// TIA Portal V17 export
// export: Created 2025-03-05T07:59:04.4522338Z, ExportSetting WithDefaults, DisplayName Totally Integrated Automation Portal, DisplayVersion V17 Update 8, DisplayName TIA Portal Openness, DisplayVersion V17 Update 8, DisplayName TIA Portal Version Control Interface, DisplayVersion V17, DisplayName SINAMICS Startdrive Advanced, DisplayVersion V17 SP2, DisplayName SINAMICS Startdrive G110M, G120, G120C, G120D, G120P, G115D, DisplayVersion V17 SP2, DisplayName SINAMICS Startdrive G130, G150, S120, S150, SINAMICS MV, S210, DisplayVersion V17 SP2, DisplayName STEP 7 Professional, DisplayVersion V17 Update 8, DisplayName SINUMERIK ONE STEP 7 Toolbox, DisplayVersion V17 Update 12, DisplayName SINUMERIK 840D sl STEP 7 Toolbox, DisplayVersion V17 Update 12, DisplayName STEP 7 Safety, DisplayVersion V17 Update 6, DisplayName WinCC Advanced, DisplayVersion V17 Update 8
FUNCTION_BLOCK "FB2509_CYL_OPEN_CLOSE_FIX_CLADDING"   // FB2509, LAD
TITLE = CYLINDER CLOSE OPEN
{ S7_Optimized_Access := 'FALSE' }
AUTHOR : ETXETAR
VERSION : 1.0
// stored: AutoNumber false, IsIECCheckEnabled false, SetENOAutomatically false, UDAEnableTagReadback false
   VAR_INPUT
      OPTIONS_0 : Byte := 2#0000_0000;   // OPTIONS 0
      OPTIONS_1 : Byte := 2#0000_0000;   // OPTIONS 1
      OPTIONS_2 : Byte := 2#0000_0000;   // OPTIONS 2
      CLOSED_PART_A : Bool;   // CLOSED PART A INPUT
      CLOSED_PART_B : Bool;   // CLOSED PART B INPUT
      CLOSED_PART_C : Bool;   // CLOSED PART C INPUT
      CLOSED_PART_D : Bool;   // CLOSED PART D INPUT
      OPEN_PART_A : Bool;   // OPEN PART A INPUT
      OPEN_PART_B : Bool;   // OPEN PART B INPUT
      OPEN_PART_C : Bool;   // OPEN PART C INPUT
      OPEN_PART_D : Bool;   // OPEN PART D INPUT
      CLOSED_PRESSURE_SWITCH_1 : Bool;   // CLOSED PRESSURE SWITCH INPUT 1
      CLOSED_PRESSURE_SWITCH_2 : Bool;   // CLOSED PRESSURE SWITCH INPUT 2
      OPEN_PRESSURE_SWITCH_1 : Bool;   // OPEN PRESSURE SWITCH INPUT 1
      OPEN_PRESSURE_SWITCH_2 : Bool;   // OPEN PRESSURE SWITCH INPUT 2
      CLOSED_LOW_PRESSURE_SWITCH : Bool;   // CLOSED LOW PRESSURE SWITCH INPUT
      OPEN_LOW_PRESSURE_SWITCH : Bool;   // OPEN LOW PRESSURE SWITCH INPUT
      GENERAL_CONDITIONS : Bool;   // GENERAL CONDITIONS INPUT
      CLOSE_CONDITIONS : Bool;   // CLOSE CONDITIONS INPUT
      OPEN_CONDITIONS : Bool;   // OPEN CONDITIONS INPUT
      RELEASE_PRESSURE_CONDITIONS : Bool;   // RELEASE PRESSURE CONDITIONS INPUT
      LOW_PRESSURE_CONDITIONS : Bool;   // LOW PRESSURE CONDITIONS INPUT
      HYDRAULIC_OR_PNEUMATIC : Bool;   // HYDRAULIC OR PNEUMATIC IN SERVICE
      FIXTURE_PART_TYPE_SEL : Bool;   // FIXTURE PART TYPE SELECTED
      HMI_CMM_LINE_ACT_DEACT : Bool;   // HMI COMMAND LINE FOR CLOSE OPEN
      HMI_CMM_LINE_RELEASE_LOW : Bool;   // HMI COMMAND LINE FOR RELEASE LOW PRESSURE
      HMI_CLOSE_MAN_REQ : Bool;   // HMI CLOSE MANUAL REQUEST
      HMI_OPEN_MAN_REQ : Bool;   // HMI OPEN MANUAL REQUEST
      HMI_RELEASE_PRESSURE_MAN_REQ : Bool;   // HMI RELEASE PRESSURE MANUAL REQUEST
      HMI_LOW_PRESSURE_MAN_REQ : Bool;   // HMI LOW PRESSURE MANUAL REQUEST
      FLOWMETER_RESET : Bool;   // RESET FLOWMETER
      CLOSE_AUTO_REQ : Bool;   // CLOSE AUTOMATIC REQUEST
      OPEN_AUTO_REQ : Bool;   // OPEN AUTOMATIC REQUEST
      RELEASE_PRESSURE_AUTO_REQ : Bool;   // RELEASE PRESSURE AUTOMATIC REQUEST
      LOW_PRESSURE_AUTO_REQ : Bool;   // LOW PRESSURE AUTOMATIC REQUEST
      M_VERIFY_CLOSED : Bool;   // M CODE TO VERIFY CYLINDER CLOSED
      M_VERIFY_OPEN : Bool;   // M CODE TO VERIFY CYLINDER OPEN
      M_VERIFY_LOW_PRESSURE : Bool;   // M TO VERIFY LOW PRESSURED
      CHECK_CLOSED_CNC_PLC_SIGNAL : Bool;   // CHECK CLOSED CNC PLC SIGNAL
      CHECK_OPEN_CNC_PLC_SIGNAL : Bool;   // CHECK OPEN CNC PLC SIGNAL
      CHECK_CLOSED_LOW_PRESSURE_CNC_PLC_SIGNAL : Bool;   // CHECK CLOSED LOW PRESSURE CNC PLC SIGNAL
      CHECK_OPEN_LOW_PRESSURE_CNC_PLC_SIGNAL : Bool;   // CHECK OPEN LOW PRESSURE CNC PLC SIGNAL
      CLOSE_FLOW_ACTIVE : Bool;   // FLOWMETER CLOSE FLOW ACTIVE
      UNIT_ALARM : UInt;   // UNIT NUMBER MIN. NUMBER=1 MAX. NUMBER=3
      STATION_ALARM : UInt;   // UNIT NUMBER MIN. NUMBER=0 MAX. NUMBER=4
   END_VAR
   VAR_OUTPUT
      CLOSED : Bool;   // CLOSED
      OPEN_STATUS : Bool;   // OPEN
      PRESSURE_RELEASED : Bool;   // PRESSURE RELEASED
      LOW_PRESSURED : Bool;   // LOW PRESSURED
      HMI_MOTION_EXECUTABILITY_LEFT : Bool;   // HMI MOTION EXECUTABILITY LEFT
      HMI_MOTION_EXECUTABILITY_RIGHT : Bool;   // HMI MOTION EXECUTABILITY RIGHT
      HMI_MOTION_EXECUTABILITY_LEFT_2 : Bool;   // HMI MOTION EXECUTABILITY LEFT 2
      HMI_MOTION_EXECUTABILITY_RIGHT_2 : Bool;   // HMI MOTION EXECUTABILITY RIGHT 2
      HMI_MOTION_END_POS_LEFT : Bool;   // HMI MOTION END POSITION LEFT
      HMI_MOTION_END_POS_RIGHT : Bool;   // HMI MOTION END POSITION RIGHT
      HMI_MOTION_END_POS_LEFT_2 : Bool;   // HMI MOTION END POSITION LEFT 2
      HMI_MOTION_END_POS_RIGHT_2 : Bool;   // HMI MOTION END POSITION RIGHT 2
      HMI_MOTION_ACTIVE_LEFT : Bool;   // HMI MOTION ACTIVE LEFT
      HMI_MOTION_ACTIVE_RIGHT : Bool;   // HMI MOTION ACTIVE RIGHT
      HMI_MOTION_ACTIVE_LEFT_2 : Bool;   // HMI MOTION ACTIVE LEFT 2
      HMI_MOTION_ACTIVE_RIGHT_2 : Bool;   // HMI MOTION ACTIVE RIGHT 2
      ALARMS : "CYL_ALARMS_OPN_CLS";
      RESET_FLOWMETER : Bool;   // RESET FLOWMETER
      CLOSE : Bool;   // CLOSE
      OPEN_ACTION : Bool;   // OPEN
      LOW_PRESSURE : Bool;   // LOW PRESSURE
      SAFETY_UNBLOCK : Bool;   // SAFETY UNBLOCK
      PRESSURIZE_A : Bool;   // PRESSURIZE A
      PRESSURIZE_B : Bool;   // PRESSURIZE B
      PRESSURIZE_C : Bool;   // PRESSURIZE C
   END_VAR
   VAR_IN_OUT
      OPEN_FLOW_ACTIVE_FLOWMETER : Bool;   // FLOWMETER OPEN FLOW ACTIVE
   END_VAR
   VAR DB_SPECIFIC
      CYL { S7_SetPoint := 'True'} : "OPEN_CLOSE";
      TIMER_CLOSED { S7_SetPoint := 'True'} : TON_TIME;   // CLOSED TIMER
      TIMER_OPEN { S7_SetPoint := 'True'} : TON_TIME;   // OPEN TIMER
      TIMER_PRESSURE_RELEASED { S7_SetPoint := 'True'} : TON_TIME;   // PRESSURE RELEASED TIMER
      TIMER_LOW_PRESSURE { S7_SetPoint := 'True'} : TON_TIME;   // LOW PRESSURE TIMER
      TIMER_SIMULTANEITY { S7_SetPoint := 'True'} : TON_TIME;   // SIMULTANEITY TIMER
      TIMER_TIME_EXCEEDED { S7_SetPoint := 'True'} : TON_TIME;   // TIME EXCEEDED TIMER
      TIMER_ACTD_PRESSURE_TIME_EXCEEDED_1 { S7_SetPoint := 'True'} : TON_TIME;   // CLOSED PRESSURE TIME EXCEEDED TIMER 1
      TIMER_ACTD_PRESSURE_SWITCH_1 { S7_SetPoint := 'True'} : TON_TIME;   // CLOSED PRESSURE SWITCH TIMER 1
      "TIMER_ACTD PRESSURE_TIME_EXCEEDED_2" { S7_SetPoint := 'True'} : TON_TIME;   // CLOSED PRESSURE TIME EXCEEDED TIMER 2
      "TIMER_ACTD PRESSURE_SWITCH_2" { S7_SetPoint := 'True'} : TON_TIME;   // CLOSED PRESSURE SWITCH TIMER 2
      TIMER_DEACTD_PRESSURE_TIME_EXCEEDED_1 { S7_SetPoint := 'True'} : TON_TIME;   // OPEN PRESSURE TIME EXCEEDED TIMER 1
      TIMER_DEACTD_PRESSURE_SWITCH_1 { S7_SetPoint := 'True'} : TON_TIME;   // OPEN PRESSURE SWITCH TIMER 1
      TIMER_DEACTD_PRESSURE_TIME_EXCEEDED_2 { S7_SetPoint := 'True'} : TON_TIME;   // OPEN PRESSURE TIME EXCEEDED TIMER 2
      TIMER_DEACTD_PRESSURE_SWITCH_2 { S7_SetPoint := 'True'} : TON_TIME;   // OPEN PRESSURE SWITCH TIMER 2
      TIMER_ACTD_LOW_PRESSURE_TIME_EXCEEDED { S7_SetPoint := 'True'} : TON_TIME;   // CLOSED LOW PRESSURE TIME EXCEEDED TIMER
      TIMER_ACTD_LOW_PRESSURE_SWITCH { S7_SetPoint := 'True'} : TON_TIME;   // CLOSED LOW PRESSURE SWITCH TIMER
      TIMER_DEACTD_LOW_PRESSURE_TIME_EXCEEDED { S7_SetPoint := 'True'} : TON_TIME;   // OPEN LOW PRESSURE TIME EXCEEDED TIMER
      TIMER_DEACTD_LOW_PRESSURE_SWITCH { S7_SetPoint := 'True'} : TON_TIME;   // OPEN LOW PRESSURE SWITCH TIMER
      TIMER_SAFETY_UNBLOCK { S7_SetPoint := 'True'} : TOF_TIME;   // SAFETY UNBLOCK TIMER
      TIMER_CLMP_RCVRY_CLAMPED { S7_SetPoint := 'True'} : TON_TIME;   // CLAMP RECOVERY CLAMPED TIMER
      TIMER_CLMP_RCVRY_UNCLAMPED { S7_SetPoint := 'True'} : TON_TIME;   // CLAMP RECOVERY UNCLAMPED TIMER
   END_VAR
   VAR_TEMP
      INPUTS_MASK : Byte;   // INPUTS MASK
      O_BYTE_0 : Struct   // OPTIONS BYTE 0
         CLOSED_PART_A : Bool;   // CLOSED PART A OPTION
         CLOSED_PART_B : Bool;   // CLOSED PART B OPTION
         CLOSED_PART_C : Bool;   // CLOSED PART C OPTION
         CLOSED_PART_D : Bool;   // CLOSED PART D OPTION
         CLOSED_PRESSURE_INPUT_1 : Bool;   // CLOSED PRESSURE INPUT 1 OPTION
         CLOSED_PRESSURE_INPUT_2 : Bool;   // CLOSED PRESSURE INPUT 2 OPTION
         CLOSED_LOW_PRESSURE_INPUT : Bool;   // CLOSED LOW PRESSURE INPUT OPTION
         SPARE_7 : Bool;   // SPARE OPTION
      END_STRUCT;
      O_BYTE_1 : Struct   // OPTIONS BYTE 1
         OPEN_PART_A : Bool;   // OPEN PART A OPTION
         OPEN_PART_B : Bool;   // OPEN PART B OPTION
         OPEN_PART_C : Bool;   // OPEN PART C OPTION
         OPEN_PART_D : Bool;   // OPEN PART D OPTION
         OPEN_PRESSURE_INPUT_1 : Bool;   // OPEN PRESSURE INPUT 1 OPTION
         OPEN_PRESSURE_INPUT_2 : Bool;   // OPEN PRESSURE INPUT 2 OPTION
         OPEN_LOW_PRESSURE_INPUT : Bool;   // OPEN LOW PRESSURE INPUT OPTION
         SPARE_7 : Bool;   // SPARE OPTION
      END_STRUCT;
      O_BYTE_2 : Struct   // OPTIONS BYTE 2
         TWO_STATES_VALVE : Bool;   // TWO STATES VALVE OPTION
         HIGH_LOW_PRESSURE_VALVE : Bool;   // HIGH OR LOW PRESSURE VALVE OPTION
         OPEN_LOW : Bool;   // OPEN LOW OPTION
         SPARE_3 : Bool;   // SPARE OPTION
         SPARE_4 : Bool;   // SPARE OPTION
         SPARE_5 : Bool;   // SPARE OPTION
         SPARE_6 : Bool;   // SPARE OPTION
         CLAMP_RECOVERY : Bool;   // CLAMP RECOVERY OPTION
      END_STRUCT;
      DB_NUMBER : DInt;   // DB NUMBER FOR ALARM AND HELP DECODING
      CLAMP_RECOVERY_AUX : Bool;   // CLAMP RECOVERY AUXILIARY
   END_VAR
   // TIMER_CLOSED.PT := T#100MS;
   // TIMER_OPEN.PT := T#100MS;
   // TIMER_PRESSURE_RELEASED.PT := T#100MS;
   // TIMER_LOW_PRESSURE.PT := T#100MS;
   // TIMER_SIMULTANEITY.PT := T#100MS;
   // TIMER_TIME_EXCEEDED.PT := T#3S;
   // TIMER_ACTD_PRESSURE_TIME_EXCEEDED_1.PT := T#3S;
   // TIMER_ACTD_PRESSURE_SWITCH_1.PT := T#3S;
   // "TIMER_ACTD PRESSURE_TIME_EXCEEDED_2".PT := T#3S;
   // "TIMER_ACTD PRESSURE_SWITCH_2".PT := T#3S;
   // TIMER_DEACTD_PRESSURE_TIME_EXCEEDED_1.PT := T#3S;
   // TIMER_DEACTD_PRESSURE_SWITCH_1.PT := T#3S;
   // TIMER_DEACTD_PRESSURE_TIME_EXCEEDED_2.PT := T#3S;
   // TIMER_DEACTD_PRESSURE_SWITCH_2.PT := T#3S;
   // TIMER_ACTD_LOW_PRESSURE_TIME_EXCEEDED.PT := T#3S;
   // TIMER_ACTD_LOW_PRESSURE_SWITCH.PT := T#3S;
   // TIMER_DEACTD_LOW_PRESSURE_TIME_EXCEEDED.PT := T#3S;
   // TIMER_DEACTD_LOW_PRESSURE_SWITCH.PT := T#3S;
   // TIMER_SAFETY_UNBLOCK.PT := T#5s;
   // TIMER_CLMP_RCVRY_CLAMPED.PT := T#5s;
   // TIMER_CLMP_RCVRY_UNCLAMPED.PT := T#5s;
   VAR_TEMP   // added for the SCL form of the ladder/FBD networks
      _w1 : Bool;
      _w2 : Bool;
      _w3 : Bool;
      _w4 : Bool;
      _w5 : Bool;
      _w6 : Bool;
      _w7 : Bool;
      _w8 : Bool;
      _w9 : Bool;
      _w10 : Bool;
      _w11 : Bool;
      _w12 : Bool;
      _w13 : Bool;
   END_VAR
BEGIN

NETWORK
TITLE = READ INSTANCE DB
      L     DINO;
      +     10#800000;
      T     #DB_NUMBER;


REGION Network 2: OPTIONS
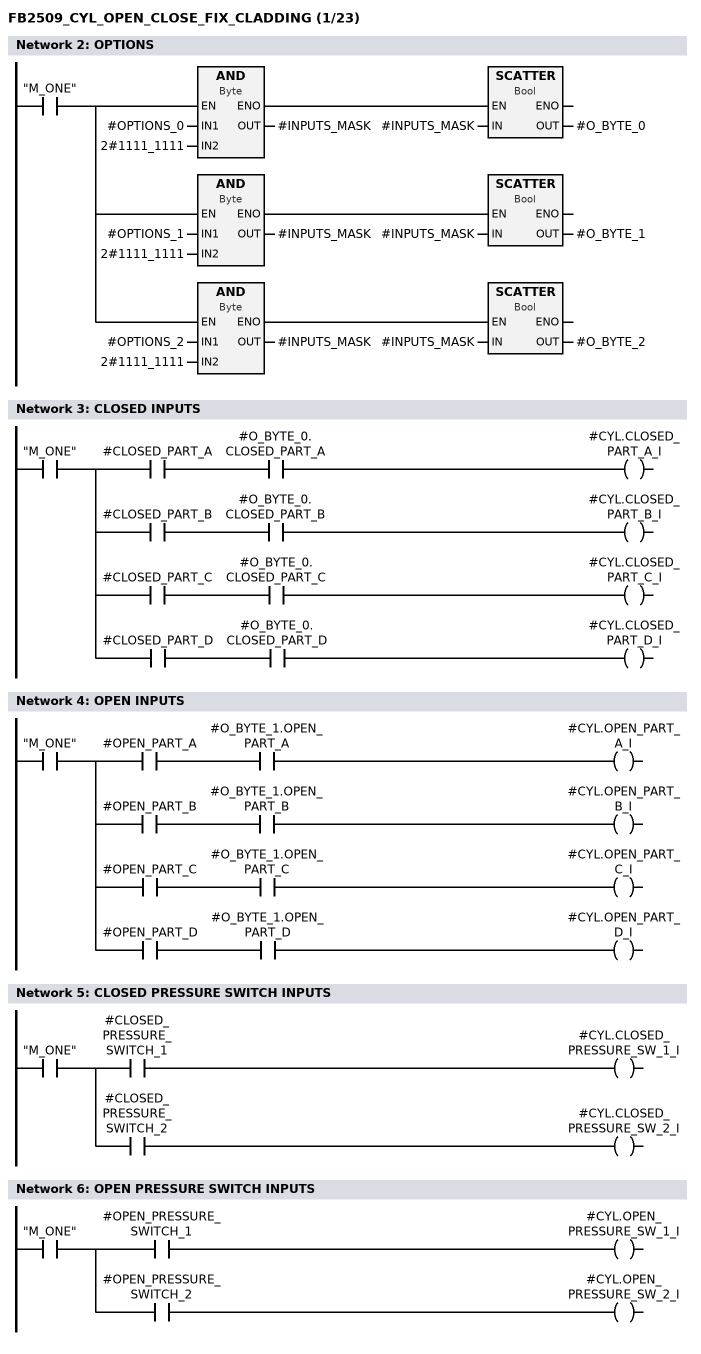
   RUNG wire#powerrail
      Contact( "M_ONE" )
      wire#w1
      { S7_Templates := "SrcType := Byte"; S7_GenerateENO := "TRUE" } And(in1 := #OPTIONS_0, in2 := 2#1111_1111, out => #INPUTS_MASK)
      { S7_Templates := "[dest_type := Bool, src_type := Byte]" } SCATTER(IN := #INPUTS_MASK, OUT => #O_BYTE_0)
   END_RUNG
   RUNG wire#w1
      { S7_Templates := "SrcType := Byte"; S7_GenerateENO := "TRUE" } And(in1 := #OPTIONS_1, in2 := 2#1111_1111, out => #INPUTS_MASK)
      { S7_Templates := "[dest_type := Bool, src_type := Byte]" } SCATTER(IN := #INPUTS_MASK, OUT => #O_BYTE_1)
   END_RUNG
   RUNG wire#w1
      { S7_Templates := "SrcType := Byte"; S7_GenerateENO := "TRUE" } And(in1 := #OPTIONS_2, in2 := 2#1111_1111, out => #INPUTS_MASK)
      { S7_Templates := "[dest_type := Bool, src_type := Byte]" } SCATTER(IN := #INPUTS_MASK, OUT => #O_BYTE_2)
   END_RUNG
   // the same network as SCL:
   IF "M_ONE" THEN #INPUTS_MASK := #OPTIONS_0 AND 2#1111_1111; END_IF;
   #_w1 := "M_ONE";
   IF #_w1 THEN
       SCATTER(IN := #INPUTS_MASK, OUT => #O_BYTE_0);
       #INPUTS_MASK := #OPTIONS_1 AND 2#1111_1111;
       SCATTER(IN := #INPUTS_MASK, OUT => #O_BYTE_1);
       #INPUTS_MASK := #OPTIONS_2 AND 2#1111_1111;
       SCATTER(IN := #INPUTS_MASK, OUT => #O_BYTE_2);
   END_IF;
END_REGION

REGION Network 3: CLOSED INPUTS
   RUNG wire#powerrail
      Contact( "M_ONE" )
      wire#w1
      Contact( #CLOSED_PART_A )
      Contact( #O_BYTE_0.CLOSED_PART_A )
      Coil( #CYL.CLOSED_PART_A_I )
   END_RUNG
   RUNG wire#w1
      Contact( #CLOSED_PART_B )
      Contact( #O_BYTE_0.CLOSED_PART_B )
      Coil( #CYL.CLOSED_PART_B_I )
   END_RUNG
   RUNG wire#w1
      Contact( #CLOSED_PART_C )
      Contact( #O_BYTE_0.CLOSED_PART_C )
      Coil( #CYL.CLOSED_PART_C_I )
   END_RUNG
   RUNG wire#w1
      Contact( #CLOSED_PART_D )
      Contact( #O_BYTE_0.CLOSED_PART_D )
      Coil( #CYL.CLOSED_PART_D_I )
   END_RUNG
   // the same network as SCL:
   #CYL.CLOSED_PART_A_I := "M_ONE" AND #CLOSED_PART_A AND #O_BYTE_0.CLOSED_PART_A;
   #CYL.CLOSED_PART_B_I := "M_ONE" AND #CLOSED_PART_B AND #O_BYTE_0.CLOSED_PART_B;
   #CYL.CLOSED_PART_C_I := "M_ONE" AND #CLOSED_PART_C AND #O_BYTE_0.CLOSED_PART_C;
   #CYL.CLOSED_PART_D_I := "M_ONE" AND #CLOSED_PART_D AND #O_BYTE_0.CLOSED_PART_D;
END_REGION

REGION Network 4: OPEN INPUTS
   RUNG wire#powerrail
      Contact( "M_ONE" )
      wire#w1
      Contact( #OPEN_PART_A )
      Contact( #O_BYTE_1.OPEN_PART_A )
      Coil( #CYL.OPEN_PART_A_I )
   END_RUNG
   RUNG wire#w1
      Contact( #OPEN_PART_B )
      Contact( #O_BYTE_1.OPEN_PART_B )
      Coil( #CYL.OPEN_PART_B_I )
   END_RUNG
   RUNG wire#w1
      Contact( #OPEN_PART_C )
      Contact( #O_BYTE_1.OPEN_PART_C )
      Coil( #CYL.OPEN_PART_C_I )
   END_RUNG
   RUNG wire#w1
      Contact( #OPEN_PART_D )
      Contact( #O_BYTE_1.OPEN_PART_D )
      Coil( #CYL.OPEN_PART_D_I )
   END_RUNG
   // the same network as SCL:
   #CYL.OPEN_PART_A_I := "M_ONE" AND #OPEN_PART_A AND #O_BYTE_1.OPEN_PART_A;
   #CYL.OPEN_PART_B_I := "M_ONE" AND #OPEN_PART_B AND #O_BYTE_1.OPEN_PART_B;
   #CYL.OPEN_PART_C_I := "M_ONE" AND #OPEN_PART_C AND #O_BYTE_1.OPEN_PART_C;
   #CYL.OPEN_PART_D_I := "M_ONE" AND #OPEN_PART_D AND #O_BYTE_1.OPEN_PART_D;
END_REGION

REGION Network 5: CLOSED PRESSURE SWITCH INPUTS
   RUNG wire#powerrail
      Contact( "M_ONE" )
      wire#w1
      Contact( #CLOSED_PRESSURE_SWITCH_1 )
      Coil( #CYL.CLOSED_PRESSURE_SW_1_I )
   END_RUNG
   RUNG wire#w1
      Contact( #CLOSED_PRESSURE_SWITCH_2 )
      Coil( #CYL.CLOSED_PRESSURE_SW_2_I )
   END_RUNG
   // the same network as SCL:
   #CYL.CLOSED_PRESSURE_SW_1_I := "M_ONE" AND #CLOSED_PRESSURE_SWITCH_1;
   #CYL.CLOSED_PRESSURE_SW_2_I := "M_ONE" AND #CLOSED_PRESSURE_SWITCH_2;
END_REGION

REGION Network 6: OPEN PRESSURE SWITCH INPUTS
   RUNG wire#powerrail
      Contact( "M_ONE" )
      wire#w1
      Contact( #OPEN_PRESSURE_SWITCH_1 )
      Coil( #CYL.OPEN_PRESSURE_SW_1_I )
   END_RUNG
   RUNG wire#w1
      Contact( #OPEN_PRESSURE_SWITCH_2 )
      Coil( #CYL.OPEN_PRESSURE_SW_2_I )
   END_RUNG
   // the same network as SCL:
   #CYL.OPEN_PRESSURE_SW_1_I := "M_ONE" AND #OPEN_PRESSURE_SWITCH_1;
   #CYL.OPEN_PRESSURE_SW_2_I := "M_ONE" AND #OPEN_PRESSURE_SWITCH_2;
END_REGION

REGION Network 7: LOW PRESSURE SWITCH INPUT
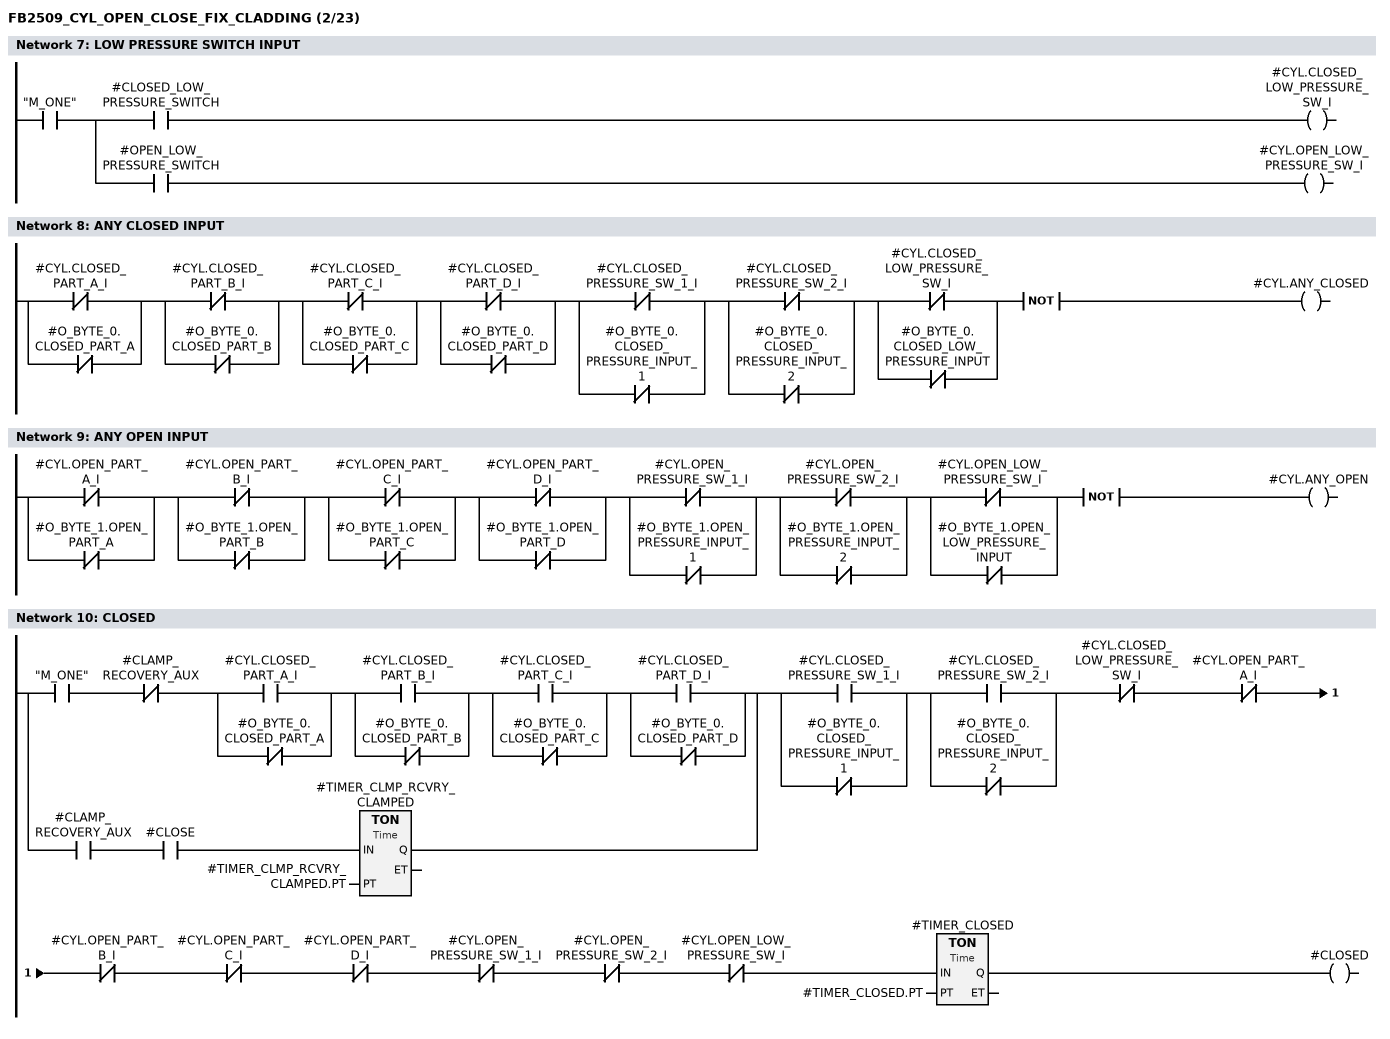
   RUNG wire#powerrail
      Contact( "M_ONE" )
      wire#w1
      Contact( #CLOSED_LOW_PRESSURE_SWITCH )
      Coil( #CYL.CLOSED_LOW_PRESSURE_SW_I )
   END_RUNG
   RUNG wire#w1
      Contact( #OPEN_LOW_PRESSURE_SWITCH )
      Coil( #CYL.OPEN_LOW_PRESSURE_SW_I )
   END_RUNG
   // the same network as SCL:
   #CYL.CLOSED_LOW_PRESSURE_SW_I := "M_ONE" AND #CLOSED_LOW_PRESSURE_SWITCH;
   #CYL.OPEN_LOW_PRESSURE_SW_I := "M_ONE" AND #OPEN_LOW_PRESSURE_SWITCH;
END_REGION

REGION Network 8: ANY CLOSED INPUT
   RUNG wire#powerrail
      I_Contact( #CYL.CLOSED_PART_A_I )
      wire#w1
      I_Contact( #CYL.CLOSED_PART_B_I )
      wire#w2
      I_Contact( #CYL.CLOSED_PART_C_I )
      wire#w3
      I_Contact( #CYL.CLOSED_PART_D_I )
      wire#w4
      I_Contact( #CYL.CLOSED_PRESSURE_SW_1_I )
      wire#w5
      I_Contact( #CYL.CLOSED_PRESSURE_SW_2_I )
      wire#w6
      I_Contact( #CYL.CLOSED_LOW_PRESSURE_SW_I )
      wire#w7
      Not()
      Coil( #CYL.ANY_CLOSED )
   END_RUNG
   RUNG wire#powerrail
      I_Contact( #O_BYTE_0.CLOSED_PART_A )
   END_RUNG wire#w1
   RUNG wire#w1
      I_Contact( #O_BYTE_0.CLOSED_PART_B )
   END_RUNG wire#w2
   RUNG wire#w2
      I_Contact( #O_BYTE_0.CLOSED_PART_C )
   END_RUNG wire#w3
   RUNG wire#w3
      I_Contact( #O_BYTE_0.CLOSED_PART_D )
   END_RUNG wire#w4
   RUNG wire#w4
      I_Contact( #O_BYTE_0.CLOSED_PRESSURE_INPUT_1 )
   END_RUNG wire#w5
   RUNG wire#w5
      I_Contact( #O_BYTE_0.CLOSED_PRESSURE_INPUT_2 )
   END_RUNG wire#w6
   RUNG wire#w6
      I_Contact( #O_BYTE_0.CLOSED_LOW_PRESSURE_INPUT )
   END_RUNG wire#w7
   // the same network as SCL:
   #CYL.ANY_CLOSED := NOT ((NOT #CYL.CLOSED_PART_A_I OR NOT #O_BYTE_0.CLOSED_PART_A) AND (NOT #CYL.CLOSED_PART_B_I OR NOT #O_BYTE_0.CLOSED_PART_B) AND (NOT #CYL.CLOSED_PART_C_I OR NOT #O_BYTE_0.CLOSED_PART_C) AND (NOT #CYL.CLOSED_PART_D_I OR NOT #O_BYTE_0.CLOSED_PART_D) AND (NOT #CYL.CLOSED_PRESSURE_SW_1_I OR NOT #O_BYTE_0.CLOSED_PRESSURE_INPUT_1) AND (NOT #CYL.CLOSED_PRESSURE_SW_2_I OR NOT #O_BYTE_0.CLOSED_PRESSURE_INPUT_2) AND (NOT #CYL.CLOSED_LOW_PRESSURE_SW_I OR NOT #O_BYTE_0.CLOSED_LOW_PRESSURE_INPUT));
END_REGION

REGION Network 9: ANY OPEN INPUT
   RUNG wire#powerrail
      I_Contact( #CYL.OPEN_PART_A_I )
      wire#w1
      I_Contact( #CYL.OPEN_PART_B_I )
      wire#w2
      I_Contact( #CYL.OPEN_PART_C_I )
      wire#w3
      I_Contact( #CYL.OPEN_PART_D_I )
      wire#w4
      I_Contact( #CYL.OPEN_PRESSURE_SW_1_I )
      wire#w5
      I_Contact( #CYL.OPEN_PRESSURE_SW_2_I )
      wire#w6
      I_Contact( #CYL.OPEN_LOW_PRESSURE_SW_I )
      wire#w7
      Not()
      Coil( #CYL.ANY_OPEN )
   END_RUNG
   RUNG wire#powerrail
      I_Contact( #O_BYTE_1.OPEN_PART_A )
   END_RUNG wire#w1
   RUNG wire#w1
      I_Contact( #O_BYTE_1.OPEN_PART_B )
   END_RUNG wire#w2
   RUNG wire#w2
      I_Contact( #O_BYTE_1.OPEN_PART_C )
   END_RUNG wire#w3
   RUNG wire#w3
      I_Contact( #O_BYTE_1.OPEN_PART_D )
   END_RUNG wire#w4
   RUNG wire#w4
      I_Contact( #O_BYTE_1.OPEN_PRESSURE_INPUT_1 )
   END_RUNG wire#w5
   RUNG wire#w5
      I_Contact( #O_BYTE_1.OPEN_PRESSURE_INPUT_2 )
   END_RUNG wire#w6
   RUNG wire#w6
      I_Contact( #O_BYTE_1.OPEN_LOW_PRESSURE_INPUT )
   END_RUNG wire#w7
   // the same network as SCL:
   #CYL.ANY_OPEN := NOT ((NOT #CYL.OPEN_PART_A_I OR NOT #O_BYTE_1.OPEN_PART_A) AND (NOT #CYL.OPEN_PART_B_I OR NOT #O_BYTE_1.OPEN_PART_B) AND (NOT #CYL.OPEN_PART_C_I OR NOT #O_BYTE_1.OPEN_PART_C) AND (NOT #CYL.OPEN_PART_D_I OR NOT #O_BYTE_1.OPEN_PART_D) AND (NOT #CYL.OPEN_PRESSURE_SW_1_I OR NOT #O_BYTE_1.OPEN_PRESSURE_INPUT_1) AND (NOT #CYL.OPEN_PRESSURE_SW_2_I OR NOT #O_BYTE_1.OPEN_PRESSURE_INPUT_2) AND (NOT #CYL.OPEN_LOW_PRESSURE_SW_I OR NOT #O_BYTE_1.OPEN_LOW_PRESSURE_INPUT));
END_REGION

REGION Network 10: CLOSED
   RUNG wire#powerrail
      Contact( "M_ONE" )
      I_Contact( #CLAMP_RECOVERY_AUX )
      wire#w1
      Contact( #CYL.CLOSED_PART_A_I )
      wire#w2
      Contact( #CYL.CLOSED_PART_B_I )
      wire#w3
      Contact( #CYL.CLOSED_PART_C_I )
      wire#w4
      Contact( #CYL.CLOSED_PART_D_I )
      wire#w5
      Contact( #CYL.CLOSED_PRESSURE_SW_1_I )
      wire#w6
      Contact( #CYL.CLOSED_PRESSURE_SW_2_I )
      wire#w7
      I_Contact( #CYL.CLOSED_LOW_PRESSURE_SW_I )
      I_Contact( #CYL.OPEN_PART_A_I )
      I_Contact( #CYL.OPEN_PART_B_I )
      I_Contact( #CYL.OPEN_PART_C_I )
      I_Contact( #CYL.OPEN_PART_D_I )
      I_Contact( #CYL.OPEN_PRESSURE_SW_1_I )
      I_Contact( #CYL.OPEN_PRESSURE_SW_2_I )
      I_Contact( #CYL.OPEN_LOW_PRESSURE_SW_I )
      { S7_Templates := "time_type := Time" } #TIMER_CLOSED.TON(pt := #TIMER_CLOSED.PT, et =>)
      Coil( #CLOSED )
   END_RUNG
   RUNG wire#w1
      I_Contact( #O_BYTE_0.CLOSED_PART_A )
   END_RUNG wire#w2
   RUNG wire#w2
      I_Contact( #O_BYTE_0.CLOSED_PART_B )
   END_RUNG wire#w3
   RUNG wire#w3
      I_Contact( #O_BYTE_0.CLOSED_PART_C )
   END_RUNG wire#w4
   RUNG wire#w4
      I_Contact( #O_BYTE_0.CLOSED_PART_D )
   END_RUNG wire#w5
   RUNG wire#powerrail
      Contact( #CLAMP_RECOVERY_AUX )
      Contact( #CLOSE )
      { S7_Templates := "time_type := Time" } #TIMER_CLMP_RCVRY_CLAMPED.TON(pt := #TIMER_CLMP_RCVRY_CLAMPED.PT, et =>)
   END_RUNG wire#w5
   RUNG wire#w5
      I_Contact( #O_BYTE_0.CLOSED_PRESSURE_INPUT_1 )
   END_RUNG wire#w6
   RUNG wire#w6
      I_Contact( #O_BYTE_0.CLOSED_PRESSURE_INPUT_2 )
   END_RUNG wire#w7
   // the same network as SCL:
   #TIMER_CLMP_RCVRY_CLAMPED(IN := #CLAMP_RECOVERY_AUX AND #CLOSE, PT := #TIMER_CLMP_RCVRY_CLAMPED.PT);   // TON
   #TIMER_CLOSED(IN := (("M_ONE" AND NOT #CLAMP_RECOVERY_AUX AND (#CYL.CLOSED_PART_A_I OR NOT #O_BYTE_0.CLOSED_PART_A) AND (#CYL.CLOSED_PART_B_I OR NOT #O_BYTE_0.CLOSED_PART_B) AND (#CYL.CLOSED_PART_C_I OR NOT #O_BYTE_0.CLOSED_PART_C) AND (#CYL.CLOSED_PART_D_I OR NOT #O_BYTE_0.CLOSED_PART_D)) OR #TIMER_CLMP_RCVRY_CLAMPED.Q) AND (#CYL.CLOSED_PRESSURE_SW_1_I OR NOT #O_BYTE_0.CLOSED_PRESSURE_INPUT_1) AND (#CYL.CLOSED_PRESSURE_SW_2_I OR NOT #O_BYTE_0.CLOSED_PRESSURE_INPUT_2) AND NOT #CYL.CLOSED_LOW_PRESSURE_SW_I AND NOT #CYL.OPEN_PART_A_I AND NOT #CYL.OPEN_PART_B_I AND NOT #CYL.OPEN_PART_C_I AND NOT #CYL.OPEN_PART_D_I AND NOT #CYL.OPEN_PRESSURE_SW_1_I AND NOT #CYL.OPEN_PRESSURE_SW_2_I AND NOT #CYL.OPEN_LOW_PRESSURE_SW_I,   // TON
                 PT := #TIMER_CLOSED.PT);
   #CLOSED := #TIMER_CLOSED.Q;
END_REGION

REGION Network 11: OPEN
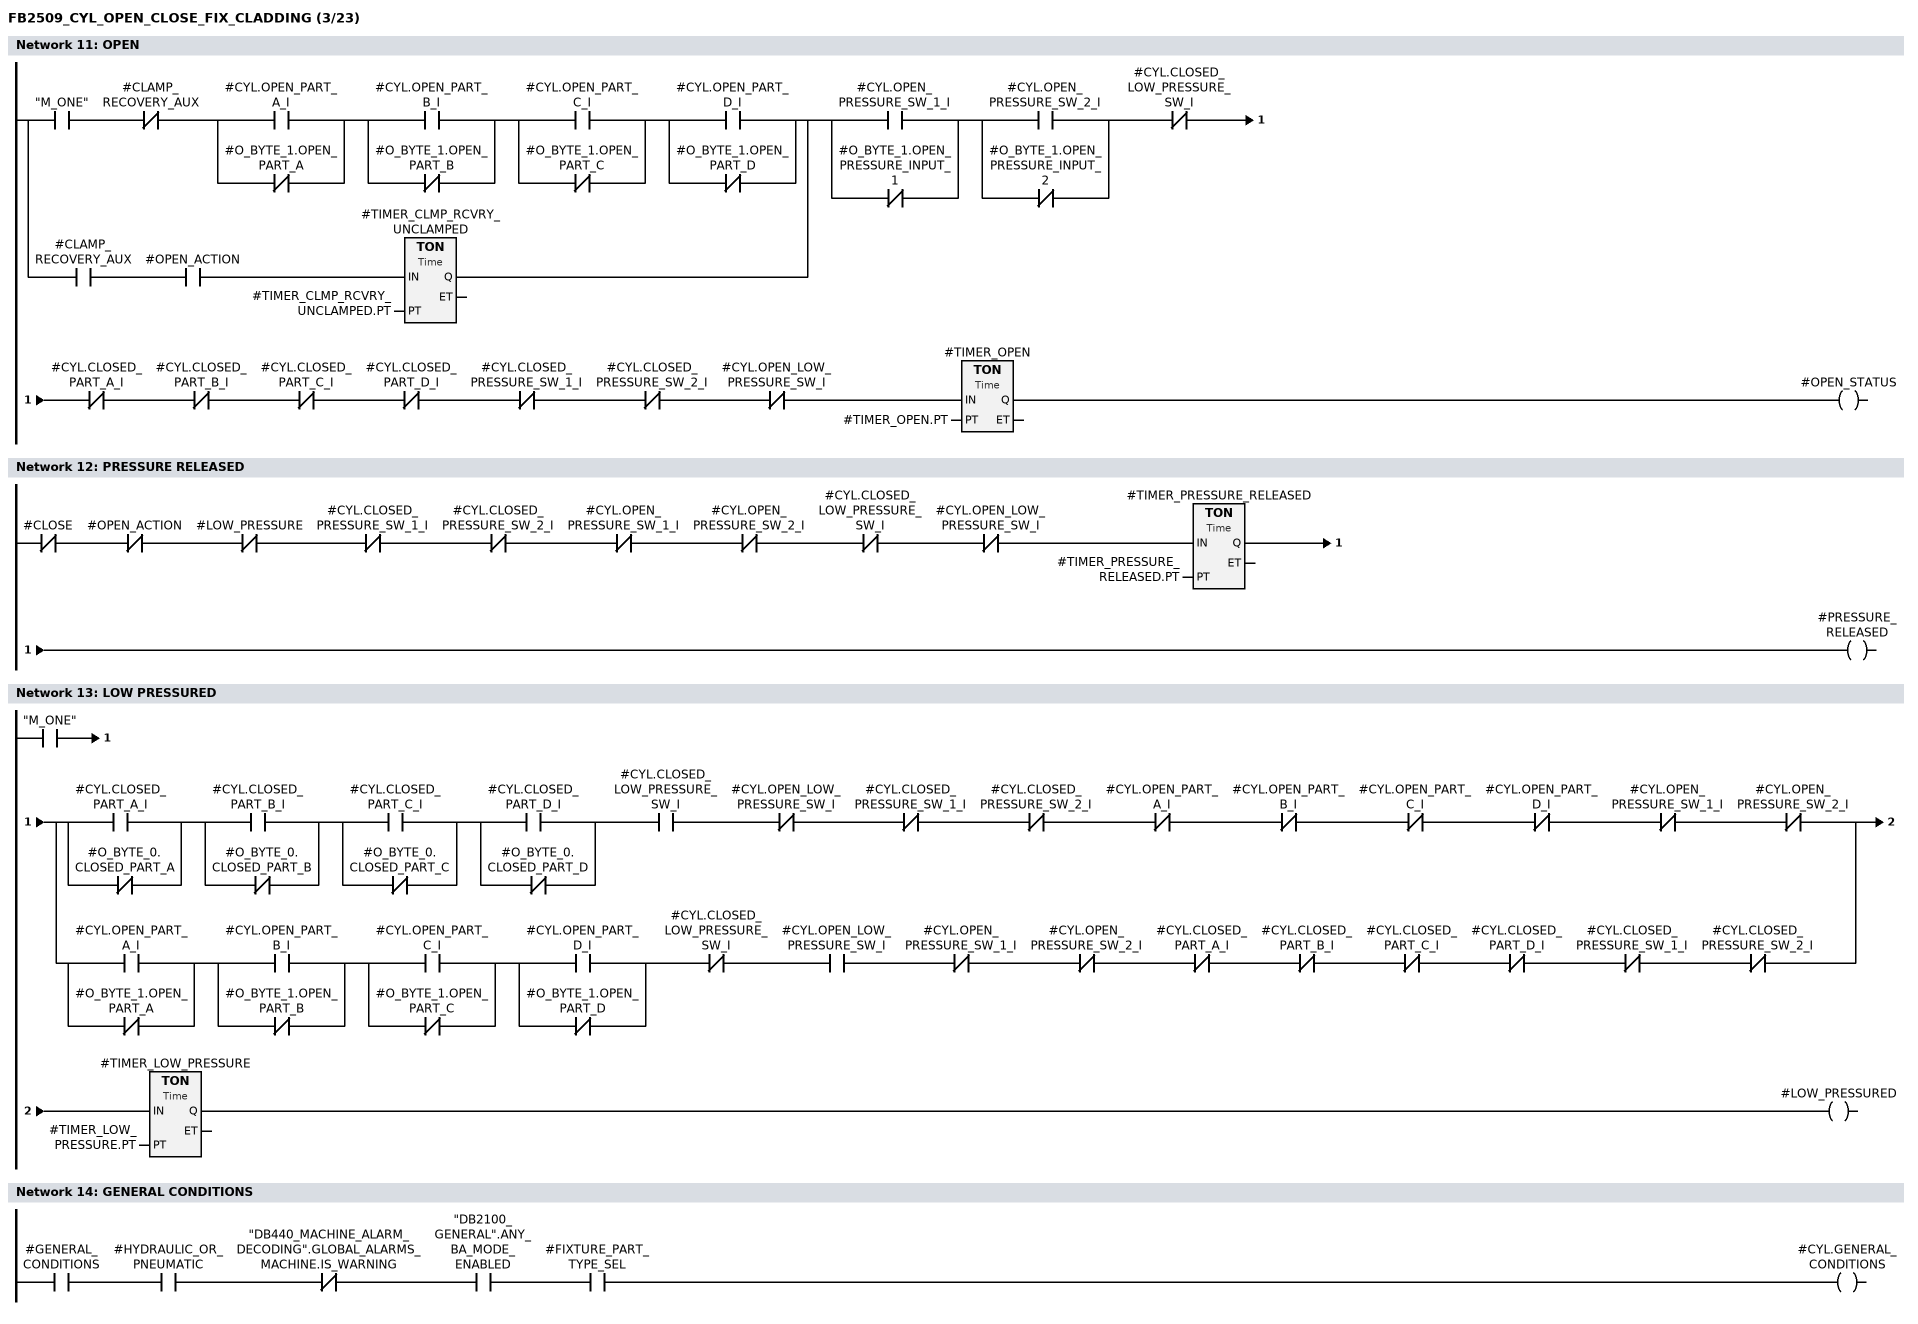
   RUNG wire#powerrail
      Contact( "M_ONE" )
      I_Contact( #CLAMP_RECOVERY_AUX )
      wire#w1
      Contact( #CYL.OPEN_PART_A_I )
      wire#w2
      Contact( #CYL.OPEN_PART_B_I )
      wire#w3
      Contact( #CYL.OPEN_PART_C_I )
      wire#w4
      Contact( #CYL.OPEN_PART_D_I )
      wire#w5
      Contact( #CYL.OPEN_PRESSURE_SW_1_I )
      wire#w6
      Contact( #CYL.OPEN_PRESSURE_SW_2_I )
      wire#w7
      I_Contact( #CYL.CLOSED_LOW_PRESSURE_SW_I )
      I_Contact( #CYL.CLOSED_PART_A_I )
      I_Contact( #CYL.CLOSED_PART_B_I )
      I_Contact( #CYL.CLOSED_PART_C_I )
      I_Contact( #CYL.CLOSED_PART_D_I )
      I_Contact( #CYL.CLOSED_PRESSURE_SW_1_I )
      I_Contact( #CYL.CLOSED_PRESSURE_SW_2_I )
      I_Contact( #CYL.OPEN_LOW_PRESSURE_SW_I )
      { S7_Templates := "time_type := Time" } #TIMER_OPEN.TON(pt := #TIMER_OPEN.PT, et =>)
      Coil( #OPEN_STATUS )
   END_RUNG
   RUNG wire#w1
      I_Contact( #O_BYTE_1.OPEN_PART_A )
   END_RUNG wire#w2
   RUNG wire#w2
      I_Contact( #O_BYTE_1.OPEN_PART_B )
   END_RUNG wire#w3
   RUNG wire#w3
      I_Contact( #O_BYTE_1.OPEN_PART_C )
   END_RUNG wire#w4
   RUNG wire#w4
      I_Contact( #O_BYTE_1.OPEN_PART_D )
   END_RUNG wire#w5
   RUNG wire#powerrail
      Contact( #CLAMP_RECOVERY_AUX )
      Contact( #OPEN_ACTION )
      { S7_Templates := "time_type := Time" } #TIMER_CLMP_RCVRY_UNCLAMPED.TON(pt := #TIMER_CLMP_RCVRY_UNCLAMPED.PT, et =>)
   END_RUNG wire#w5
   RUNG wire#w5
      I_Contact( #O_BYTE_1.OPEN_PRESSURE_INPUT_1 )
   END_RUNG wire#w6
   RUNG wire#w6
      I_Contact( #O_BYTE_1.OPEN_PRESSURE_INPUT_2 )
   END_RUNG wire#w7
   // the same network as SCL:
   #TIMER_CLMP_RCVRY_UNCLAMPED(IN := #CLAMP_RECOVERY_AUX AND #OPEN_ACTION, PT := #TIMER_CLMP_RCVRY_UNCLAMPED.PT);   // TON
   #TIMER_OPEN(IN := (("M_ONE" AND NOT #CLAMP_RECOVERY_AUX AND (#CYL.OPEN_PART_A_I OR NOT #O_BYTE_1.OPEN_PART_A) AND (#CYL.OPEN_PART_B_I OR NOT #O_BYTE_1.OPEN_PART_B) AND (#CYL.OPEN_PART_C_I OR NOT #O_BYTE_1.OPEN_PART_C) AND (#CYL.OPEN_PART_D_I OR NOT #O_BYTE_1.OPEN_PART_D)) OR #TIMER_CLMP_RCVRY_UNCLAMPED.Q) AND (#CYL.OPEN_PRESSURE_SW_1_I OR NOT #O_BYTE_1.OPEN_PRESSURE_INPUT_1) AND (#CYL.OPEN_PRESSURE_SW_2_I OR NOT #O_BYTE_1.OPEN_PRESSURE_INPUT_2) AND NOT #CYL.CLOSED_LOW_PRESSURE_SW_I AND NOT #CYL.CLOSED_PART_A_I AND NOT #CYL.CLOSED_PART_B_I AND NOT #CYL.CLOSED_PART_C_I AND NOT #CYL.CLOSED_PART_D_I AND NOT #CYL.CLOSED_PRESSURE_SW_1_I AND NOT #CYL.CLOSED_PRESSURE_SW_2_I AND NOT #CYL.OPEN_LOW_PRESSURE_SW_I,   // TON
               PT := #TIMER_OPEN.PT);
   #OPEN_STATUS := #TIMER_OPEN.Q;
END_REGION

REGION Network 12: PRESSURE RELEASED
   RUNG wire#powerrail
      I_Contact( #CLOSE )
      I_Contact( #OPEN_ACTION )
      I_Contact( #LOW_PRESSURE )
      I_Contact( #CYL.CLOSED_PRESSURE_SW_1_I )
      I_Contact( #CYL.CLOSED_PRESSURE_SW_2_I )
      I_Contact( #CYL.OPEN_PRESSURE_SW_1_I )
      I_Contact( #CYL.OPEN_PRESSURE_SW_2_I )
      I_Contact( #CYL.CLOSED_LOW_PRESSURE_SW_I )
      I_Contact( #CYL.OPEN_LOW_PRESSURE_SW_I )
      { S7_Templates := "time_type := Time" } #TIMER_PRESSURE_RELEASED.TON(pt := #TIMER_PRESSURE_RELEASED.PT, et =>)
      Coil( #PRESSURE_RELEASED )
   END_RUNG
   // the same network as SCL:
   #TIMER_PRESSURE_RELEASED(IN := NOT #CLOSE AND NOT #OPEN_ACTION AND NOT #LOW_PRESSURE AND NOT #CYL.CLOSED_PRESSURE_SW_1_I AND NOT #CYL.CLOSED_PRESSURE_SW_2_I AND NOT #CYL.OPEN_PRESSURE_SW_1_I AND NOT #CYL.OPEN_PRESSURE_SW_2_I AND NOT #CYL.CLOSED_LOW_PRESSURE_SW_I AND NOT #CYL.OPEN_LOW_PRESSURE_SW_I,   // TON
                           PT := #TIMER_PRESSURE_RELEASED.PT);
   #PRESSURE_RELEASED := #TIMER_PRESSURE_RELEASED.Q;
END_REGION

REGION Network 13: LOW PRESSURED
   RUNG wire#powerrail
      Contact( "M_ONE" )
      wire#w1
      Contact( #CYL.CLOSED_PART_A_I )
      wire#w2
      Contact( #CYL.CLOSED_PART_B_I )
      wire#w3
      Contact( #CYL.CLOSED_PART_C_I )
      wire#w4
      Contact( #CYL.CLOSED_PART_D_I )
      wire#w5
      Contact( #CYL.CLOSED_LOW_PRESSURE_SW_I )
      I_Contact( #CYL.OPEN_LOW_PRESSURE_SW_I )
      I_Contact( #CYL.CLOSED_PRESSURE_SW_1_I )
      I_Contact( #CYL.CLOSED_PRESSURE_SW_2_I )
      I_Contact( #CYL.OPEN_PART_A_I )
      I_Contact( #CYL.OPEN_PART_B_I )
      I_Contact( #CYL.OPEN_PART_C_I )
      I_Contact( #CYL.OPEN_PART_D_I )
      I_Contact( #CYL.OPEN_PRESSURE_SW_1_I )
      I_Contact( #CYL.OPEN_PRESSURE_SW_2_I )
      wire#w6
      { S7_Templates := "time_type := Time" } #TIMER_LOW_PRESSURE.TON(pt := #TIMER_LOW_PRESSURE.PT, et =>)
      Coil( #LOW_PRESSURED )
   END_RUNG
   RUNG wire#w1
      I_Contact( #O_BYTE_0.CLOSED_PART_A )
   END_RUNG wire#w2
   RUNG wire#w2
      I_Contact( #O_BYTE_0.CLOSED_PART_B )
   END_RUNG wire#w3
   RUNG wire#w3
      I_Contact( #O_BYTE_0.CLOSED_PART_C )
   END_RUNG wire#w4
   RUNG wire#w4
      I_Contact( #O_BYTE_0.CLOSED_PART_D )
   END_RUNG wire#w5
   RUNG wire#w1
      Contact( #CYL.OPEN_PART_A_I )
      wire#w7
      Contact( #CYL.OPEN_PART_B_I )
      wire#w8
      Contact( #CYL.OPEN_PART_C_I )
      wire#w9
      Contact( #CYL.OPEN_PART_D_I )
      wire#w10
      I_Contact( #CYL.CLOSED_LOW_PRESSURE_SW_I )
      Contact( #CYL.OPEN_LOW_PRESSURE_SW_I )
      I_Contact( #CYL.OPEN_PRESSURE_SW_1_I )
      I_Contact( #CYL.OPEN_PRESSURE_SW_2_I )
      I_Contact( #CYL.CLOSED_PART_A_I )
      I_Contact( #CYL.CLOSED_PART_B_I )
      I_Contact( #CYL.CLOSED_PART_C_I )
      I_Contact( #CYL.CLOSED_PART_D_I )
      I_Contact( #CYL.CLOSED_PRESSURE_SW_1_I )
      I_Contact( #CYL.CLOSED_PRESSURE_SW_2_I )
   END_RUNG wire#w6
   RUNG wire#w1
      I_Contact( #O_BYTE_1.OPEN_PART_A )
   END_RUNG wire#w7
   RUNG wire#w7
      I_Contact( #O_BYTE_1.OPEN_PART_B )
   END_RUNG wire#w8
   RUNG wire#w8
      I_Contact( #O_BYTE_1.OPEN_PART_C )
   END_RUNG wire#w9
   RUNG wire#w9
      I_Contact( #O_BYTE_1.OPEN_PART_D )
   END_RUNG wire#w10
   // the same network as SCL:
   #TIMER_LOW_PRESSURE(IN := "M_ONE" AND (((#CYL.CLOSED_PART_A_I OR NOT #O_BYTE_0.CLOSED_PART_A) AND (#CYL.CLOSED_PART_B_I OR NOT #O_BYTE_0.CLOSED_PART_B) AND (#CYL.CLOSED_PART_C_I OR NOT #O_BYTE_0.CLOSED_PART_C) AND (#CYL.CLOSED_PART_D_I OR NOT #O_BYTE_0.CLOSED_PART_D) AND #CYL.CLOSED_LOW_PRESSURE_SW_I AND NOT #CYL.OPEN_LOW_PRESSURE_SW_I AND NOT #CYL.CLOSED_PRESSURE_SW_1_I AND NOT #CYL.CLOSED_PRESSURE_SW_2_I AND NOT #CYL.OPEN_PART_A_I AND NOT #CYL.OPEN_PART_B_I AND NOT #CYL.OPEN_PART_C_I AND NOT #CYL.OPEN_PART_D_I AND NOT #CYL.OPEN_PRESSURE_SW_1_I AND NOT #CYL.OPEN_PRESSURE_SW_2_I) OR ((#CYL.OPEN_PART_A_I OR NOT #O_BYTE_1.OPEN_PART_A) AND (#CYL.OPEN_PART_B_I OR NOT #O_BYTE_1.OPEN_PART_B) AND (#CYL.OPEN_PART_C_I OR NOT #O_BYTE_1.OPEN_PART_C) AND (#CYL.OPEN_PART_D_I OR NOT #O_BYTE_1.OPEN_PART_D) AND NOT #CYL.CLOSED_LOW_PRESSURE_SW_I AND #CYL.OPEN_LOW_PRESSURE_SW_I AND NOT #CYL.OPEN_PRESSURE_SW_1_I AND NOT #CYL.OPEN_PRESSURE_SW_2_I AND NOT #CYL.CLOSED_PART_A_I AND NOT #CYL.CLOSED_PART_B_I AND NOT #CYL.CLOSED_PART_C_I AND NOT #CYL.CLOSED_PART_D_I AND NOT #CYL.CLOSED_PRESSURE_SW_1_I AND NOT #CYL.CLOSED_PRESSURE_SW_2_I)),   // TON
                       PT := #TIMER_LOW_PRESSURE.PT);
   #LOW_PRESSURED := #TIMER_LOW_PRESSURE.Q;
END_REGION

REGION Network 14: GENERAL CONDITIONS
   RUNG wire#powerrail
      Contact( #GENERAL_CONDITIONS )
      Contact( #HYDRAULIC_OR_PNEUMATIC )
      I_Contact( "DB440_MACHINE_ALARM_DECODING".GLOBAL_ALARMS_MACHINE.IS_WARNING )
      Contact( "DB2100_GENERAL".ANY_BA_MODE_ENABLED )
      Contact( #FIXTURE_PART_TYPE_SEL )
      Coil( #CYL.GENERAL_CONDITIONS )
   END_RUNG
   // the same network as SCL:
   #CYL.GENERAL_CONDITIONS := #GENERAL_CONDITIONS AND #HYDRAULIC_OR_PNEUMATIC AND NOT "DB440_MACHINE_ALARM_DECODING".GLOBAL_ALARMS_MACHINE.IS_WARNING AND "DB2100_GENERAL".ANY_BA_MODE_ENABLED AND #FIXTURE_PART_TYPE_SEL;
END_REGION

REGION Network 15: OPERATOR HELP
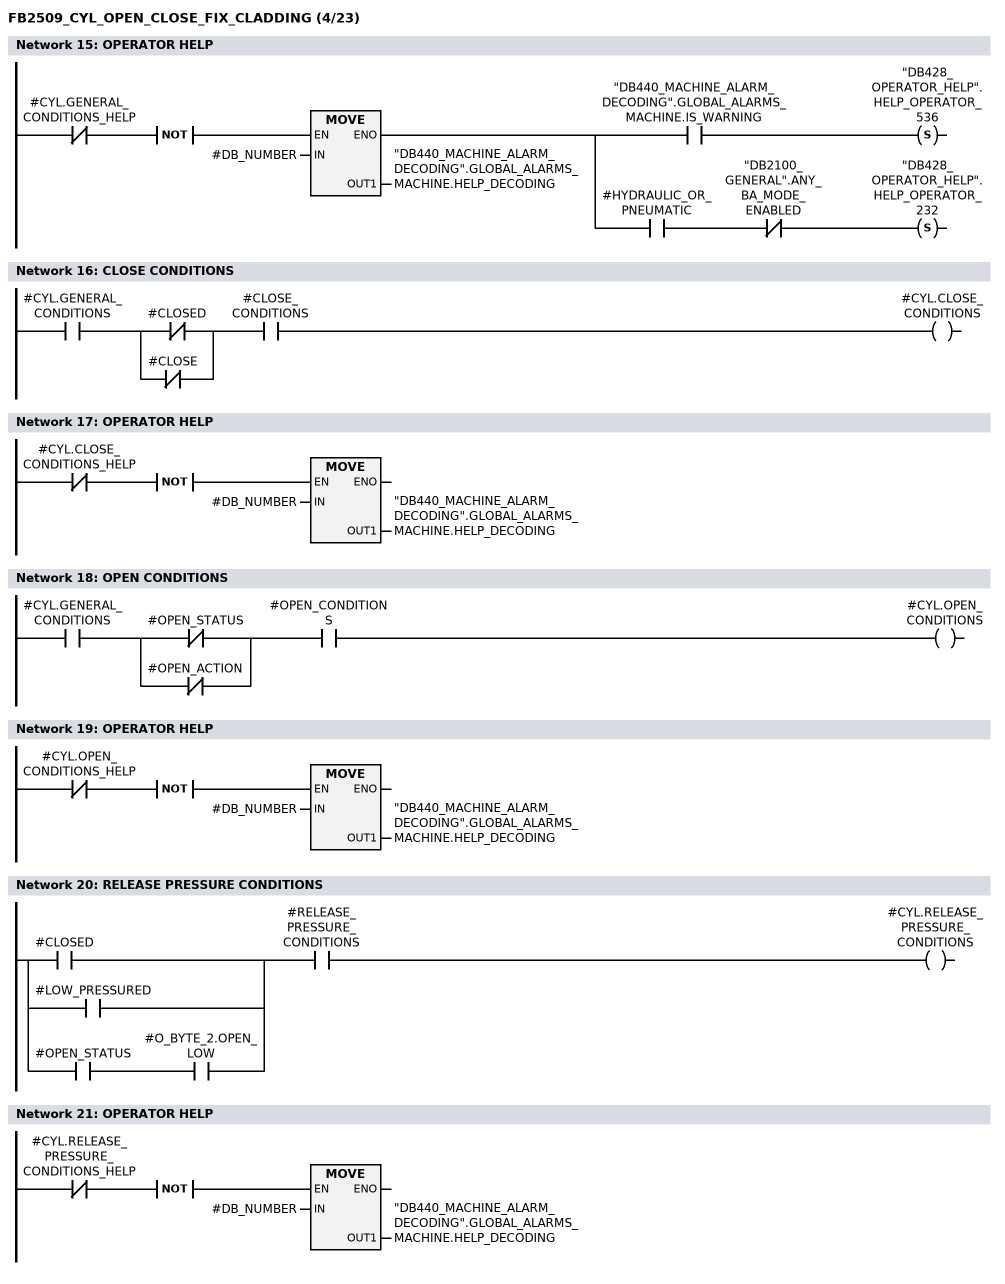
   RUNG wire#powerrail
      I_Contact( #CYL.GENERAL_CONDITIONS_HELP )
      Not()
      { S7_GenerateENO := "TRUE" } Move(in := #DB_NUMBER, out1 => "DB440_MACHINE_ALARM_DECODING".GLOBAL_ALARMS_MACHINE.HELP_DECODING)
      wire#w1
      Contact( "DB440_MACHINE_ALARM_DECODING".GLOBAL_ALARMS_MACHINE.IS_WARNING )
      S_Coil( "DB428_OPERATOR_HELP".HELP_OPERATOR_536 )
   END_RUNG
   RUNG wire#w1
      Contact( #HYDRAULIC_OR_PNEUMATIC )
      I_Contact( "DB2100_GENERAL".ANY_BA_MODE_ENABLED )
      S_Coil( "DB428_OPERATOR_HELP".HELP_OPERATOR_232 )
   END_RUNG
   // the same network as SCL:
   // ENO of a box is taken as its EN; it also drops when the box reports an error
   #_w1 := NOT (NOT #CYL.GENERAL_CONDITIONS_HELP);
   IF #_w1 THEN "DB440_MACHINE_ALARM_DECODING".GLOBAL_ALARMS_MACHINE.HELP_DECODING := #DB_NUMBER; END_IF;
   IF #_w1 AND "DB440_MACHINE_ALARM_DECODING".GLOBAL_ALARMS_MACHINE.IS_WARNING THEN
       "DB428_OPERATOR_HELP".HELP_OPERATOR_536 := TRUE;
   END_IF;
   IF #_w1 AND #HYDRAULIC_OR_PNEUMATIC AND NOT "DB2100_GENERAL".ANY_BA_MODE_ENABLED THEN
       "DB428_OPERATOR_HELP".HELP_OPERATOR_232 := TRUE;
   END_IF;
END_REGION

REGION Network 16: CLOSE CONDITIONS
   RUNG wire#powerrail
      Contact( #CYL.GENERAL_CONDITIONS )
      wire#w1
      I_Contact( #CLOSED )
      wire#w2
      Contact( #CLOSE_CONDITIONS )
      Coil( #CYL.CLOSE_CONDITIONS )
   END_RUNG
   RUNG wire#w1
      I_Contact( #CLOSE )
   END_RUNG wire#w2
   // the same network as SCL:
   #CYL.CLOSE_CONDITIONS := #CYL.GENERAL_CONDITIONS AND (NOT #CLOSED OR NOT #CLOSE) AND #CLOSE_CONDITIONS;
END_REGION

REGION Network 17: OPERATOR HELP
   RUNG wire#powerrail
      I_Contact( #CYL.CLOSE_CONDITIONS_HELP )
      Not()
      { S7_GenerateENO := "TRUE" } Move(in := #DB_NUMBER, out1 => "DB440_MACHINE_ALARM_DECODING".GLOBAL_ALARMS_MACHINE.HELP_DECODING)
   END_RUNG
   // the same network as SCL:
   IF NOT (NOT #CYL.CLOSE_CONDITIONS_HELP) THEN
       "DB440_MACHINE_ALARM_DECODING".GLOBAL_ALARMS_MACHINE.HELP_DECODING := #DB_NUMBER;
   END_IF;
END_REGION

REGION Network 18: OPEN CONDITIONS
   RUNG wire#powerrail
      Contact( #CYL.GENERAL_CONDITIONS )
      wire#w1
      I_Contact( #OPEN_STATUS )
      wire#w2
      Contact( #OPEN_CONDITIONS )
      Coil( #CYL.OPEN_CONDITIONS )
   END_RUNG
   RUNG wire#w1
      I_Contact( #OPEN_ACTION )
   END_RUNG wire#w2
   // the same network as SCL:
   #CYL.OPEN_CONDITIONS := #CYL.GENERAL_CONDITIONS AND (NOT #OPEN_STATUS OR NOT #OPEN_ACTION) AND #OPEN_CONDITIONS;
END_REGION

REGION Network 19: OPERATOR HELP
   RUNG wire#powerrail
      I_Contact( #CYL.OPEN_CONDITIONS_HELP )
      Not()
      { S7_GenerateENO := "TRUE" } Move(in := #DB_NUMBER, out1 => "DB440_MACHINE_ALARM_DECODING".GLOBAL_ALARMS_MACHINE.HELP_DECODING)
   END_RUNG
   // the same network as SCL:
   IF NOT (NOT #CYL.OPEN_CONDITIONS_HELP) THEN
       "DB440_MACHINE_ALARM_DECODING".GLOBAL_ALARMS_MACHINE.HELP_DECODING := #DB_NUMBER;
   END_IF;
END_REGION

REGION Network 20: RELEASE PRESSURE CONDITIONS
   RUNG wire#powerrail
      Contact( #CLOSED )
      wire#w1
      Contact( #RELEASE_PRESSURE_CONDITIONS )
      Coil( #CYL.RELEASE_PRESSURE_CONDITIONS )
   END_RUNG
   RUNG wire#powerrail
      Contact( #LOW_PRESSURED )
   END_RUNG wire#w1
   RUNG wire#powerrail
      Contact( #OPEN_STATUS )
      Contact( #O_BYTE_2.OPEN_LOW )
   END_RUNG wire#w1
   // the same network as SCL:
   #CYL.RELEASE_PRESSURE_CONDITIONS := (#CLOSED OR #LOW_PRESSURED OR (#OPEN_STATUS AND #O_BYTE_2.OPEN_LOW)) AND #RELEASE_PRESSURE_CONDITIONS;
END_REGION

REGION Network 21: OPERATOR HELP
   RUNG wire#powerrail
      I_Contact( #CYL.RELEASE_PRESSURE_CONDITIONS_HELP )
      Not()
      { S7_GenerateENO := "TRUE" } Move(in := #DB_NUMBER, out1 => "DB440_MACHINE_ALARM_DECODING".GLOBAL_ALARMS_MACHINE.HELP_DECODING)
   END_RUNG
   // the same network as SCL:
   IF NOT (NOT #CYL.RELEASE_PRESSURE_CONDITIONS_HELP) THEN
       "DB440_MACHINE_ALARM_DECODING".GLOBAL_ALARMS_MACHINE.HELP_DECODING := #DB_NUMBER;
   END_IF;
END_REGION

REGION Network 22: LOW PRESSURE CONDITIONS
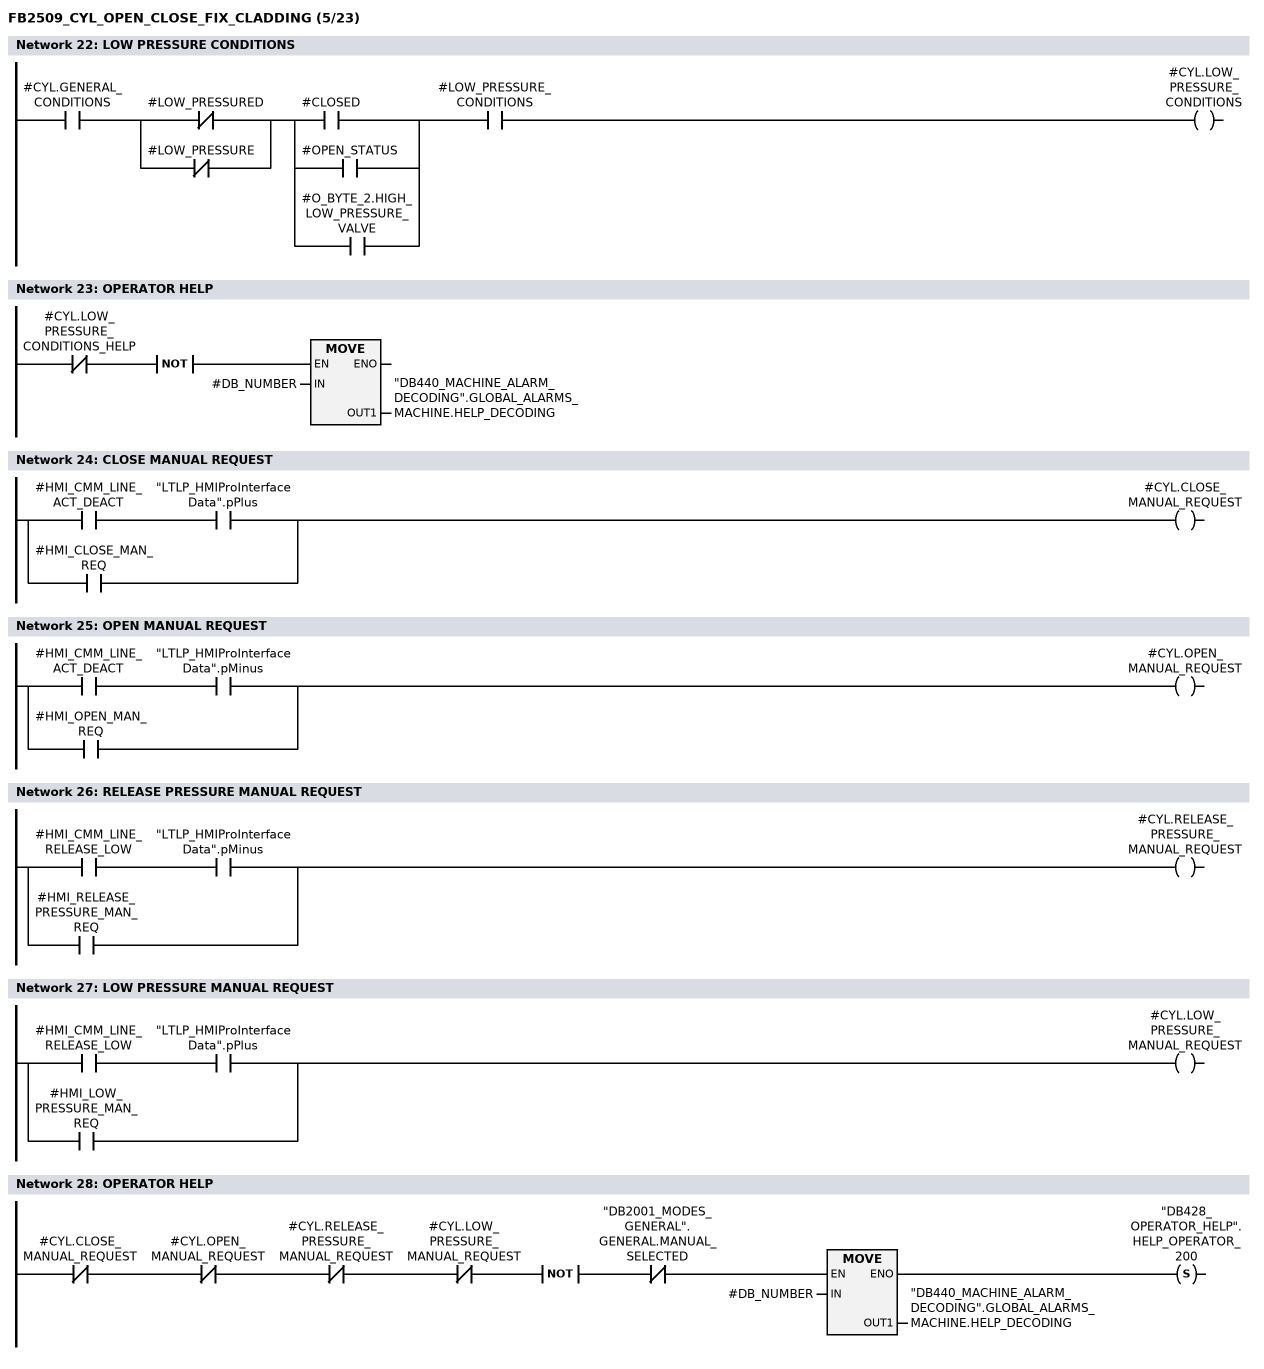
   RUNG wire#powerrail
      Contact( #CYL.GENERAL_CONDITIONS )
      wire#w1
      I_Contact( #LOW_PRESSURED )
      wire#w2
      Contact( #CLOSED )
      wire#w3
      Contact( #LOW_PRESSURE_CONDITIONS )
      Coil( #CYL.LOW_PRESSURE_CONDITIONS )
   END_RUNG
   RUNG wire#w1
      I_Contact( #LOW_PRESSURE )
   END_RUNG wire#w2
   RUNG wire#w2
      Contact( #OPEN_STATUS )
   END_RUNG wire#w3
   RUNG wire#w2
      Contact( #O_BYTE_2.HIGH_LOW_PRESSURE_VALVE )
   END_RUNG wire#w3
   // the same network as SCL:
   #CYL.LOW_PRESSURE_CONDITIONS := #CYL.GENERAL_CONDITIONS AND (NOT #LOW_PRESSURED OR NOT #LOW_PRESSURE) AND (#CLOSED OR #OPEN_STATUS OR #O_BYTE_2.HIGH_LOW_PRESSURE_VALVE) AND #LOW_PRESSURE_CONDITIONS;
END_REGION

REGION Network 23: OPERATOR HELP
   RUNG wire#powerrail
      I_Contact( #CYL.LOW_PRESSURE_CONDITIONS_HELP )
      Not()
      { S7_GenerateENO := "TRUE" } Move(in := #DB_NUMBER, out1 => "DB440_MACHINE_ALARM_DECODING".GLOBAL_ALARMS_MACHINE.HELP_DECODING)
   END_RUNG
   // the same network as SCL:
   IF NOT (NOT #CYL.LOW_PRESSURE_CONDITIONS_HELP) THEN
       "DB440_MACHINE_ALARM_DECODING".GLOBAL_ALARMS_MACHINE.HELP_DECODING := #DB_NUMBER;
   END_IF;
END_REGION

REGION Network 24: CLOSE MANUAL REQUEST
   RUNG wire#powerrail
      Contact( #HMI_CMM_LINE_ACT_DEACT )
      Contact( "LTLP_HMIProInterfaceData".pPlus )
      wire#w1
      Coil( #CYL.CLOSE_MANUAL_REQUEST )
   END_RUNG
   RUNG wire#powerrail
      Contact( #HMI_CLOSE_MAN_REQ )
   END_RUNG wire#w1
   // the same network as SCL:
   #CYL.CLOSE_MANUAL_REQUEST := (#HMI_CMM_LINE_ACT_DEACT AND "LTLP_HMIProInterfaceData".pPlus) OR #HMI_CLOSE_MAN_REQ;
END_REGION

REGION Network 25: OPEN MANUAL REQUEST
   RUNG wire#powerrail
      Contact( #HMI_CMM_LINE_ACT_DEACT )
      Contact( "LTLP_HMIProInterfaceData".pMinus )
      wire#w1
      Coil( #CYL.OPEN_MANUAL_REQUEST )
   END_RUNG
   RUNG wire#powerrail
      Contact( #HMI_OPEN_MAN_REQ )
   END_RUNG wire#w1
   // the same network as SCL:
   #CYL.OPEN_MANUAL_REQUEST := (#HMI_CMM_LINE_ACT_DEACT AND "LTLP_HMIProInterfaceData".pMinus) OR #HMI_OPEN_MAN_REQ;
END_REGION

REGION Network 26: RELEASE PRESSURE MANUAL REQUEST
   RUNG wire#powerrail
      Contact( #HMI_CMM_LINE_RELEASE_LOW )
      Contact( "LTLP_HMIProInterfaceData".pMinus )
      wire#w1
      Coil( #CYL.RELEASE_PRESSURE_MANUAL_REQUEST )
   END_RUNG
   RUNG wire#powerrail
      Contact( #HMI_RELEASE_PRESSURE_MAN_REQ )
   END_RUNG wire#w1
   // the same network as SCL:
   #CYL.RELEASE_PRESSURE_MANUAL_REQUEST := (#HMI_CMM_LINE_RELEASE_LOW AND "LTLP_HMIProInterfaceData".pMinus) OR #HMI_RELEASE_PRESSURE_MAN_REQ;
END_REGION

REGION Network 27: LOW PRESSURE MANUAL REQUEST
   RUNG wire#powerrail
      Contact( #HMI_CMM_LINE_RELEASE_LOW )
      Contact( "LTLP_HMIProInterfaceData".pPlus )
      wire#w1
      Coil( #CYL.LOW_PRESSURE_MANUAL_REQUEST )
   END_RUNG
   RUNG wire#powerrail
      Contact( #HMI_LOW_PRESSURE_MAN_REQ )
   END_RUNG wire#w1
   // the same network as SCL:
   #CYL.LOW_PRESSURE_MANUAL_REQUEST := (#HMI_CMM_LINE_RELEASE_LOW AND "LTLP_HMIProInterfaceData".pPlus) OR #HMI_LOW_PRESSURE_MAN_REQ;
END_REGION

REGION Network 28: OPERATOR HELP
   RUNG wire#powerrail
      I_Contact( #CYL.CLOSE_MANUAL_REQUEST )
      I_Contact( #CYL.OPEN_MANUAL_REQUEST )
      I_Contact( #CYL.RELEASE_PRESSURE_MANUAL_REQUEST )
      I_Contact( #CYL.LOW_PRESSURE_MANUAL_REQUEST )
      Not()
      I_Contact( "DB2001_MODES_GENERAL".GENERAL.MANUAL_SELECTED )
      { S7_GenerateENO := "TRUE" } Move(in := #DB_NUMBER, out1 => "DB440_MACHINE_ALARM_DECODING".GLOBAL_ALARMS_MACHINE.HELP_DECODING)
      S_Coil( "DB428_OPERATOR_HELP".HELP_OPERATOR_200 )
   END_RUNG
   // the same network as SCL:
   // ENO of a box is taken as its EN; it also drops when the box reports an error
   IF NOT (NOT #CYL.CLOSE_MANUAL_REQUEST AND NOT #CYL.OPEN_MANUAL_REQUEST AND NOT #CYL.RELEASE_PRESSURE_MANUAL_REQUEST AND NOT #CYL.LOW_PRESSURE_MANUAL_REQUEST) AND NOT "DB2001_MODES_GENERAL".GENERAL.MANUAL_SELECTED THEN
       "DB440_MACHINE_ALARM_DECODING".GLOBAL_ALARMS_MACHINE.HELP_DECODING := #DB_NUMBER;
       "DB428_OPERATOR_HELP".HELP_OPERATOR_200 := TRUE;
   END_IF;
END_REGION

REGION Network 29: CLOSE AUTO REQUEST
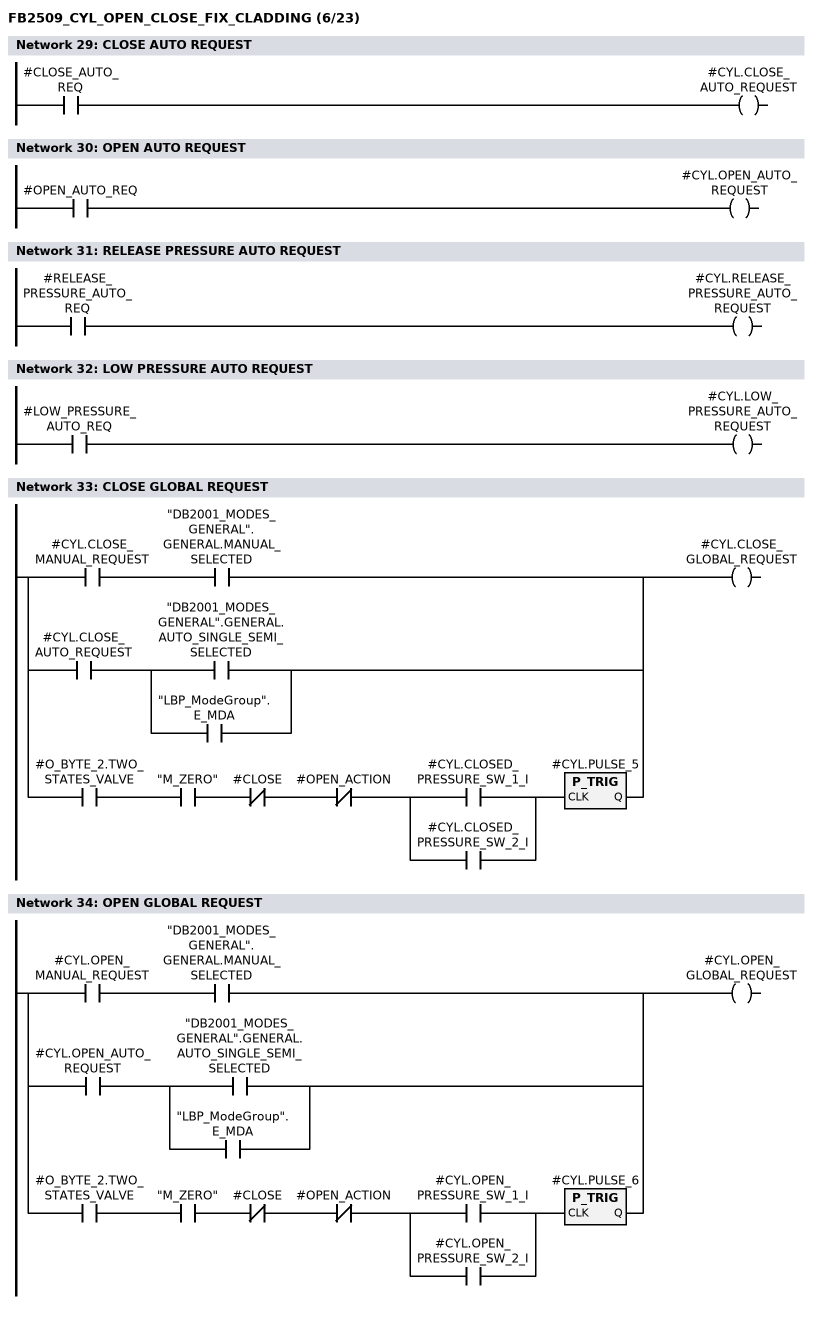
   RUNG wire#powerrail
      Contact( #CLOSE_AUTO_REQ )
      Coil( #CYL.CLOSE_AUTO_REQUEST )
   END_RUNG
   // the same network as SCL:
   #CYL.CLOSE_AUTO_REQUEST := #CLOSE_AUTO_REQ;
END_REGION

REGION Network 30: OPEN AUTO REQUEST
   RUNG wire#powerrail
      Contact( #OPEN_AUTO_REQ )
      Coil( #CYL.OPEN_AUTO_REQUEST )
   END_RUNG
   // the same network as SCL:
   #CYL.OPEN_AUTO_REQUEST := #OPEN_AUTO_REQ;
END_REGION

REGION Network 31: RELEASE PRESSURE AUTO REQUEST
   RUNG wire#powerrail
      Contact( #RELEASE_PRESSURE_AUTO_REQ )
      Coil( #CYL.RELEASE_PRESSURE_AUTO_REQUEST )
   END_RUNG
   // the same network as SCL:
   #CYL.RELEASE_PRESSURE_AUTO_REQUEST := #RELEASE_PRESSURE_AUTO_REQ;
END_REGION

REGION Network 32: LOW PRESSURE AUTO REQUEST
   RUNG wire#powerrail
      Contact( #LOW_PRESSURE_AUTO_REQ )
      Coil( #CYL.LOW_PRESSURE_AUTO_REQUEST )
   END_RUNG
   // the same network as SCL:
   #CYL.LOW_PRESSURE_AUTO_REQUEST := #LOW_PRESSURE_AUTO_REQ;
END_REGION

REGION Network 33: CLOSE GLOBAL REQUEST
   RUNG wire#powerrail
      Contact( #CYL.CLOSE_MANUAL_REQUEST )
      Contact( "DB2001_MODES_GENERAL".GENERAL.MANUAL_SELECTED )
      wire#w1
      Coil( #CYL.CLOSE_GLOBAL_REQUEST )
   END_RUNG
   RUNG wire#powerrail
      Contact( #CYL.CLOSE_AUTO_REQUEST )
      wire#w2
      Contact( "DB2001_MODES_GENERAL".GENERAL.AUTO_SINGLE_SEMI_SELECTED )
   END_RUNG wire#w1
   RUNG wire#w2
      Contact( "LBP_ModeGroup".E_MDA )
   END_RUNG wire#w1
   RUNG wire#powerrail
      Contact( #O_BYTE_2.TWO_STATES_VALVE )
      Contact( "M_ZERO" )
      I_Contact( #CLOSE )
      I_Contact( #OPEN_ACTION )
      wire#w3
      Contact( #CYL.CLOSED_PRESSURE_SW_1_I )
      wire#w4
      P_Trig( #CYL.PULSE_5 )
   END_RUNG wire#w1
   RUNG wire#w3
      Contact( #CYL.CLOSED_PRESSURE_SW_2_I )
   END_RUNG wire#w4
   // the same network as SCL:
   #_w1 := #O_BYTE_2.TWO_STATES_VALVE AND "M_ZERO" AND NOT #CLOSE AND NOT #OPEN_ACTION AND (#CYL.CLOSED_PRESSURE_SW_1_I OR #CYL.CLOSED_PRESSURE_SW_2_I);
   #_w2 := #_w1 AND NOT #CYL.PULSE_5;   // rising edge
   #CYL.PULSE_5 := #_w1;
   #CYL.CLOSE_GLOBAL_REQUEST := (#CYL.CLOSE_MANUAL_REQUEST AND "DB2001_MODES_GENERAL".GENERAL.MANUAL_SELECTED) OR (#CYL.CLOSE_AUTO_REQUEST AND ("DB2001_MODES_GENERAL".GENERAL.AUTO_SINGLE_SEMI_SELECTED OR "LBP_ModeGroup".E_MDA)) OR #_w2;
END_REGION

REGION Network 34: OPEN GLOBAL REQUEST
   RUNG wire#powerrail
      Contact( #CYL.OPEN_MANUAL_REQUEST )
      Contact( "DB2001_MODES_GENERAL".GENERAL.MANUAL_SELECTED )
      wire#w1
      Coil( #CYL.OPEN_GLOBAL_REQUEST )
   END_RUNG
   RUNG wire#powerrail
      Contact( #CYL.OPEN_AUTO_REQUEST )
      wire#w2
      Contact( "DB2001_MODES_GENERAL".GENERAL.AUTO_SINGLE_SEMI_SELECTED )
   END_RUNG wire#w1
   RUNG wire#w2
      Contact( "LBP_ModeGroup".E_MDA )
   END_RUNG wire#w1
   RUNG wire#powerrail
      Contact( #O_BYTE_2.TWO_STATES_VALVE )
      Contact( "M_ZERO" )
      I_Contact( #CLOSE )
      I_Contact( #OPEN_ACTION )
      wire#w3
      Contact( #CYL.OPEN_PRESSURE_SW_1_I )
      wire#w4
      P_Trig( #CYL.PULSE_6 )
   END_RUNG wire#w1
   RUNG wire#w3
      Contact( #CYL.OPEN_PRESSURE_SW_2_I )
   END_RUNG wire#w4
   // the same network as SCL:
   #_w1 := #O_BYTE_2.TWO_STATES_VALVE AND "M_ZERO" AND NOT #CLOSE AND NOT #OPEN_ACTION AND (#CYL.OPEN_PRESSURE_SW_1_I OR #CYL.OPEN_PRESSURE_SW_2_I);
   #_w2 := #_w1 AND NOT #CYL.PULSE_6;   // rising edge
   #CYL.PULSE_6 := #_w1;
   #CYL.OPEN_GLOBAL_REQUEST := (#CYL.OPEN_MANUAL_REQUEST AND "DB2001_MODES_GENERAL".GENERAL.MANUAL_SELECTED) OR (#CYL.OPEN_AUTO_REQUEST AND ("DB2001_MODES_GENERAL".GENERAL.AUTO_SINGLE_SEMI_SELECTED OR "LBP_ModeGroup".E_MDA)) OR #_w2;
END_REGION

REGION Network 35: RELEASE PRESSURE GLOBAL REQUEST
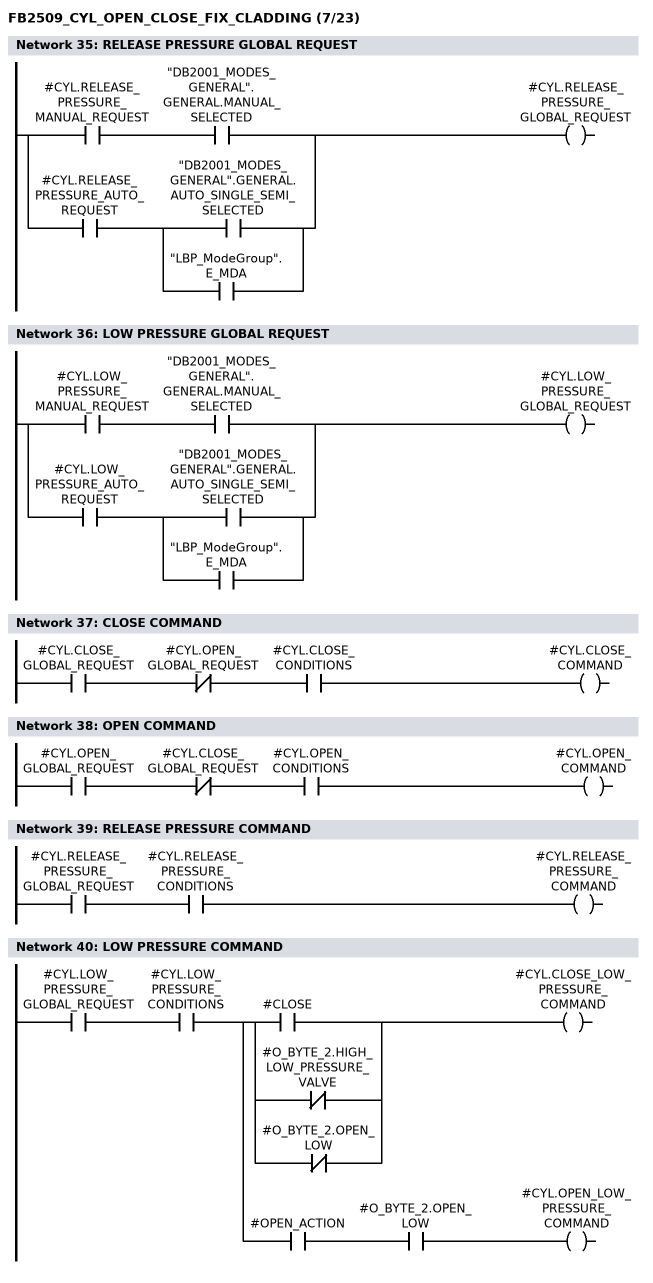
   RUNG wire#powerrail
      Contact( #CYL.RELEASE_PRESSURE_MANUAL_REQUEST )
      Contact( "DB2001_MODES_GENERAL".GENERAL.MANUAL_SELECTED )
      wire#w1
      Coil( #CYL.RELEASE_PRESSURE_GLOBAL_REQUEST )
   END_RUNG
   RUNG wire#powerrail
      Contact( #CYL.RELEASE_PRESSURE_AUTO_REQUEST )
      wire#w2
      Contact( "DB2001_MODES_GENERAL".GENERAL.AUTO_SINGLE_SEMI_SELECTED )
   END_RUNG wire#w1
   RUNG wire#w2
      Contact( "LBP_ModeGroup".E_MDA )
   END_RUNG wire#w1
   // the same network as SCL:
   #CYL.RELEASE_PRESSURE_GLOBAL_REQUEST := (#CYL.RELEASE_PRESSURE_MANUAL_REQUEST AND "DB2001_MODES_GENERAL".GENERAL.MANUAL_SELECTED) OR (#CYL.RELEASE_PRESSURE_AUTO_REQUEST AND ("DB2001_MODES_GENERAL".GENERAL.AUTO_SINGLE_SEMI_SELECTED OR "LBP_ModeGroup".E_MDA));
END_REGION

REGION Network 36: LOW PRESSURE GLOBAL REQUEST
   RUNG wire#powerrail
      Contact( #CYL.LOW_PRESSURE_MANUAL_REQUEST )
      Contact( "DB2001_MODES_GENERAL".GENERAL.MANUAL_SELECTED )
      wire#w1
      Coil( #CYL.LOW_PRESSURE_GLOBAL_REQUEST )
   END_RUNG
   RUNG wire#powerrail
      Contact( #CYL.LOW_PRESSURE_AUTO_REQUEST )
      wire#w2
      Contact( "DB2001_MODES_GENERAL".GENERAL.AUTO_SINGLE_SEMI_SELECTED )
   END_RUNG wire#w1
   RUNG wire#w2
      Contact( "LBP_ModeGroup".E_MDA )
   END_RUNG wire#w1
   // the same network as SCL:
   #CYL.LOW_PRESSURE_GLOBAL_REQUEST := (#CYL.LOW_PRESSURE_MANUAL_REQUEST AND "DB2001_MODES_GENERAL".GENERAL.MANUAL_SELECTED) OR (#CYL.LOW_PRESSURE_AUTO_REQUEST AND ("DB2001_MODES_GENERAL".GENERAL.AUTO_SINGLE_SEMI_SELECTED OR "LBP_ModeGroup".E_MDA));
END_REGION

REGION Network 37: CLOSE COMMAND
   RUNG wire#powerrail
      Contact( #CYL.CLOSE_GLOBAL_REQUEST )
      I_Contact( #CYL.OPEN_GLOBAL_REQUEST )
      Contact( #CYL.CLOSE_CONDITIONS )
      Coil( #CYL.CLOSE_COMMAND )
   END_RUNG
   // the same network as SCL:
   #CYL.CLOSE_COMMAND := #CYL.CLOSE_GLOBAL_REQUEST AND NOT #CYL.OPEN_GLOBAL_REQUEST AND #CYL.CLOSE_CONDITIONS;
END_REGION

REGION Network 38: OPEN COMMAND
   RUNG wire#powerrail
      Contact( #CYL.OPEN_GLOBAL_REQUEST )
      I_Contact( #CYL.CLOSE_GLOBAL_REQUEST )
      Contact( #CYL.OPEN_CONDITIONS )
      Coil( #CYL.OPEN_COMMAND )
   END_RUNG
   // the same network as SCL:
   #CYL.OPEN_COMMAND := #CYL.OPEN_GLOBAL_REQUEST AND NOT #CYL.CLOSE_GLOBAL_REQUEST AND #CYL.OPEN_CONDITIONS;
END_REGION

REGION Network 39: RELEASE PRESSURE COMMAND
   RUNG wire#powerrail
      Contact( #CYL.RELEASE_PRESSURE_GLOBAL_REQUEST )
      Contact( #CYL.RELEASE_PRESSURE_CONDITIONS )
      Coil( #CYL.RELEASE_PRESSURE_COMMAND )
   END_RUNG
   // the same network as SCL:
   #CYL.RELEASE_PRESSURE_COMMAND := #CYL.RELEASE_PRESSURE_GLOBAL_REQUEST AND #CYL.RELEASE_PRESSURE_CONDITIONS;
END_REGION

REGION Network 40: LOW PRESSURE COMMAND
   RUNG wire#powerrail
      Contact( #CYL.LOW_PRESSURE_GLOBAL_REQUEST )
      Contact( #CYL.LOW_PRESSURE_CONDITIONS )
      wire#w1
      Contact( #CLOSE )
      wire#w2
      Coil( #CYL.CLOSE_LOW_PRESSURE_COMMAND )
   END_RUNG
   RUNG wire#w1
      I_Contact( #O_BYTE_2.HIGH_LOW_PRESSURE_VALVE )
   END_RUNG wire#w2
   RUNG wire#w1
      I_Contact( #O_BYTE_2.OPEN_LOW )
   END_RUNG wire#w2
   RUNG wire#w1
      Contact( #OPEN_ACTION )
      Contact( #O_BYTE_2.OPEN_LOW )
      Coil( #CYL.OPEN_LOW_PRESSURE_COMMAND )
   END_RUNG
   // the same network as SCL:
   #_w1 := #CYL.LOW_PRESSURE_GLOBAL_REQUEST AND #CYL.LOW_PRESSURE_CONDITIONS;
   #CYL.CLOSE_LOW_PRESSURE_COMMAND := #_w1 AND (#CLOSE OR NOT #O_BYTE_2.HIGH_LOW_PRESSURE_VALVE OR NOT #O_BYTE_2.OPEN_LOW);
   #CYL.OPEN_LOW_PRESSURE_COMMAND := #_w1 AND #OPEN_ACTION AND #O_BYTE_2.OPEN_LOW;
END_REGION

REGION Network 41: CLOSE LOW PRESSURE
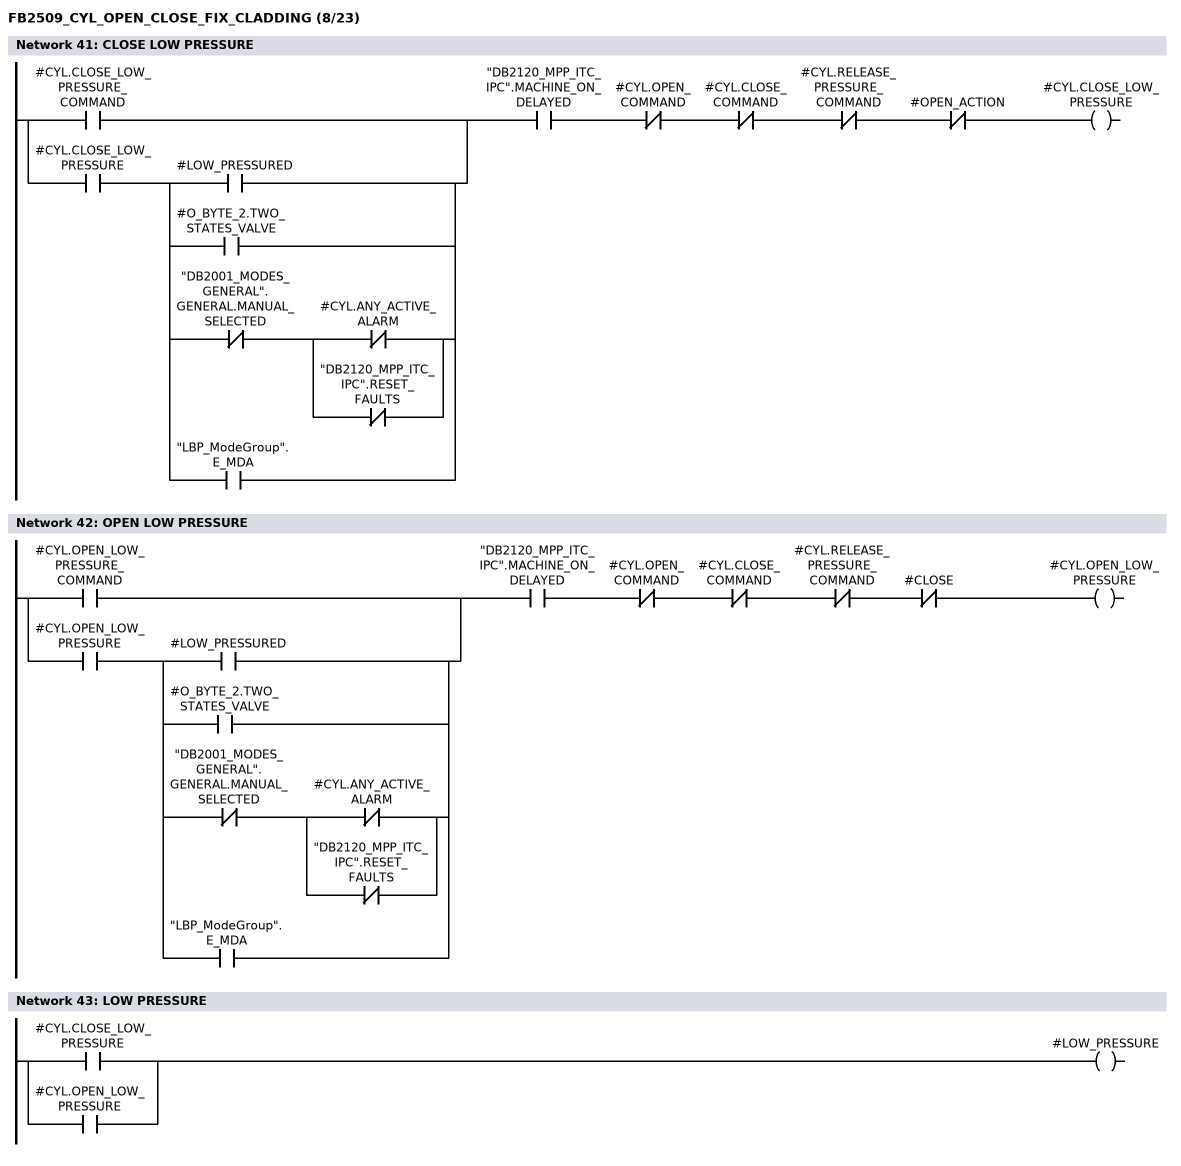
   RUNG wire#powerrail
      Contact( #CYL.CLOSE_LOW_PRESSURE_COMMAND )
      wire#w1
      Contact( "DB2120_MPP_ITC_IPC".MACHINE_ON_DELAYED )
      I_Contact( #CYL.OPEN_COMMAND )
      I_Contact( #CYL.CLOSE_COMMAND )
      I_Contact( #CYL.RELEASE_PRESSURE_COMMAND )
      I_Contact( #OPEN_ACTION )
      Coil( #CYL.CLOSE_LOW_PRESSURE )
   END_RUNG
   RUNG wire#powerrail
      Contact( #CYL.CLOSE_LOW_PRESSURE )
      wire#w2
      Contact( #LOW_PRESSURED )
   END_RUNG wire#w1
   RUNG wire#w2
      Contact( #O_BYTE_2.TWO_STATES_VALVE )
   END_RUNG wire#w1
   RUNG wire#w2
      I_Contact( "DB2001_MODES_GENERAL".GENERAL.MANUAL_SELECTED )
      wire#w3
      I_Contact( #CYL.ANY_ACTIVE_ALARM )
   END_RUNG wire#w1
   RUNG wire#w3
      I_Contact( "DB2120_MPP_ITC_IPC".RESET_FAULTS )
   END_RUNG wire#w1
   RUNG wire#w2
      Contact( "LBP_ModeGroup".E_MDA )
   END_RUNG wire#w1
   // the same network as SCL:
   #CYL.CLOSE_LOW_PRESSURE := (#CYL.CLOSE_LOW_PRESSURE_COMMAND OR (#CYL.CLOSE_LOW_PRESSURE AND (#LOW_PRESSURED OR #O_BYTE_2.TWO_STATES_VALVE OR (NOT "DB2001_MODES_GENERAL".GENERAL.MANUAL_SELECTED AND (NOT #CYL.ANY_ACTIVE_ALARM OR NOT "DB2120_MPP_ITC_IPC".RESET_FAULTS)) OR "LBP_ModeGroup".E_MDA))) AND "DB2120_MPP_ITC_IPC".MACHINE_ON_DELAYED AND NOT #CYL.OPEN_COMMAND AND NOT #CYL.CLOSE_COMMAND AND NOT #CYL.RELEASE_PRESSURE_COMMAND AND NOT #OPEN_ACTION;
END_REGION

REGION Network 42: OPEN LOW PRESSURE
   RUNG wire#powerrail
      Contact( #CYL.OPEN_LOW_PRESSURE_COMMAND )
      wire#w1
      Contact( "DB2120_MPP_ITC_IPC".MACHINE_ON_DELAYED )
      I_Contact( #CYL.OPEN_COMMAND )
      I_Contact( #CYL.CLOSE_COMMAND )
      I_Contact( #CYL.RELEASE_PRESSURE_COMMAND )
      I_Contact( #CLOSE )
      Coil( #CYL.OPEN_LOW_PRESSURE )
   END_RUNG
   RUNG wire#powerrail
      Contact( #CYL.OPEN_LOW_PRESSURE )
      wire#w2
      Contact( #LOW_PRESSURED )
   END_RUNG wire#w1
   RUNG wire#w2
      Contact( #O_BYTE_2.TWO_STATES_VALVE )
   END_RUNG wire#w1
   RUNG wire#w2
      I_Contact( "DB2001_MODES_GENERAL".GENERAL.MANUAL_SELECTED )
      wire#w3
      I_Contact( #CYL.ANY_ACTIVE_ALARM )
   END_RUNG wire#w1
   RUNG wire#w3
      I_Contact( "DB2120_MPP_ITC_IPC".RESET_FAULTS )
   END_RUNG wire#w1
   RUNG wire#w2
      Contact( "LBP_ModeGroup".E_MDA )
   END_RUNG wire#w1
   // the same network as SCL:
   #CYL.OPEN_LOW_PRESSURE := (#CYL.OPEN_LOW_PRESSURE_COMMAND OR (#CYL.OPEN_LOW_PRESSURE AND (#LOW_PRESSURED OR #O_BYTE_2.TWO_STATES_VALVE OR (NOT "DB2001_MODES_GENERAL".GENERAL.MANUAL_SELECTED AND (NOT #CYL.ANY_ACTIVE_ALARM OR NOT "DB2120_MPP_ITC_IPC".RESET_FAULTS)) OR "LBP_ModeGroup".E_MDA))) AND "DB2120_MPP_ITC_IPC".MACHINE_ON_DELAYED AND NOT #CYL.OPEN_COMMAND AND NOT #CYL.CLOSE_COMMAND AND NOT #CYL.RELEASE_PRESSURE_COMMAND AND NOT #CLOSE;
END_REGION

REGION Network 43: LOW PRESSURE
   RUNG wire#powerrail
      Contact( #CYL.CLOSE_LOW_PRESSURE )
      wire#w1
      Coil( #LOW_PRESSURE )
   END_RUNG
   RUNG wire#powerrail
      Contact( #CYL.OPEN_LOW_PRESSURE )
   END_RUNG wire#w1
   // the same network as SCL:
   #LOW_PRESSURE := #CYL.CLOSE_LOW_PRESSURE OR #CYL.OPEN_LOW_PRESSURE;
END_REGION

REGION Network 44: CLOSE
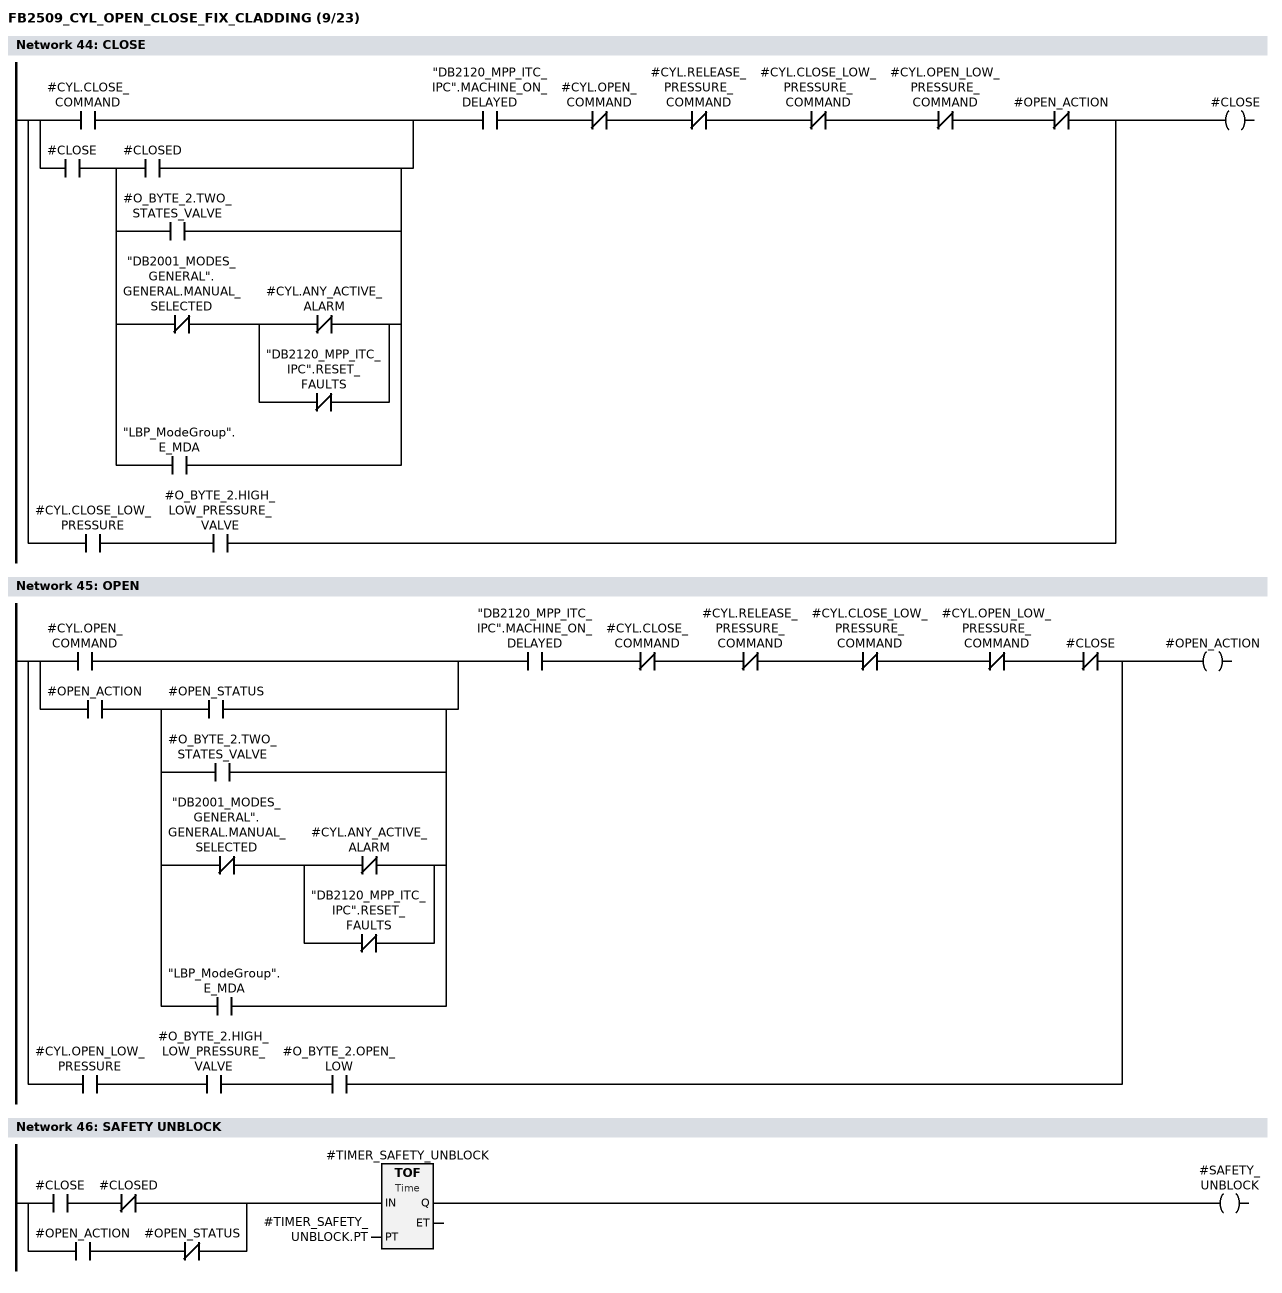
   RUNG wire#powerrail
      Contact( #CYL.CLOSE_COMMAND )
      wire#w1
      Contact( "DB2120_MPP_ITC_IPC".MACHINE_ON_DELAYED )
      I_Contact( #CYL.OPEN_COMMAND )
      I_Contact( #CYL.RELEASE_PRESSURE_COMMAND )
      I_Contact( #CYL.CLOSE_LOW_PRESSURE_COMMAND )
      I_Contact( #CYL.OPEN_LOW_PRESSURE_COMMAND )
      I_Contact( #OPEN_ACTION )
      wire#w4
      Coil( #CLOSE )
   END_RUNG
   RUNG wire#powerrail
      Contact( #CLOSE )
      wire#w2
      Contact( #CLOSED )
   END_RUNG wire#w1
   RUNG wire#w2
      Contact( #O_BYTE_2.TWO_STATES_VALVE )
   END_RUNG wire#w1
   RUNG wire#w2
      I_Contact( "DB2001_MODES_GENERAL".GENERAL.MANUAL_SELECTED )
      wire#w3
      I_Contact( #CYL.ANY_ACTIVE_ALARM )
   END_RUNG wire#w1
   RUNG wire#w3
      I_Contact( "DB2120_MPP_ITC_IPC".RESET_FAULTS )
   END_RUNG wire#w1
   RUNG wire#w2
      Contact( "LBP_ModeGroup".E_MDA )
   END_RUNG wire#w1
   RUNG wire#powerrail
      Contact( #CYL.CLOSE_LOW_PRESSURE )
      Contact( #O_BYTE_2.HIGH_LOW_PRESSURE_VALVE )
   END_RUNG wire#w4
   // the same network as SCL:
   #CLOSE := ((#CYL.CLOSE_COMMAND OR (#CLOSE AND (#CLOSED OR #O_BYTE_2.TWO_STATES_VALVE OR (NOT "DB2001_MODES_GENERAL".GENERAL.MANUAL_SELECTED AND (NOT #CYL.ANY_ACTIVE_ALARM OR NOT "DB2120_MPP_ITC_IPC".RESET_FAULTS)) OR "LBP_ModeGroup".E_MDA))) AND "DB2120_MPP_ITC_IPC".MACHINE_ON_DELAYED AND NOT #CYL.OPEN_COMMAND AND NOT #CYL.RELEASE_PRESSURE_COMMAND AND NOT #CYL.CLOSE_LOW_PRESSURE_COMMAND AND NOT #CYL.OPEN_LOW_PRESSURE_COMMAND AND NOT #OPEN_ACTION) OR (#CYL.CLOSE_LOW_PRESSURE AND #O_BYTE_2.HIGH_LOW_PRESSURE_VALVE);
END_REGION

REGION Network 45: OPEN
   RUNG wire#powerrail
      Contact( #CYL.OPEN_COMMAND )
      wire#w1
      Contact( "DB2120_MPP_ITC_IPC".MACHINE_ON_DELAYED )
      I_Contact( #CYL.CLOSE_COMMAND )
      I_Contact( #CYL.RELEASE_PRESSURE_COMMAND )
      I_Contact( #CYL.CLOSE_LOW_PRESSURE_COMMAND )
      I_Contact( #CYL.OPEN_LOW_PRESSURE_COMMAND )
      I_Contact( #CLOSE )
      wire#w4
      Coil( #OPEN_ACTION )
   END_RUNG
   RUNG wire#powerrail
      Contact( #OPEN_ACTION )
      wire#w2
      Contact( #OPEN_STATUS )
   END_RUNG wire#w1
   RUNG wire#w2
      Contact( #O_BYTE_2.TWO_STATES_VALVE )
   END_RUNG wire#w1
   RUNG wire#w2
      I_Contact( "DB2001_MODES_GENERAL".GENERAL.MANUAL_SELECTED )
      wire#w3
      I_Contact( #CYL.ANY_ACTIVE_ALARM )
   END_RUNG wire#w1
   RUNG wire#w3
      I_Contact( "DB2120_MPP_ITC_IPC".RESET_FAULTS )
   END_RUNG wire#w1
   RUNG wire#w2
      Contact( "LBP_ModeGroup".E_MDA )
   END_RUNG wire#w1
   RUNG wire#powerrail
      Contact( #CYL.OPEN_LOW_PRESSURE )
      Contact( #O_BYTE_2.HIGH_LOW_PRESSURE_VALVE )
      Contact( #O_BYTE_2.OPEN_LOW )
   END_RUNG wire#w4
   // the same network as SCL:
   #OPEN_ACTION := ((#CYL.OPEN_COMMAND OR (#OPEN_ACTION AND (#OPEN_STATUS OR #O_BYTE_2.TWO_STATES_VALVE OR (NOT "DB2001_MODES_GENERAL".GENERAL.MANUAL_SELECTED AND (NOT #CYL.ANY_ACTIVE_ALARM OR NOT "DB2120_MPP_ITC_IPC".RESET_FAULTS)) OR "LBP_ModeGroup".E_MDA))) AND "DB2120_MPP_ITC_IPC".MACHINE_ON_DELAYED AND NOT #CYL.CLOSE_COMMAND AND NOT #CYL.RELEASE_PRESSURE_COMMAND AND NOT #CYL.CLOSE_LOW_PRESSURE_COMMAND AND NOT #CYL.OPEN_LOW_PRESSURE_COMMAND AND NOT #CLOSE) OR (#CYL.OPEN_LOW_PRESSURE AND #O_BYTE_2.HIGH_LOW_PRESSURE_VALVE AND #O_BYTE_2.OPEN_LOW);
END_REGION

REGION Network 46: SAFETY UNBLOCK
   RUNG wire#powerrail
      Contact( #CLOSE )
      I_Contact( #CLOSED )
      wire#w1
      { S7_Templates := "time_type := Time" } #TIMER_SAFETY_UNBLOCK.TOF(pt := #TIMER_SAFETY_UNBLOCK.PT, et =>)
      Coil( #SAFETY_UNBLOCK )
   END_RUNG
   RUNG wire#powerrail
      Contact( #OPEN_ACTION )
      I_Contact( #OPEN_STATUS )
   END_RUNG wire#w1
   // the same network as SCL:
   #TIMER_SAFETY_UNBLOCK(IN := (#CLOSE AND NOT #CLOSED) OR (#OPEN_ACTION AND NOT #OPEN_STATUS),   // TOF
                         PT := #TIMER_SAFETY_UNBLOCK.PT);
   #SAFETY_UNBLOCK := #TIMER_SAFETY_UNBLOCK.Q;
END_REGION

REGION Network 47: PRESSURIZE
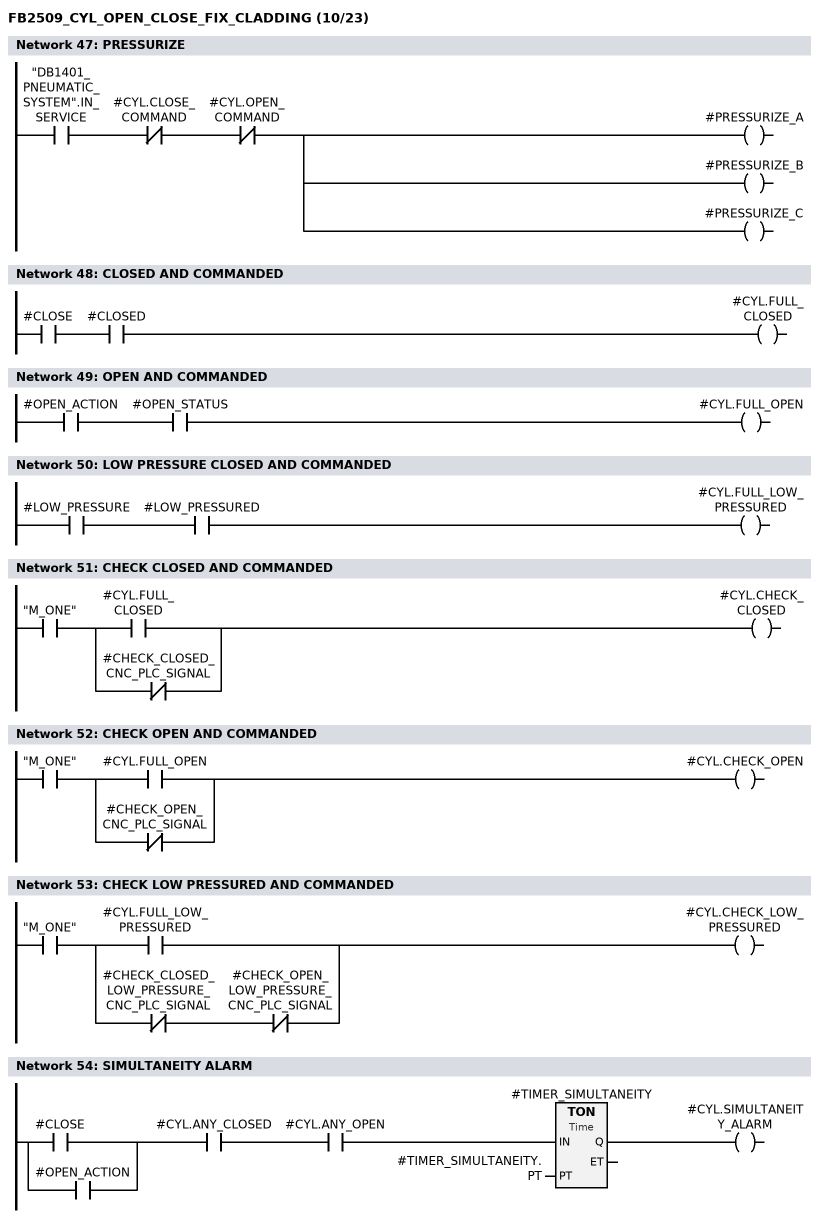
   RUNG wire#powerrail
      Contact( "DB1401_PNEUMATIC_SYSTEM".IN_SERVICE )
      I_Contact( #CYL.CLOSE_COMMAND )
      I_Contact( #CYL.OPEN_COMMAND )
      wire#w1
      Coil( #PRESSURIZE_A )
   END_RUNG
   RUNG wire#w1
      Coil( #PRESSURIZE_B )
   END_RUNG
   RUNG wire#w1
      Coil( #PRESSURIZE_C )
   END_RUNG
   // the same network as SCL:
   #PRESSURIZE_A := "DB1401_PNEUMATIC_SYSTEM".IN_SERVICE AND NOT #CYL.CLOSE_COMMAND AND NOT #CYL.OPEN_COMMAND;
   #PRESSURIZE_B := #PRESSURIZE_A;
   #PRESSURIZE_C := #PRESSURIZE_A;
END_REGION

REGION Network 48: CLOSED AND COMMANDED
   RUNG wire#powerrail
      Contact( #CLOSE )
      Contact( #CLOSED )
      Coil( #CYL.FULL_CLOSED )
   END_RUNG
   // the same network as SCL:
   #CYL.FULL_CLOSED := #CLOSE AND #CLOSED;
END_REGION

REGION Network 49: OPEN AND COMMANDED
   RUNG wire#powerrail
      Contact( #OPEN_ACTION )
      Contact( #OPEN_STATUS )
      Coil( #CYL.FULL_OPEN )
   END_RUNG
   // the same network as SCL:
   #CYL.FULL_OPEN := #OPEN_ACTION AND #OPEN_STATUS;
END_REGION

REGION Network 50: LOW PRESSURE CLOSED AND COMMANDED
   RUNG wire#powerrail
      Contact( #LOW_PRESSURE )
      Contact( #LOW_PRESSURED )
      Coil( #CYL.FULL_LOW_PRESSURED )
   END_RUNG
   // the same network as SCL:
   #CYL.FULL_LOW_PRESSURED := #LOW_PRESSURE AND #LOW_PRESSURED;
END_REGION

REGION Network 51: CHECK CLOSED AND COMMANDED
   RUNG wire#powerrail
      Contact( "M_ONE" )
      wire#w1
      Contact( #CYL.FULL_CLOSED )
      wire#w2
      Coil( #CYL.CHECK_CLOSED )
   END_RUNG
   RUNG wire#w1
      I_Contact( #CHECK_CLOSED_CNC_PLC_SIGNAL )
   END_RUNG wire#w2
   // the same network as SCL:
   #CYL.CHECK_CLOSED := "M_ONE" AND (#CYL.FULL_CLOSED OR NOT #CHECK_CLOSED_CNC_PLC_SIGNAL);
END_REGION

REGION Network 52: CHECK OPEN AND COMMANDED
   RUNG wire#powerrail
      Contact( "M_ONE" )
      wire#w1
      Contact( #CYL.FULL_OPEN )
      wire#w2
      Coil( #CYL.CHECK_OPEN )
   END_RUNG
   RUNG wire#w1
      I_Contact( #CHECK_OPEN_CNC_PLC_SIGNAL )
   END_RUNG wire#w2
   // the same network as SCL:
   #CYL.CHECK_OPEN := "M_ONE" AND (#CYL.FULL_OPEN OR NOT #CHECK_OPEN_CNC_PLC_SIGNAL);
END_REGION

REGION Network 53: CHECK LOW PRESSURED AND COMMANDED
   RUNG wire#powerrail
      Contact( "M_ONE" )
      wire#w1
      Contact( #CYL.FULL_LOW_PRESSURED )
      wire#w2
      Coil( #CYL.CHECK_LOW_PRESSURED )
   END_RUNG
   RUNG wire#w1
      I_Contact( #CHECK_CLOSED_LOW_PRESSURE_CNC_PLC_SIGNAL )
      I_Contact( #CHECK_OPEN_LOW_PRESSURE_CNC_PLC_SIGNAL )
   END_RUNG wire#w2
   // the same network as SCL:
   #CYL.CHECK_LOW_PRESSURED := "M_ONE" AND (#CYL.FULL_LOW_PRESSURED OR (NOT #CHECK_CLOSED_LOW_PRESSURE_CNC_PLC_SIGNAL AND NOT #CHECK_OPEN_LOW_PRESSURE_CNC_PLC_SIGNAL));
END_REGION

REGION Network 54: SIMULTANEITY ALARM
   RUNG wire#powerrail
      Contact( #CLOSE )
      wire#w1
      Contact( #CYL.ANY_CLOSED )
      Contact( #CYL.ANY_OPEN )
      { S7_Templates := "time_type := Time" } #TIMER_SIMULTANEITY.TON(pt := #TIMER_SIMULTANEITY.PT, et =>)
      Coil( #CYL.SIMULTANEITY_ALARM )
   END_RUNG
   RUNG wire#powerrail
      Contact( #OPEN_ACTION )
   END_RUNG wire#w1
   // the same network as SCL:
   #TIMER_SIMULTANEITY(IN := (#CLOSE OR #OPEN_ACTION) AND #CYL.ANY_CLOSED AND #CYL.ANY_OPEN,   // TON
                       PT := #TIMER_SIMULTANEITY.PT);
   #CYL.SIMULTANEITY_ALARM := #TIMER_SIMULTANEITY.Q;
END_REGION

REGION Network 55: TIME EXCEEDED ALARM
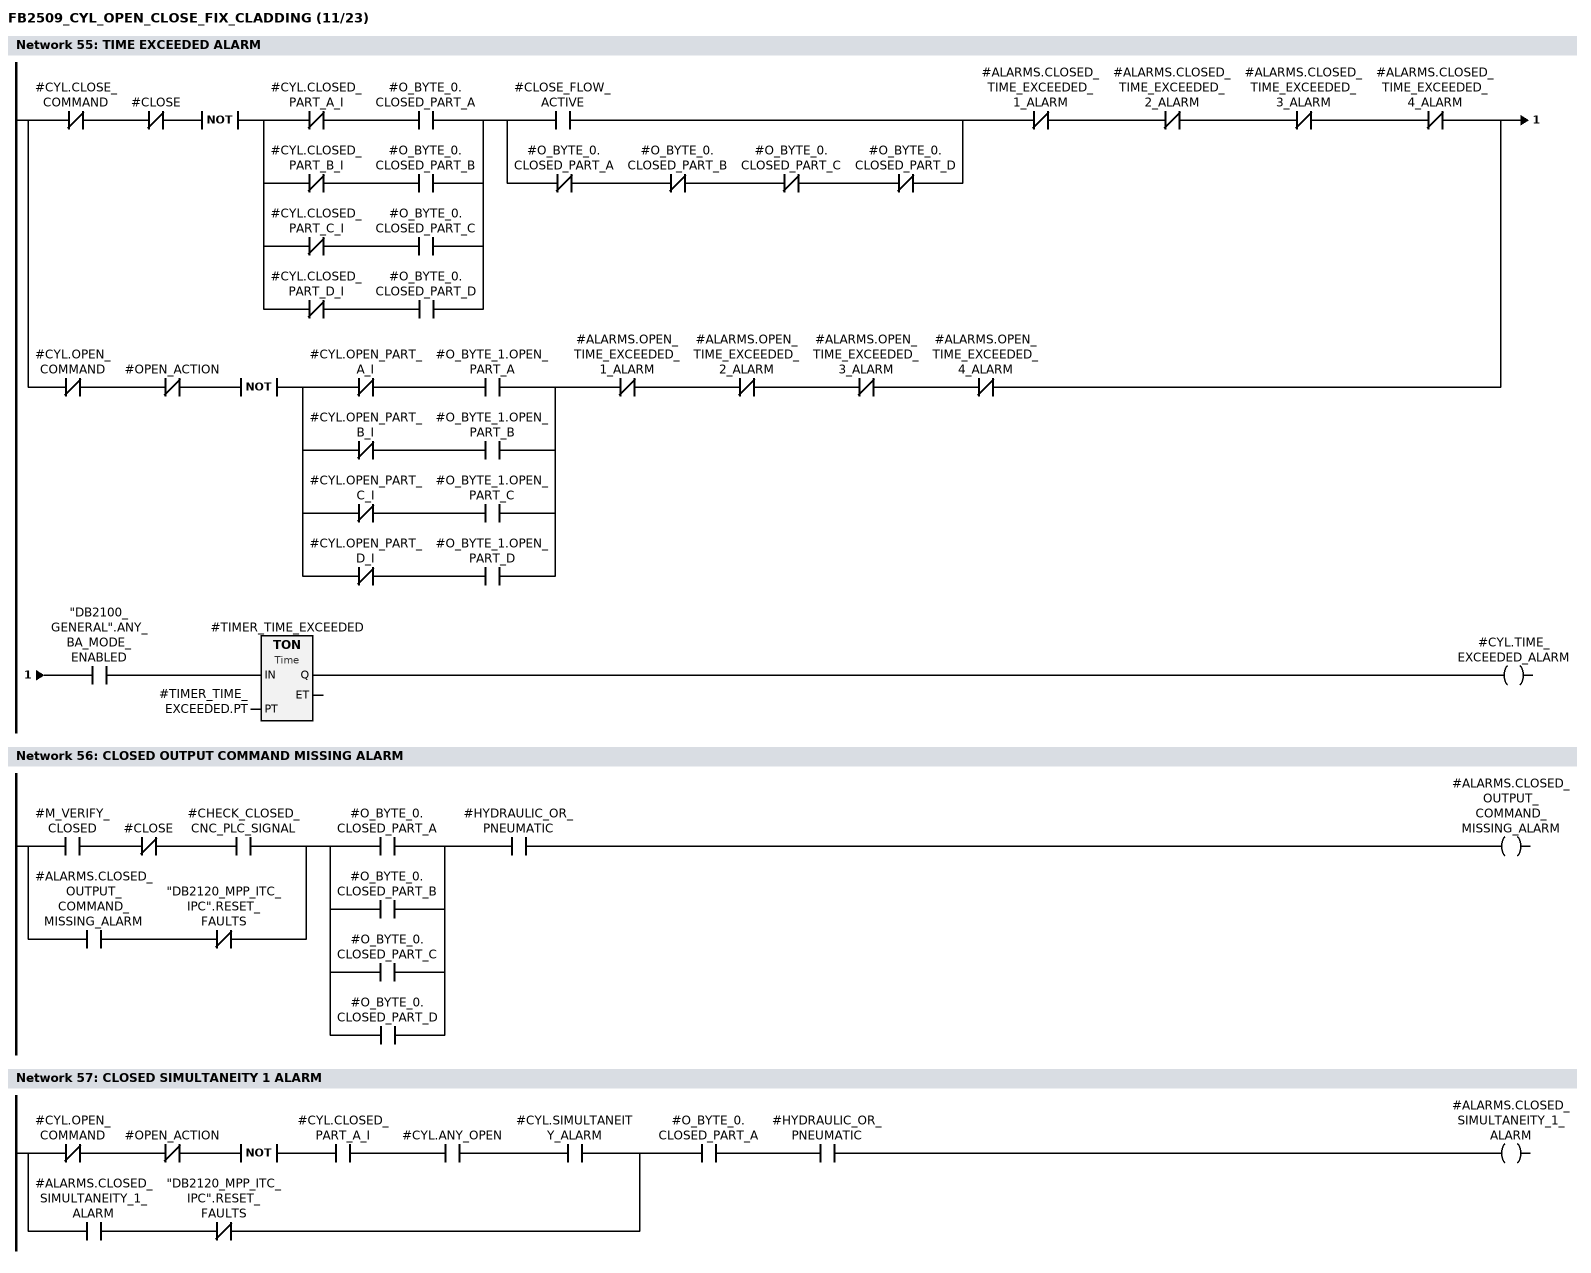
   RUNG wire#powerrail
      I_Contact( #CYL.CLOSE_COMMAND )
      I_Contact( #CLOSE )
      Not()
      wire#w1
      I_Contact( #CYL.CLOSED_PART_A_I )
      Contact( #O_BYTE_0.CLOSED_PART_A )
      wire#w2
      Contact( #CLOSE_FLOW_ACTIVE )
      wire#w3
      I_Contact( #ALARMS.CLOSED_TIME_EXCEEDED_1_ALARM )
      I_Contact( #ALARMS.CLOSED_TIME_EXCEEDED_2_ALARM )
      I_Contact( #ALARMS.CLOSED_TIME_EXCEEDED_3_ALARM )
      I_Contact( #ALARMS.CLOSED_TIME_EXCEEDED_4_ALARM )
      wire#w4
      Contact( "DB2100_GENERAL".ANY_BA_MODE_ENABLED )
      { S7_Templates := "time_type := Time" } #TIMER_TIME_EXCEEDED.TON(pt := #TIMER_TIME_EXCEEDED.PT, et =>)
      Coil( #CYL.TIME_EXCEEDED_ALARM )
   END_RUNG
   RUNG wire#w1
      I_Contact( #CYL.CLOSED_PART_B_I )
      Contact( #O_BYTE_0.CLOSED_PART_B )
   END_RUNG wire#w2
   RUNG wire#w1
      I_Contact( #CYL.CLOSED_PART_C_I )
      Contact( #O_BYTE_0.CLOSED_PART_C )
   END_RUNG wire#w2
   RUNG wire#w1
      I_Contact( #CYL.CLOSED_PART_D_I )
      Contact( #O_BYTE_0.CLOSED_PART_D )
   END_RUNG wire#w2
   RUNG wire#w2
      I_Contact( #O_BYTE_0.CLOSED_PART_A )
      I_Contact( #O_BYTE_0.CLOSED_PART_B )
      I_Contact( #O_BYTE_0.CLOSED_PART_C )
      I_Contact( #O_BYTE_0.CLOSED_PART_D )
   END_RUNG wire#w3
   RUNG wire#powerrail
      I_Contact( #CYL.OPEN_COMMAND )
      I_Contact( #OPEN_ACTION )
      Not()
      wire#w5
      I_Contact( #CYL.OPEN_PART_A_I )
      Contact( #O_BYTE_1.OPEN_PART_A )
      wire#w6
      I_Contact( #ALARMS.OPEN_TIME_EXCEEDED_1_ALARM )
      I_Contact( #ALARMS.OPEN_TIME_EXCEEDED_2_ALARM )
      I_Contact( #ALARMS.OPEN_TIME_EXCEEDED_3_ALARM )
      I_Contact( #ALARMS.OPEN_TIME_EXCEEDED_4_ALARM )
   END_RUNG wire#w4
   RUNG wire#w5
      I_Contact( #CYL.OPEN_PART_B_I )
      Contact( #O_BYTE_1.OPEN_PART_B )
   END_RUNG wire#w6
   RUNG wire#w5
      I_Contact( #CYL.OPEN_PART_C_I )
      Contact( #O_BYTE_1.OPEN_PART_C )
   END_RUNG wire#w6
   RUNG wire#w5
      I_Contact( #CYL.OPEN_PART_D_I )
      Contact( #O_BYTE_1.OPEN_PART_D )
   END_RUNG wire#w6
   // the same network as SCL:
   #TIMER_TIME_EXCEEDED(IN := ((NOT (NOT #CYL.CLOSE_COMMAND AND NOT #CLOSE) AND ((NOT #CYL.CLOSED_PART_A_I AND #O_BYTE_0.CLOSED_PART_A) OR (NOT #CYL.CLOSED_PART_B_I AND #O_BYTE_0.CLOSED_PART_B) OR (NOT #CYL.CLOSED_PART_C_I AND #O_BYTE_0.CLOSED_PART_C) OR (NOT #CYL.CLOSED_PART_D_I AND #O_BYTE_0.CLOSED_PART_D)) AND (#CLOSE_FLOW_ACTIVE OR (NOT #O_BYTE_0.CLOSED_PART_A AND NOT #O_BYTE_0.CLOSED_PART_B AND NOT #O_BYTE_0.CLOSED_PART_C AND NOT #O_BYTE_0.CLOSED_PART_D)) AND NOT #ALARMS.CLOSED_TIME_EXCEEDED_1_ALARM AND NOT #ALARMS.CLOSED_TIME_EXCEEDED_2_ALARM AND NOT #ALARMS.CLOSED_TIME_EXCEEDED_3_ALARM AND NOT #ALARMS.CLOSED_TIME_EXCEEDED_4_ALARM) OR (NOT (NOT #CYL.OPEN_COMMAND AND NOT #OPEN_ACTION) AND ((NOT #CYL.OPEN_PART_A_I AND #O_BYTE_1.OPEN_PART_A) OR (NOT #CYL.OPEN_PART_B_I AND #O_BYTE_1.OPEN_PART_B) OR (NOT #CYL.OPEN_PART_C_I AND #O_BYTE_1.OPEN_PART_C) OR (NOT #CYL.OPEN_PART_D_I AND #O_BYTE_1.OPEN_PART_D)) AND NOT #ALARMS.OPEN_TIME_EXCEEDED_1_ALARM AND NOT #ALARMS.OPEN_TIME_EXCEEDED_2_ALARM AND NOT #ALARMS.OPEN_TIME_EXCEEDED_3_ALARM AND NOT #ALARMS.OPEN_TIME_EXCEEDED_4_ALARM)) AND "DB2100_GENERAL".ANY_BA_MODE_ENABLED,   // TON
                        PT := #TIMER_TIME_EXCEEDED.PT);
   #CYL.TIME_EXCEEDED_ALARM := #TIMER_TIME_EXCEEDED.Q;
END_REGION

REGION Network 56: CLOSED OUTPUT COMMAND MISSING ALARM
   RUNG wire#powerrail
      Contact( #M_VERIFY_CLOSED )
      I_Contact( #CLOSE )
      Contact( #CHECK_CLOSED_CNC_PLC_SIGNAL )
      wire#w1
      Contact( #O_BYTE_0.CLOSED_PART_A )
      wire#w2
      Contact( #HYDRAULIC_OR_PNEUMATIC )
      Coil( #ALARMS.CLOSED_OUTPUT_COMMAND_MISSING_ALARM )
   END_RUNG
   RUNG wire#powerrail
      Contact( #ALARMS.CLOSED_OUTPUT_COMMAND_MISSING_ALARM )
      I_Contact( "DB2120_MPP_ITC_IPC".RESET_FAULTS )
   END_RUNG wire#w1
   RUNG wire#w1
      Contact( #O_BYTE_0.CLOSED_PART_B )
   END_RUNG wire#w2
   RUNG wire#w1
      Contact( #O_BYTE_0.CLOSED_PART_C )
   END_RUNG wire#w2
   RUNG wire#w1
      Contact( #O_BYTE_0.CLOSED_PART_D )
   END_RUNG wire#w2
   // the same network as SCL:
   #ALARMS.CLOSED_OUTPUT_COMMAND_MISSING_ALARM := ((#M_VERIFY_CLOSED AND NOT #CLOSE AND #CHECK_CLOSED_CNC_PLC_SIGNAL) OR (#ALARMS.CLOSED_OUTPUT_COMMAND_MISSING_ALARM AND NOT "DB2120_MPP_ITC_IPC".RESET_FAULTS)) AND (#O_BYTE_0.CLOSED_PART_A OR #O_BYTE_0.CLOSED_PART_B OR #O_BYTE_0.CLOSED_PART_C OR #O_BYTE_0.CLOSED_PART_D) AND #HYDRAULIC_OR_PNEUMATIC;
END_REGION

REGION Network 57: CLOSED SIMULTANEITY 1 ALARM
   RUNG wire#powerrail
      I_Contact( #CYL.OPEN_COMMAND )
      I_Contact( #OPEN_ACTION )
      Not()
      Contact( #CYL.CLOSED_PART_A_I )
      Contact( #CYL.ANY_OPEN )
      Contact( #CYL.SIMULTANEITY_ALARM )
      wire#w1
      Contact( #O_BYTE_0.CLOSED_PART_A )
      Contact( #HYDRAULIC_OR_PNEUMATIC )
      Coil( #ALARMS.CLOSED_SIMULTANEITY_1_ALARM )
   END_RUNG
   RUNG wire#powerrail
      Contact( #ALARMS.CLOSED_SIMULTANEITY_1_ALARM )
      I_Contact( "DB2120_MPP_ITC_IPC".RESET_FAULTS )
   END_RUNG wire#w1
   // the same network as SCL:
   #ALARMS.CLOSED_SIMULTANEITY_1_ALARM := ((NOT (NOT #CYL.OPEN_COMMAND AND NOT #OPEN_ACTION) AND #CYL.CLOSED_PART_A_I AND #CYL.ANY_OPEN AND #CYL.SIMULTANEITY_ALARM) OR (#ALARMS.CLOSED_SIMULTANEITY_1_ALARM AND NOT "DB2120_MPP_ITC_IPC".RESET_FAULTS)) AND #O_BYTE_0.CLOSED_PART_A AND #HYDRAULIC_OR_PNEUMATIC;
END_REGION

REGION Network 58: CLOSED TIME EXCEEDED 1 ALARM
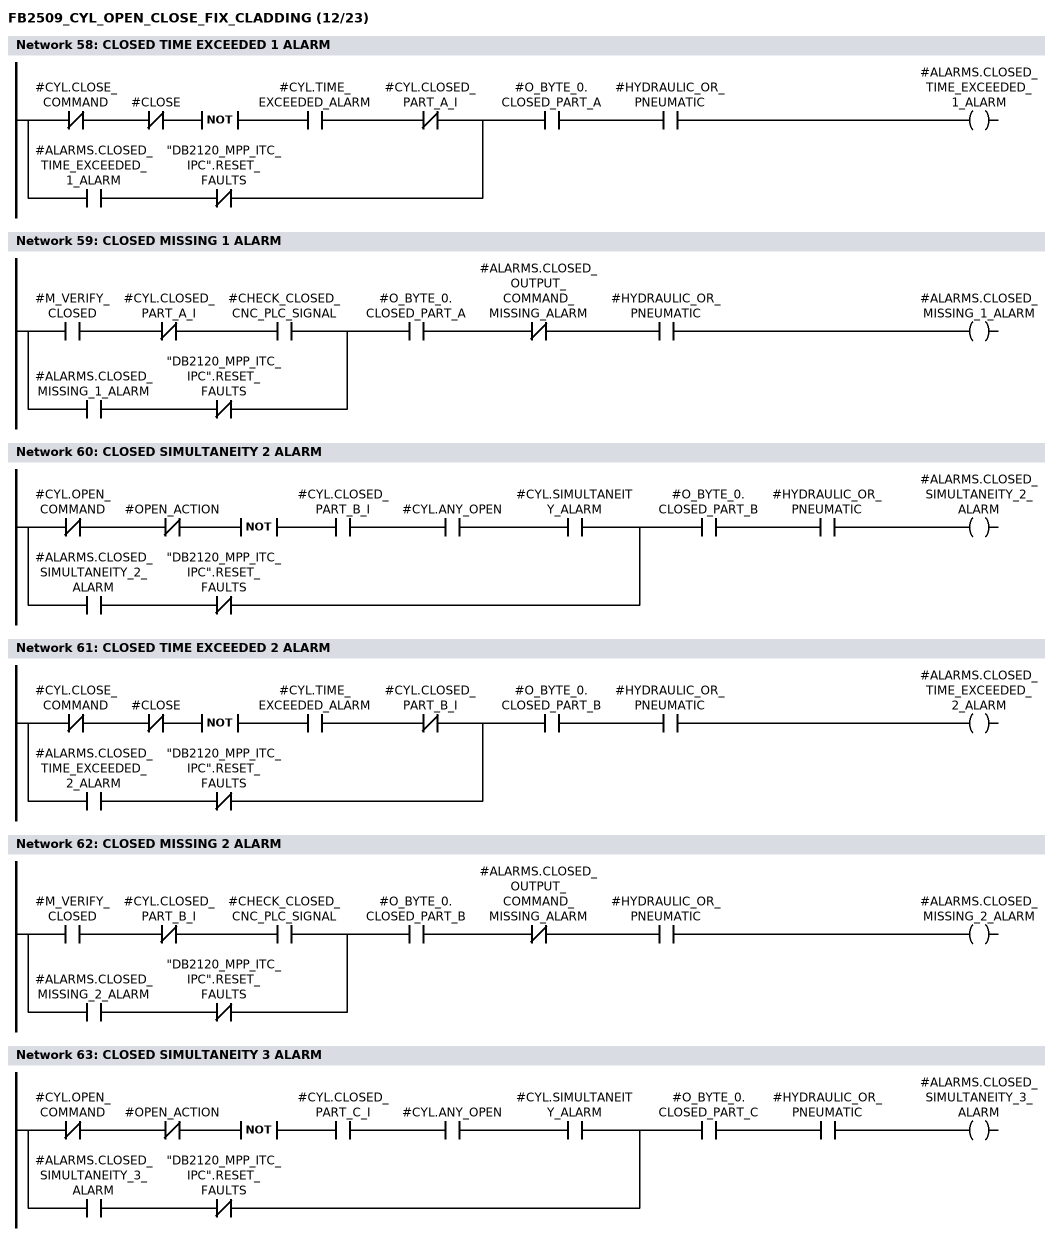
   RUNG wire#powerrail
      I_Contact( #CYL.CLOSE_COMMAND )
      I_Contact( #CLOSE )
      Not()
      Contact( #CYL.TIME_EXCEEDED_ALARM )
      I_Contact( #CYL.CLOSED_PART_A_I )
      wire#w1
      Contact( #O_BYTE_0.CLOSED_PART_A )
      Contact( #HYDRAULIC_OR_PNEUMATIC )
      Coil( #ALARMS.CLOSED_TIME_EXCEEDED_1_ALARM )
   END_RUNG
   RUNG wire#powerrail
      Contact( #ALARMS.CLOSED_TIME_EXCEEDED_1_ALARM )
      I_Contact( "DB2120_MPP_ITC_IPC".RESET_FAULTS )
   END_RUNG wire#w1
   // the same network as SCL:
   #ALARMS.CLOSED_TIME_EXCEEDED_1_ALARM := ((NOT (NOT #CYL.CLOSE_COMMAND AND NOT #CLOSE) AND #CYL.TIME_EXCEEDED_ALARM AND NOT #CYL.CLOSED_PART_A_I) OR (#ALARMS.CLOSED_TIME_EXCEEDED_1_ALARM AND NOT "DB2120_MPP_ITC_IPC".RESET_FAULTS)) AND #O_BYTE_0.CLOSED_PART_A AND #HYDRAULIC_OR_PNEUMATIC;
END_REGION

REGION Network 59: CLOSED MISSING 1 ALARM
   RUNG wire#powerrail
      Contact( #M_VERIFY_CLOSED )
      I_Contact( #CYL.CLOSED_PART_A_I )
      Contact( #CHECK_CLOSED_CNC_PLC_SIGNAL )
      wire#w1
      Contact( #O_BYTE_0.CLOSED_PART_A )
      I_Contact( #ALARMS.CLOSED_OUTPUT_COMMAND_MISSING_ALARM )
      Contact( #HYDRAULIC_OR_PNEUMATIC )
      Coil( #ALARMS.CLOSED_MISSING_1_ALARM )
   END_RUNG
   RUNG wire#powerrail
      Contact( #ALARMS.CLOSED_MISSING_1_ALARM )
      I_Contact( "DB2120_MPP_ITC_IPC".RESET_FAULTS )
   END_RUNG wire#w1
   // the same network as SCL:
   #ALARMS.CLOSED_MISSING_1_ALARM := ((#M_VERIFY_CLOSED AND NOT #CYL.CLOSED_PART_A_I AND #CHECK_CLOSED_CNC_PLC_SIGNAL) OR (#ALARMS.CLOSED_MISSING_1_ALARM AND NOT "DB2120_MPP_ITC_IPC".RESET_FAULTS)) AND #O_BYTE_0.CLOSED_PART_A AND NOT #ALARMS.CLOSED_OUTPUT_COMMAND_MISSING_ALARM AND #HYDRAULIC_OR_PNEUMATIC;
END_REGION

REGION Network 60: CLOSED SIMULTANEITY 2 ALARM
   RUNG wire#powerrail
      I_Contact( #CYL.OPEN_COMMAND )
      I_Contact( #OPEN_ACTION )
      Not()
      Contact( #CYL.CLOSED_PART_B_I )
      Contact( #CYL.ANY_OPEN )
      Contact( #CYL.SIMULTANEITY_ALARM )
      wire#w1
      Contact( #O_BYTE_0.CLOSED_PART_B )
      Contact( #HYDRAULIC_OR_PNEUMATIC )
      Coil( #ALARMS.CLOSED_SIMULTANEITY_2_ALARM )
   END_RUNG
   RUNG wire#powerrail
      Contact( #ALARMS.CLOSED_SIMULTANEITY_2_ALARM )
      I_Contact( "DB2120_MPP_ITC_IPC".RESET_FAULTS )
   END_RUNG wire#w1
   // the same network as SCL:
   #ALARMS.CLOSED_SIMULTANEITY_2_ALARM := ((NOT (NOT #CYL.OPEN_COMMAND AND NOT #OPEN_ACTION) AND #CYL.CLOSED_PART_B_I AND #CYL.ANY_OPEN AND #CYL.SIMULTANEITY_ALARM) OR (#ALARMS.CLOSED_SIMULTANEITY_2_ALARM AND NOT "DB2120_MPP_ITC_IPC".RESET_FAULTS)) AND #O_BYTE_0.CLOSED_PART_B AND #HYDRAULIC_OR_PNEUMATIC;
END_REGION

REGION Network 61: CLOSED TIME EXCEEDED 2 ALARM
   RUNG wire#powerrail
      I_Contact( #CYL.CLOSE_COMMAND )
      I_Contact( #CLOSE )
      Not()
      Contact( #CYL.TIME_EXCEEDED_ALARM )
      I_Contact( #CYL.CLOSED_PART_B_I )
      wire#w1
      Contact( #O_BYTE_0.CLOSED_PART_B )
      Contact( #HYDRAULIC_OR_PNEUMATIC )
      Coil( #ALARMS.CLOSED_TIME_EXCEEDED_2_ALARM )
   END_RUNG
   RUNG wire#powerrail
      Contact( #ALARMS.CLOSED_TIME_EXCEEDED_2_ALARM )
      I_Contact( "DB2120_MPP_ITC_IPC".RESET_FAULTS )
   END_RUNG wire#w1
   // the same network as SCL:
   #ALARMS.CLOSED_TIME_EXCEEDED_2_ALARM := ((NOT (NOT #CYL.CLOSE_COMMAND AND NOT #CLOSE) AND #CYL.TIME_EXCEEDED_ALARM AND NOT #CYL.CLOSED_PART_B_I) OR (#ALARMS.CLOSED_TIME_EXCEEDED_2_ALARM AND NOT "DB2120_MPP_ITC_IPC".RESET_FAULTS)) AND #O_BYTE_0.CLOSED_PART_B AND #HYDRAULIC_OR_PNEUMATIC;
END_REGION

REGION Network 62: CLOSED MISSING 2 ALARM
   RUNG wire#powerrail
      Contact( #M_VERIFY_CLOSED )
      I_Contact( #CYL.CLOSED_PART_B_I )
      Contact( #CHECK_CLOSED_CNC_PLC_SIGNAL )
      wire#w1
      Contact( #O_BYTE_0.CLOSED_PART_B )
      I_Contact( #ALARMS.CLOSED_OUTPUT_COMMAND_MISSING_ALARM )
      Contact( #HYDRAULIC_OR_PNEUMATIC )
      Coil( #ALARMS.CLOSED_MISSING_2_ALARM )
   END_RUNG
   RUNG wire#powerrail
      Contact( #ALARMS.CLOSED_MISSING_2_ALARM )
      I_Contact( "DB2120_MPP_ITC_IPC".RESET_FAULTS )
   END_RUNG wire#w1
   // the same network as SCL:
   #ALARMS.CLOSED_MISSING_2_ALARM := ((#M_VERIFY_CLOSED AND NOT #CYL.CLOSED_PART_B_I AND #CHECK_CLOSED_CNC_PLC_SIGNAL) OR (#ALARMS.CLOSED_MISSING_2_ALARM AND NOT "DB2120_MPP_ITC_IPC".RESET_FAULTS)) AND #O_BYTE_0.CLOSED_PART_B AND NOT #ALARMS.CLOSED_OUTPUT_COMMAND_MISSING_ALARM AND #HYDRAULIC_OR_PNEUMATIC;
END_REGION

REGION Network 63: CLOSED SIMULTANEITY 3 ALARM
   RUNG wire#powerrail
      I_Contact( #CYL.OPEN_COMMAND )
      I_Contact( #OPEN_ACTION )
      Not()
      Contact( #CYL.CLOSED_PART_C_I )
      Contact( #CYL.ANY_OPEN )
      Contact( #CYL.SIMULTANEITY_ALARM )
      wire#w1
      Contact( #O_BYTE_0.CLOSED_PART_C )
      Contact( #HYDRAULIC_OR_PNEUMATIC )
      Coil( #ALARMS.CLOSED_SIMULTANEITY_3_ALARM )
   END_RUNG
   RUNG wire#powerrail
      Contact( #ALARMS.CLOSED_SIMULTANEITY_3_ALARM )
      I_Contact( "DB2120_MPP_ITC_IPC".RESET_FAULTS )
   END_RUNG wire#w1
   // the same network as SCL:
   #ALARMS.CLOSED_SIMULTANEITY_3_ALARM := ((NOT (NOT #CYL.OPEN_COMMAND AND NOT #OPEN_ACTION) AND #CYL.CLOSED_PART_C_I AND #CYL.ANY_OPEN AND #CYL.SIMULTANEITY_ALARM) OR (#ALARMS.CLOSED_SIMULTANEITY_3_ALARM AND NOT "DB2120_MPP_ITC_IPC".RESET_FAULTS)) AND #O_BYTE_0.CLOSED_PART_C AND #HYDRAULIC_OR_PNEUMATIC;
END_REGION

REGION Network 64: CLOSED TIME EXCEEDED 3 ALARM
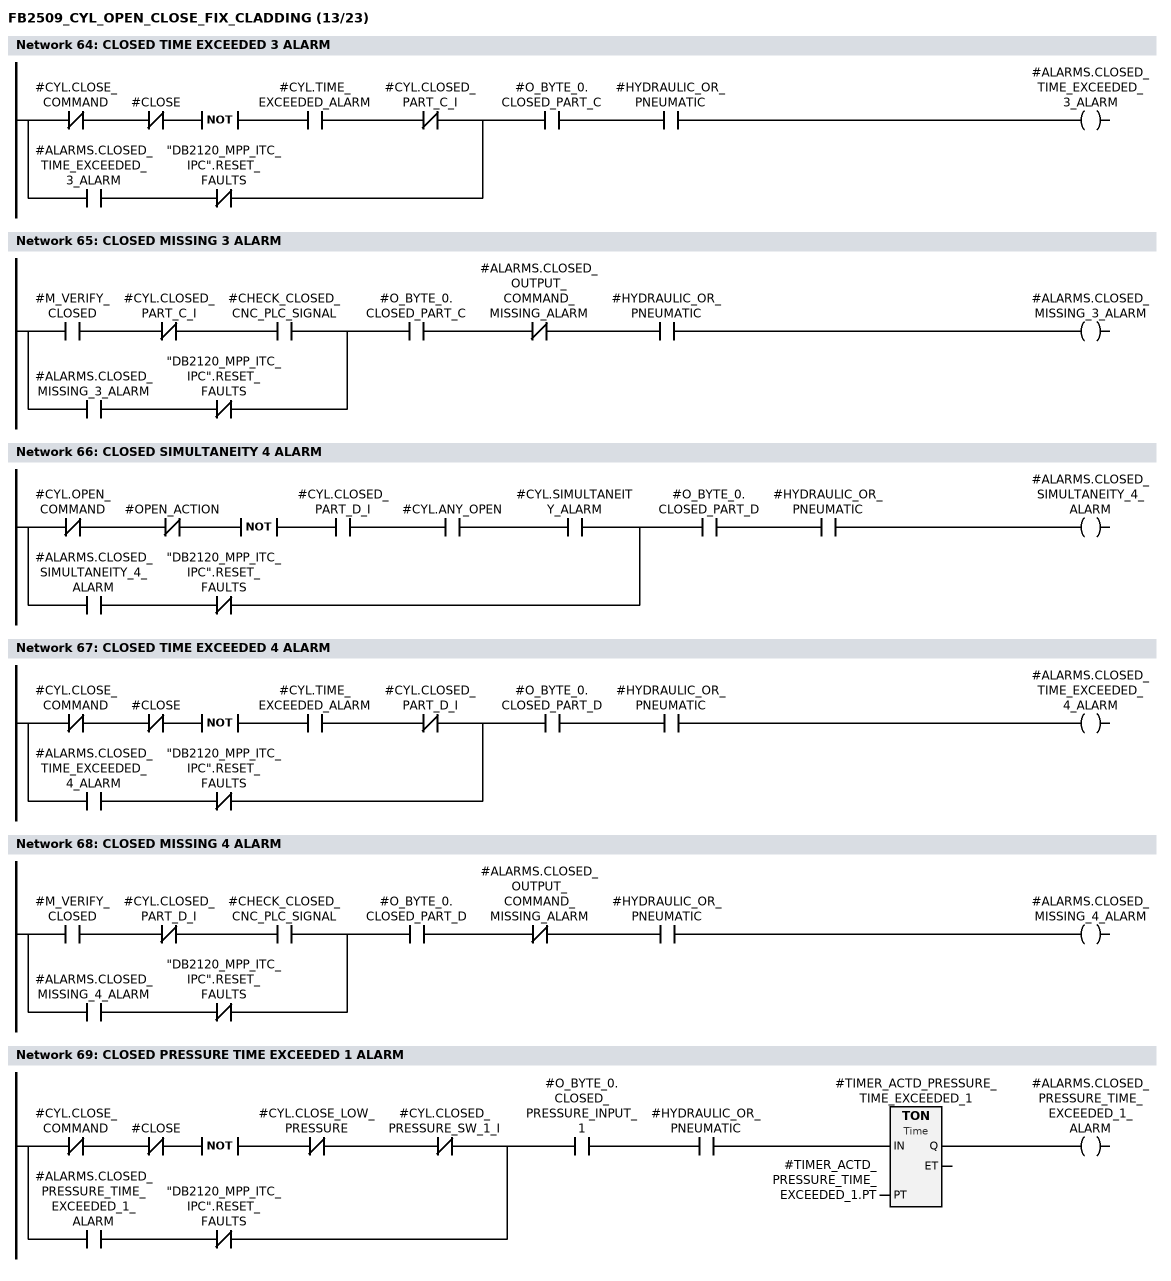
   RUNG wire#powerrail
      I_Contact( #CYL.CLOSE_COMMAND )
      I_Contact( #CLOSE )
      Not()
      Contact( #CYL.TIME_EXCEEDED_ALARM )
      I_Contact( #CYL.CLOSED_PART_C_I )
      wire#w1
      Contact( #O_BYTE_0.CLOSED_PART_C )
      Contact( #HYDRAULIC_OR_PNEUMATIC )
      Coil( #ALARMS.CLOSED_TIME_EXCEEDED_3_ALARM )
   END_RUNG
   RUNG wire#powerrail
      Contact( #ALARMS.CLOSED_TIME_EXCEEDED_3_ALARM )
      I_Contact( "DB2120_MPP_ITC_IPC".RESET_FAULTS )
   END_RUNG wire#w1
   // the same network as SCL:
   #ALARMS.CLOSED_TIME_EXCEEDED_3_ALARM := ((NOT (NOT #CYL.CLOSE_COMMAND AND NOT #CLOSE) AND #CYL.TIME_EXCEEDED_ALARM AND NOT #CYL.CLOSED_PART_C_I) OR (#ALARMS.CLOSED_TIME_EXCEEDED_3_ALARM AND NOT "DB2120_MPP_ITC_IPC".RESET_FAULTS)) AND #O_BYTE_0.CLOSED_PART_C AND #HYDRAULIC_OR_PNEUMATIC;
END_REGION

REGION Network 65: CLOSED MISSING 3 ALARM
   RUNG wire#powerrail
      Contact( #M_VERIFY_CLOSED )
      I_Contact( #CYL.CLOSED_PART_C_I )
      Contact( #CHECK_CLOSED_CNC_PLC_SIGNAL )
      wire#w1
      Contact( #O_BYTE_0.CLOSED_PART_C )
      I_Contact( #ALARMS.CLOSED_OUTPUT_COMMAND_MISSING_ALARM )
      Contact( #HYDRAULIC_OR_PNEUMATIC )
      Coil( #ALARMS.CLOSED_MISSING_3_ALARM )
   END_RUNG
   RUNG wire#powerrail
      Contact( #ALARMS.CLOSED_MISSING_3_ALARM )
      I_Contact( "DB2120_MPP_ITC_IPC".RESET_FAULTS )
   END_RUNG wire#w1
   // the same network as SCL:
   #ALARMS.CLOSED_MISSING_3_ALARM := ((#M_VERIFY_CLOSED AND NOT #CYL.CLOSED_PART_C_I AND #CHECK_CLOSED_CNC_PLC_SIGNAL) OR (#ALARMS.CLOSED_MISSING_3_ALARM AND NOT "DB2120_MPP_ITC_IPC".RESET_FAULTS)) AND #O_BYTE_0.CLOSED_PART_C AND NOT #ALARMS.CLOSED_OUTPUT_COMMAND_MISSING_ALARM AND #HYDRAULIC_OR_PNEUMATIC;
END_REGION

REGION Network 66: CLOSED SIMULTANEITY 4 ALARM
   RUNG wire#powerrail
      I_Contact( #CYL.OPEN_COMMAND )
      I_Contact( #OPEN_ACTION )
      Not()
      Contact( #CYL.CLOSED_PART_D_I )
      Contact( #CYL.ANY_OPEN )
      Contact( #CYL.SIMULTANEITY_ALARM )
      wire#w1
      Contact( #O_BYTE_0.CLOSED_PART_D )
      Contact( #HYDRAULIC_OR_PNEUMATIC )
      Coil( #ALARMS.CLOSED_SIMULTANEITY_4_ALARM )
   END_RUNG
   RUNG wire#powerrail
      Contact( #ALARMS.CLOSED_SIMULTANEITY_4_ALARM )
      I_Contact( "DB2120_MPP_ITC_IPC".RESET_FAULTS )
   END_RUNG wire#w1
   // the same network as SCL:
   #ALARMS.CLOSED_SIMULTANEITY_4_ALARM := ((NOT (NOT #CYL.OPEN_COMMAND AND NOT #OPEN_ACTION) AND #CYL.CLOSED_PART_D_I AND #CYL.ANY_OPEN AND #CYL.SIMULTANEITY_ALARM) OR (#ALARMS.CLOSED_SIMULTANEITY_4_ALARM AND NOT "DB2120_MPP_ITC_IPC".RESET_FAULTS)) AND #O_BYTE_0.CLOSED_PART_D AND #HYDRAULIC_OR_PNEUMATIC;
END_REGION

REGION Network 67: CLOSED TIME EXCEEDED 4 ALARM
   RUNG wire#powerrail
      I_Contact( #CYL.CLOSE_COMMAND )
      I_Contact( #CLOSE )
      Not()
      Contact( #CYL.TIME_EXCEEDED_ALARM )
      I_Contact( #CYL.CLOSED_PART_D_I )
      wire#w1
      Contact( #O_BYTE_0.CLOSED_PART_D )
      Contact( #HYDRAULIC_OR_PNEUMATIC )
      Coil( #ALARMS.CLOSED_TIME_EXCEEDED_4_ALARM )
   END_RUNG
   RUNG wire#powerrail
      Contact( #ALARMS.CLOSED_TIME_EXCEEDED_4_ALARM )
      I_Contact( "DB2120_MPP_ITC_IPC".RESET_FAULTS )
   END_RUNG wire#w1
   // the same network as SCL:
   #ALARMS.CLOSED_TIME_EXCEEDED_4_ALARM := ((NOT (NOT #CYL.CLOSE_COMMAND AND NOT #CLOSE) AND #CYL.TIME_EXCEEDED_ALARM AND NOT #CYL.CLOSED_PART_D_I) OR (#ALARMS.CLOSED_TIME_EXCEEDED_4_ALARM AND NOT "DB2120_MPP_ITC_IPC".RESET_FAULTS)) AND #O_BYTE_0.CLOSED_PART_D AND #HYDRAULIC_OR_PNEUMATIC;
END_REGION

REGION Network 68: CLOSED MISSING 4 ALARM
   RUNG wire#powerrail
      Contact( #M_VERIFY_CLOSED )
      I_Contact( #CYL.CLOSED_PART_D_I )
      Contact( #CHECK_CLOSED_CNC_PLC_SIGNAL )
      wire#w1
      Contact( #O_BYTE_0.CLOSED_PART_D )
      I_Contact( #ALARMS.CLOSED_OUTPUT_COMMAND_MISSING_ALARM )
      Contact( #HYDRAULIC_OR_PNEUMATIC )
      Coil( #ALARMS.CLOSED_MISSING_4_ALARM )
   END_RUNG
   RUNG wire#powerrail
      Contact( #ALARMS.CLOSED_MISSING_4_ALARM )
      I_Contact( "DB2120_MPP_ITC_IPC".RESET_FAULTS )
   END_RUNG wire#w1
   // the same network as SCL:
   #ALARMS.CLOSED_MISSING_4_ALARM := ((#M_VERIFY_CLOSED AND NOT #CYL.CLOSED_PART_D_I AND #CHECK_CLOSED_CNC_PLC_SIGNAL) OR (#ALARMS.CLOSED_MISSING_4_ALARM AND NOT "DB2120_MPP_ITC_IPC".RESET_FAULTS)) AND #O_BYTE_0.CLOSED_PART_D AND NOT #ALARMS.CLOSED_OUTPUT_COMMAND_MISSING_ALARM AND #HYDRAULIC_OR_PNEUMATIC;
END_REGION

REGION Network 69: CLOSED PRESSURE TIME EXCEEDED 1 ALARM
   RUNG wire#powerrail
      I_Contact( #CYL.CLOSE_COMMAND )
      I_Contact( #CLOSE )
      Not()
      I_Contact( #CYL.CLOSE_LOW_PRESSURE )
      I_Contact( #CYL.CLOSED_PRESSURE_SW_1_I )
      wire#w1
      Contact( #O_BYTE_0.CLOSED_PRESSURE_INPUT_1 )
      Contact( #HYDRAULIC_OR_PNEUMATIC )
      { S7_Templates := "time_type := Time" } #TIMER_ACTD_PRESSURE_TIME_EXCEEDED_1.TON(pt := #TIMER_ACTD_PRESSURE_TIME_EXCEEDED_1.PT, et =>)
      Coil( #ALARMS.CLOSED_PRESSURE_TIME_EXCEEDED_1_ALARM )
   END_RUNG
   RUNG wire#powerrail
      Contact( #ALARMS.CLOSED_PRESSURE_TIME_EXCEEDED_1_ALARM )
      I_Contact( "DB2120_MPP_ITC_IPC".RESET_FAULTS )
   END_RUNG wire#w1
   // the same network as SCL:
   #TIMER_ACTD_PRESSURE_TIME_EXCEEDED_1(IN := ((NOT (NOT #CYL.CLOSE_COMMAND AND NOT #CLOSE) AND NOT #CYL.CLOSE_LOW_PRESSURE AND NOT #CYL.CLOSED_PRESSURE_SW_1_I) OR (#ALARMS.CLOSED_PRESSURE_TIME_EXCEEDED_1_ALARM AND NOT "DB2120_MPP_ITC_IPC".RESET_FAULTS)) AND #O_BYTE_0.CLOSED_PRESSURE_INPUT_1 AND #HYDRAULIC_OR_PNEUMATIC,   // TON
                           PT := #TIMER_ACTD_PRESSURE_TIME_EXCEEDED_1.PT);
   #ALARMS.CLOSED_PRESSURE_TIME_EXCEEDED_1_ALARM := #TIMER_ACTD_PRESSURE_TIME_EXCEEDED_1.Q;
END_REGION

REGION Network 70: CLOSED PRESSURE SWITCH 1 ALARM
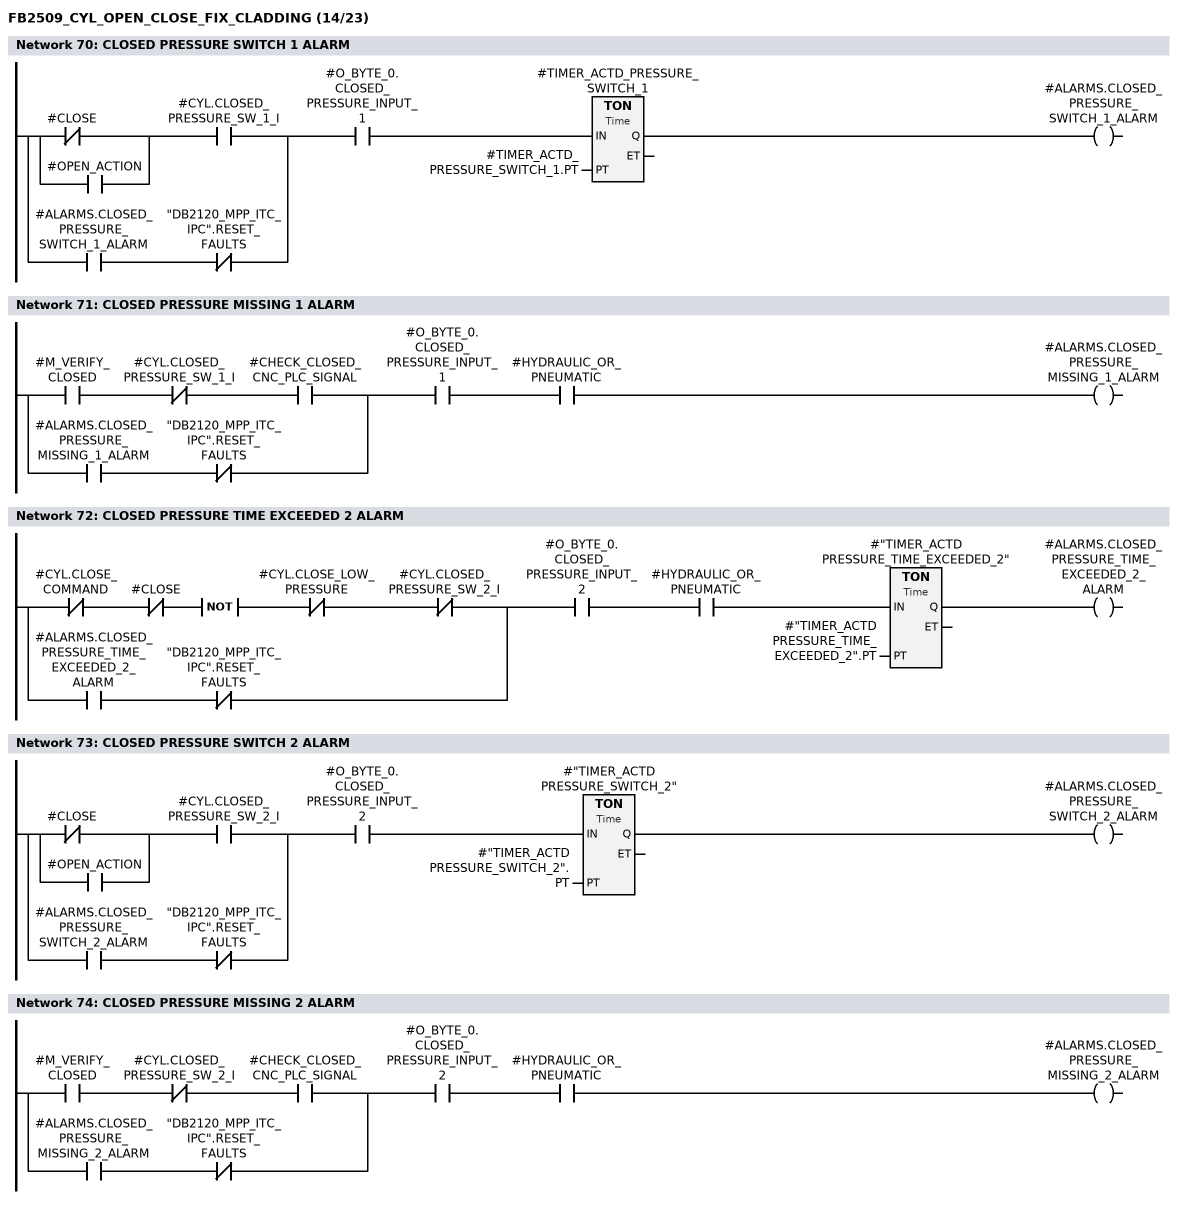
   RUNG wire#powerrail
      I_Contact( #CLOSE )
      wire#w1
      Contact( #CYL.CLOSED_PRESSURE_SW_1_I )
      wire#w2
      Contact( #O_BYTE_0.CLOSED_PRESSURE_INPUT_1 )
      { S7_Templates := "time_type := Time" } #TIMER_ACTD_PRESSURE_SWITCH_1.TON(pt := #TIMER_ACTD_PRESSURE_SWITCH_1.PT, et =>)
      Coil( #ALARMS.CLOSED_PRESSURE_SWITCH_1_ALARM )
   END_RUNG
   RUNG wire#powerrail
      Contact( #OPEN_ACTION )
   END_RUNG wire#w1
   RUNG wire#powerrail
      Contact( #ALARMS.CLOSED_PRESSURE_SWITCH_1_ALARM )
      I_Contact( "DB2120_MPP_ITC_IPC".RESET_FAULTS )
   END_RUNG wire#w2
   // the same network as SCL:
   #TIMER_ACTD_PRESSURE_SWITCH_1(IN := (((NOT #CLOSE OR #OPEN_ACTION) AND #CYL.CLOSED_PRESSURE_SW_1_I) OR (#ALARMS.CLOSED_PRESSURE_SWITCH_1_ALARM AND NOT "DB2120_MPP_ITC_IPC".RESET_FAULTS)) AND #O_BYTE_0.CLOSED_PRESSURE_INPUT_1,   // TON
                           PT := #TIMER_ACTD_PRESSURE_SWITCH_1.PT);
   #ALARMS.CLOSED_PRESSURE_SWITCH_1_ALARM := #TIMER_ACTD_PRESSURE_SWITCH_1.Q;
END_REGION

REGION Network 71: CLOSED PRESSURE MISSING 1 ALARM
   RUNG wire#powerrail
      Contact( #M_VERIFY_CLOSED )
      I_Contact( #CYL.CLOSED_PRESSURE_SW_1_I )
      Contact( #CHECK_CLOSED_CNC_PLC_SIGNAL )
      wire#w1
      Contact( #O_BYTE_0.CLOSED_PRESSURE_INPUT_1 )
      Contact( #HYDRAULIC_OR_PNEUMATIC )
      Coil( #ALARMS.CLOSED_PRESSURE_MISSING_1_ALARM )
   END_RUNG
   RUNG wire#powerrail
      Contact( #ALARMS.CLOSED_PRESSURE_MISSING_1_ALARM )
      I_Contact( "DB2120_MPP_ITC_IPC".RESET_FAULTS )
   END_RUNG wire#w1
   // the same network as SCL:
   #ALARMS.CLOSED_PRESSURE_MISSING_1_ALARM := ((#M_VERIFY_CLOSED AND NOT #CYL.CLOSED_PRESSURE_SW_1_I AND #CHECK_CLOSED_CNC_PLC_SIGNAL) OR (#ALARMS.CLOSED_PRESSURE_MISSING_1_ALARM AND NOT "DB2120_MPP_ITC_IPC".RESET_FAULTS)) AND #O_BYTE_0.CLOSED_PRESSURE_INPUT_1 AND #HYDRAULIC_OR_PNEUMATIC;
END_REGION

REGION Network 72: CLOSED PRESSURE TIME EXCEEDED 2 ALARM
   RUNG wire#powerrail
      I_Contact( #CYL.CLOSE_COMMAND )
      I_Contact( #CLOSE )
      Not()
      I_Contact( #CYL.CLOSE_LOW_PRESSURE )
      I_Contact( #CYL.CLOSED_PRESSURE_SW_2_I )
      wire#w1
      Contact( #O_BYTE_0.CLOSED_PRESSURE_INPUT_2 )
      Contact( #HYDRAULIC_OR_PNEUMATIC )
      { S7_Templates := "time_type := Time" } #"TIMER_ACTD PRESSURE_TIME_EXCEEDED_2".TON(pt := #"TIMER_ACTD PRESSURE_TIME_EXCEEDED_2".PT, et =>)
      Coil( #ALARMS.CLOSED_PRESSURE_TIME_EXCEEDED_2_ALARM )
   END_RUNG
   RUNG wire#powerrail
      Contact( #ALARMS.CLOSED_PRESSURE_TIME_EXCEEDED_2_ALARM )
      I_Contact( "DB2120_MPP_ITC_IPC".RESET_FAULTS )
   END_RUNG wire#w1
   // the same network as SCL:
   #"TIMER_ACTD PRESSURE_TIME_EXCEEDED_2"(IN := ((NOT (NOT #CYL.CLOSE_COMMAND AND NOT #CLOSE) AND NOT #CYL.CLOSE_LOW_PRESSURE AND NOT #CYL.CLOSED_PRESSURE_SW_2_I) OR (#ALARMS.CLOSED_PRESSURE_TIME_EXCEEDED_2_ALARM AND NOT "DB2120_MPP_ITC_IPC".RESET_FAULTS)) AND #O_BYTE_0.CLOSED_PRESSURE_INPUT_2 AND #HYDRAULIC_OR_PNEUMATIC,   // TON
                           PT := #"TIMER_ACTD PRESSURE_TIME_EXCEEDED_2".PT);
   #ALARMS.CLOSED_PRESSURE_TIME_EXCEEDED_2_ALARM := #"TIMER_ACTD PRESSURE_TIME_EXCEEDED_2".Q;
END_REGION

REGION Network 73: CLOSED PRESSURE SWITCH 2 ALARM
   RUNG wire#powerrail
      I_Contact( #CLOSE )
      wire#w1
      Contact( #CYL.CLOSED_PRESSURE_SW_2_I )
      wire#w2
      Contact( #O_BYTE_0.CLOSED_PRESSURE_INPUT_2 )
      { S7_Templates := "time_type := Time" } #"TIMER_ACTD PRESSURE_SWITCH_2".TON(pt := #"TIMER_ACTD PRESSURE_SWITCH_2".PT, et =>)
      Coil( #ALARMS.CLOSED_PRESSURE_SWITCH_2_ALARM )
   END_RUNG
   RUNG wire#powerrail
      Contact( #OPEN_ACTION )
   END_RUNG wire#w1
   RUNG wire#powerrail
      Contact( #ALARMS.CLOSED_PRESSURE_SWITCH_2_ALARM )
      I_Contact( "DB2120_MPP_ITC_IPC".RESET_FAULTS )
   END_RUNG wire#w2
   // the same network as SCL:
   #"TIMER_ACTD PRESSURE_SWITCH_2"(IN := (((NOT #CLOSE OR #OPEN_ACTION) AND #CYL.CLOSED_PRESSURE_SW_2_I) OR (#ALARMS.CLOSED_PRESSURE_SWITCH_2_ALARM AND NOT "DB2120_MPP_ITC_IPC".RESET_FAULTS)) AND #O_BYTE_0.CLOSED_PRESSURE_INPUT_2,   // TON
                           PT := #"TIMER_ACTD PRESSURE_SWITCH_2".PT);
   #ALARMS.CLOSED_PRESSURE_SWITCH_2_ALARM := #"TIMER_ACTD PRESSURE_SWITCH_2".Q;
END_REGION

REGION Network 74: CLOSED PRESSURE MISSING 2 ALARM
   RUNG wire#powerrail
      Contact( #M_VERIFY_CLOSED )
      I_Contact( #CYL.CLOSED_PRESSURE_SW_2_I )
      Contact( #CHECK_CLOSED_CNC_PLC_SIGNAL )
      wire#w1
      Contact( #O_BYTE_0.CLOSED_PRESSURE_INPUT_2 )
      Contact( #HYDRAULIC_OR_PNEUMATIC )
      Coil( #ALARMS.CLOSED_PRESSURE_MISSING_2_ALARM )
   END_RUNG
   RUNG wire#powerrail
      Contact( #ALARMS.CLOSED_PRESSURE_MISSING_2_ALARM )
      I_Contact( "DB2120_MPP_ITC_IPC".RESET_FAULTS )
   END_RUNG wire#w1
   // the same network as SCL:
   #ALARMS.CLOSED_PRESSURE_MISSING_2_ALARM := ((#M_VERIFY_CLOSED AND NOT #CYL.CLOSED_PRESSURE_SW_2_I AND #CHECK_CLOSED_CNC_PLC_SIGNAL) OR (#ALARMS.CLOSED_PRESSURE_MISSING_2_ALARM AND NOT "DB2120_MPP_ITC_IPC".RESET_FAULTS)) AND #O_BYTE_0.CLOSED_PRESSURE_INPUT_2 AND #HYDRAULIC_OR_PNEUMATIC;
END_REGION

REGION Network 75: OPEN OUTPUT COMMAND MISSING ALARM
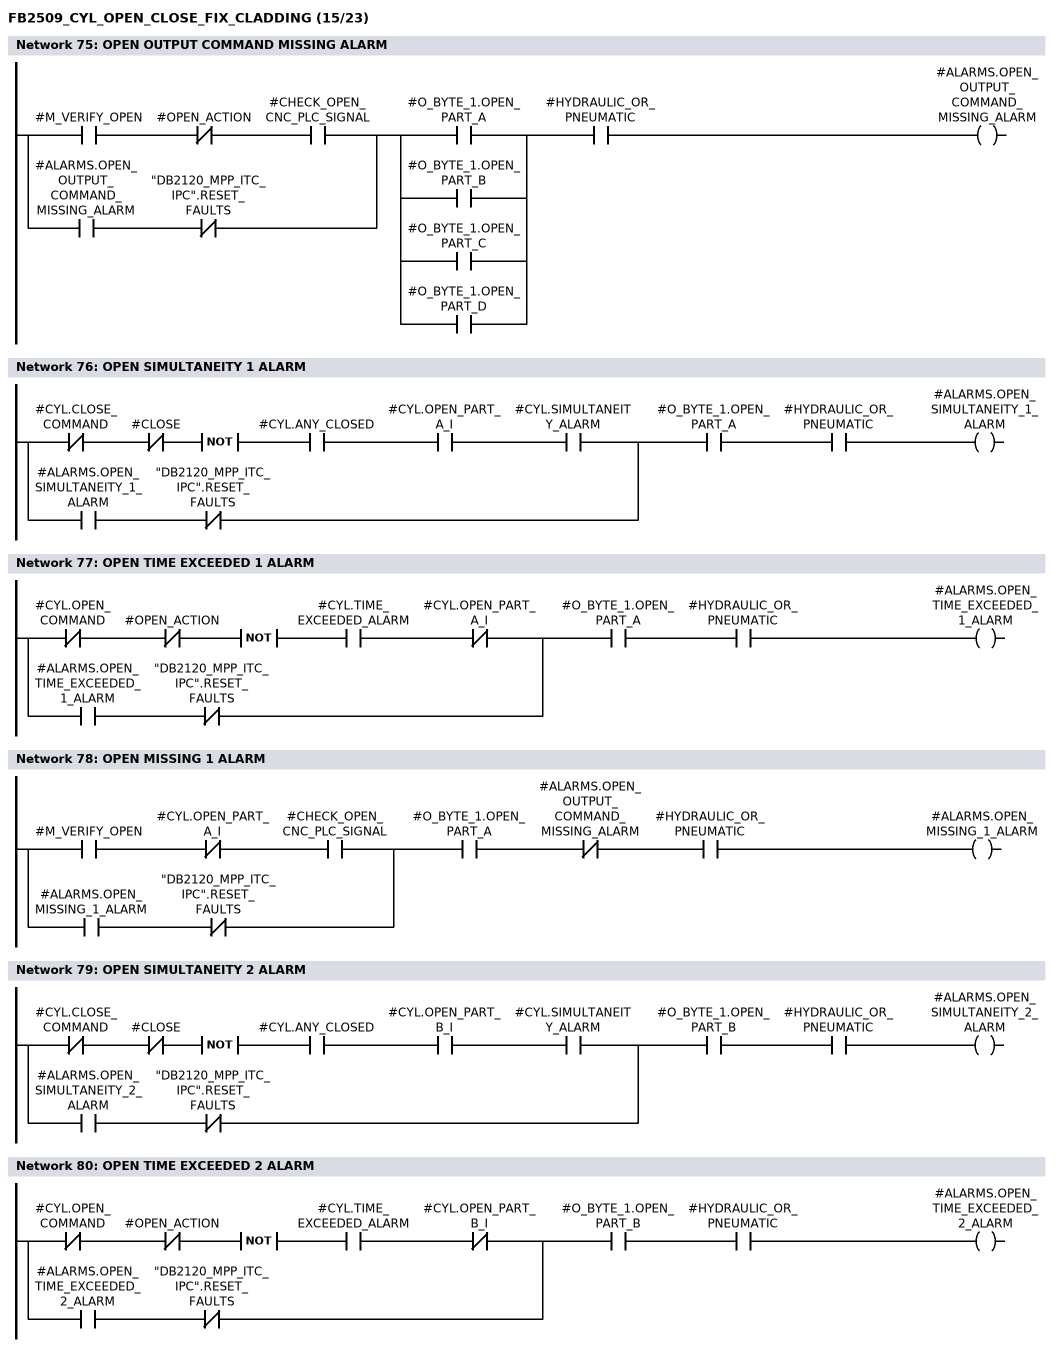
   RUNG wire#powerrail
      Contact( #M_VERIFY_OPEN )
      I_Contact( #OPEN_ACTION )
      Contact( #CHECK_OPEN_CNC_PLC_SIGNAL )
      wire#w1
      Contact( #O_BYTE_1.OPEN_PART_A )
      wire#w2
      Contact( #HYDRAULIC_OR_PNEUMATIC )
      Coil( #ALARMS.OPEN_OUTPUT_COMMAND_MISSING_ALARM )
   END_RUNG
   RUNG wire#powerrail
      Contact( #ALARMS.OPEN_OUTPUT_COMMAND_MISSING_ALARM )
      I_Contact( "DB2120_MPP_ITC_IPC".RESET_FAULTS )
   END_RUNG wire#w1
   RUNG wire#w1
      Contact( #O_BYTE_1.OPEN_PART_B )
   END_RUNG wire#w2
   RUNG wire#w1
      Contact( #O_BYTE_1.OPEN_PART_C )
   END_RUNG wire#w2
   RUNG wire#w1
      Contact( #O_BYTE_1.OPEN_PART_D )
   END_RUNG wire#w2
   // the same network as SCL:
   #ALARMS.OPEN_OUTPUT_COMMAND_MISSING_ALARM := ((#M_VERIFY_OPEN AND NOT #OPEN_ACTION AND #CHECK_OPEN_CNC_PLC_SIGNAL) OR (#ALARMS.OPEN_OUTPUT_COMMAND_MISSING_ALARM AND NOT "DB2120_MPP_ITC_IPC".RESET_FAULTS)) AND (#O_BYTE_1.OPEN_PART_A OR #O_BYTE_1.OPEN_PART_B OR #O_BYTE_1.OPEN_PART_C OR #O_BYTE_1.OPEN_PART_D) AND #HYDRAULIC_OR_PNEUMATIC;
END_REGION

REGION Network 76: OPEN SIMULTANEITY 1 ALARM
   RUNG wire#powerrail
      I_Contact( #CYL.CLOSE_COMMAND )
      I_Contact( #CLOSE )
      Not()
      Contact( #CYL.ANY_CLOSED )
      Contact( #CYL.OPEN_PART_A_I )
      Contact( #CYL.SIMULTANEITY_ALARM )
      wire#w1
      Contact( #O_BYTE_1.OPEN_PART_A )
      Contact( #HYDRAULIC_OR_PNEUMATIC )
      Coil( #ALARMS.OPEN_SIMULTANEITY_1_ALARM )
   END_RUNG
   RUNG wire#powerrail
      Contact( #ALARMS.OPEN_SIMULTANEITY_1_ALARM )
      I_Contact( "DB2120_MPP_ITC_IPC".RESET_FAULTS )
   END_RUNG wire#w1
   // the same network as SCL:
   #ALARMS.OPEN_SIMULTANEITY_1_ALARM := ((NOT (NOT #CYL.CLOSE_COMMAND AND NOT #CLOSE) AND #CYL.ANY_CLOSED AND #CYL.OPEN_PART_A_I AND #CYL.SIMULTANEITY_ALARM) OR (#ALARMS.OPEN_SIMULTANEITY_1_ALARM AND NOT "DB2120_MPP_ITC_IPC".RESET_FAULTS)) AND #O_BYTE_1.OPEN_PART_A AND #HYDRAULIC_OR_PNEUMATIC;
END_REGION

REGION Network 77: OPEN TIME EXCEEDED 1 ALARM
   RUNG wire#powerrail
      I_Contact( #CYL.OPEN_COMMAND )
      I_Contact( #OPEN_ACTION )
      Not()
      Contact( #CYL.TIME_EXCEEDED_ALARM )
      I_Contact( #CYL.OPEN_PART_A_I )
      wire#w1
      Contact( #O_BYTE_1.OPEN_PART_A )
      Contact( #HYDRAULIC_OR_PNEUMATIC )
      Coil( #ALARMS.OPEN_TIME_EXCEEDED_1_ALARM )
   END_RUNG
   RUNG wire#powerrail
      Contact( #ALARMS.OPEN_TIME_EXCEEDED_1_ALARM )
      I_Contact( "DB2120_MPP_ITC_IPC".RESET_FAULTS )
   END_RUNG wire#w1
   // the same network as SCL:
   #ALARMS.OPEN_TIME_EXCEEDED_1_ALARM := ((NOT (NOT #CYL.OPEN_COMMAND AND NOT #OPEN_ACTION) AND #CYL.TIME_EXCEEDED_ALARM AND NOT #CYL.OPEN_PART_A_I) OR (#ALARMS.OPEN_TIME_EXCEEDED_1_ALARM AND NOT "DB2120_MPP_ITC_IPC".RESET_FAULTS)) AND #O_BYTE_1.OPEN_PART_A AND #HYDRAULIC_OR_PNEUMATIC;
END_REGION

REGION Network 78: OPEN MISSING 1 ALARM
   RUNG wire#powerrail
      Contact( #M_VERIFY_OPEN )
      I_Contact( #CYL.OPEN_PART_A_I )
      Contact( #CHECK_OPEN_CNC_PLC_SIGNAL )
      wire#w1
      Contact( #O_BYTE_1.OPEN_PART_A )
      I_Contact( #ALARMS.OPEN_OUTPUT_COMMAND_MISSING_ALARM )
      Contact( #HYDRAULIC_OR_PNEUMATIC )
      Coil( #ALARMS.OPEN_MISSING_1_ALARM )
   END_RUNG
   RUNG wire#powerrail
      Contact( #ALARMS.OPEN_MISSING_1_ALARM )
      I_Contact( "DB2120_MPP_ITC_IPC".RESET_FAULTS )
   END_RUNG wire#w1
   // the same network as SCL:
   #ALARMS.OPEN_MISSING_1_ALARM := ((#M_VERIFY_OPEN AND NOT #CYL.OPEN_PART_A_I AND #CHECK_OPEN_CNC_PLC_SIGNAL) OR (#ALARMS.OPEN_MISSING_1_ALARM AND NOT "DB2120_MPP_ITC_IPC".RESET_FAULTS)) AND #O_BYTE_1.OPEN_PART_A AND NOT #ALARMS.OPEN_OUTPUT_COMMAND_MISSING_ALARM AND #HYDRAULIC_OR_PNEUMATIC;
END_REGION

REGION Network 79: OPEN SIMULTANEITY 2 ALARM
   RUNG wire#powerrail
      I_Contact( #CYL.CLOSE_COMMAND )
      I_Contact( #CLOSE )
      Not()
      Contact( #CYL.ANY_CLOSED )
      Contact( #CYL.OPEN_PART_B_I )
      Contact( #CYL.SIMULTANEITY_ALARM )
      wire#w1
      Contact( #O_BYTE_1.OPEN_PART_B )
      Contact( #HYDRAULIC_OR_PNEUMATIC )
      Coil( #ALARMS.OPEN_SIMULTANEITY_2_ALARM )
   END_RUNG
   RUNG wire#powerrail
      Contact( #ALARMS.OPEN_SIMULTANEITY_2_ALARM )
      I_Contact( "DB2120_MPP_ITC_IPC".RESET_FAULTS )
   END_RUNG wire#w1
   // the same network as SCL:
   #ALARMS.OPEN_SIMULTANEITY_2_ALARM := ((NOT (NOT #CYL.CLOSE_COMMAND AND NOT #CLOSE) AND #CYL.ANY_CLOSED AND #CYL.OPEN_PART_B_I AND #CYL.SIMULTANEITY_ALARM) OR (#ALARMS.OPEN_SIMULTANEITY_2_ALARM AND NOT "DB2120_MPP_ITC_IPC".RESET_FAULTS)) AND #O_BYTE_1.OPEN_PART_B AND #HYDRAULIC_OR_PNEUMATIC;
END_REGION

REGION Network 80: OPEN TIME EXCEEDED 2 ALARM
   RUNG wire#powerrail
      I_Contact( #CYL.OPEN_COMMAND )
      I_Contact( #OPEN_ACTION )
      Not()
      Contact( #CYL.TIME_EXCEEDED_ALARM )
      I_Contact( #CYL.OPEN_PART_B_I )
      wire#w1
      Contact( #O_BYTE_1.OPEN_PART_B )
      Contact( #HYDRAULIC_OR_PNEUMATIC )
      Coil( #ALARMS.OPEN_TIME_EXCEEDED_2_ALARM )
   END_RUNG
   RUNG wire#powerrail
      Contact( #ALARMS.OPEN_TIME_EXCEEDED_2_ALARM )
      I_Contact( "DB2120_MPP_ITC_IPC".RESET_FAULTS )
   END_RUNG wire#w1
   // the same network as SCL:
   #ALARMS.OPEN_TIME_EXCEEDED_2_ALARM := ((NOT (NOT #CYL.OPEN_COMMAND AND NOT #OPEN_ACTION) AND #CYL.TIME_EXCEEDED_ALARM AND NOT #CYL.OPEN_PART_B_I) OR (#ALARMS.OPEN_TIME_EXCEEDED_2_ALARM AND NOT "DB2120_MPP_ITC_IPC".RESET_FAULTS)) AND #O_BYTE_1.OPEN_PART_B AND #HYDRAULIC_OR_PNEUMATIC;
END_REGION

REGION Network 81: OPEN MISSING 2 ALARM
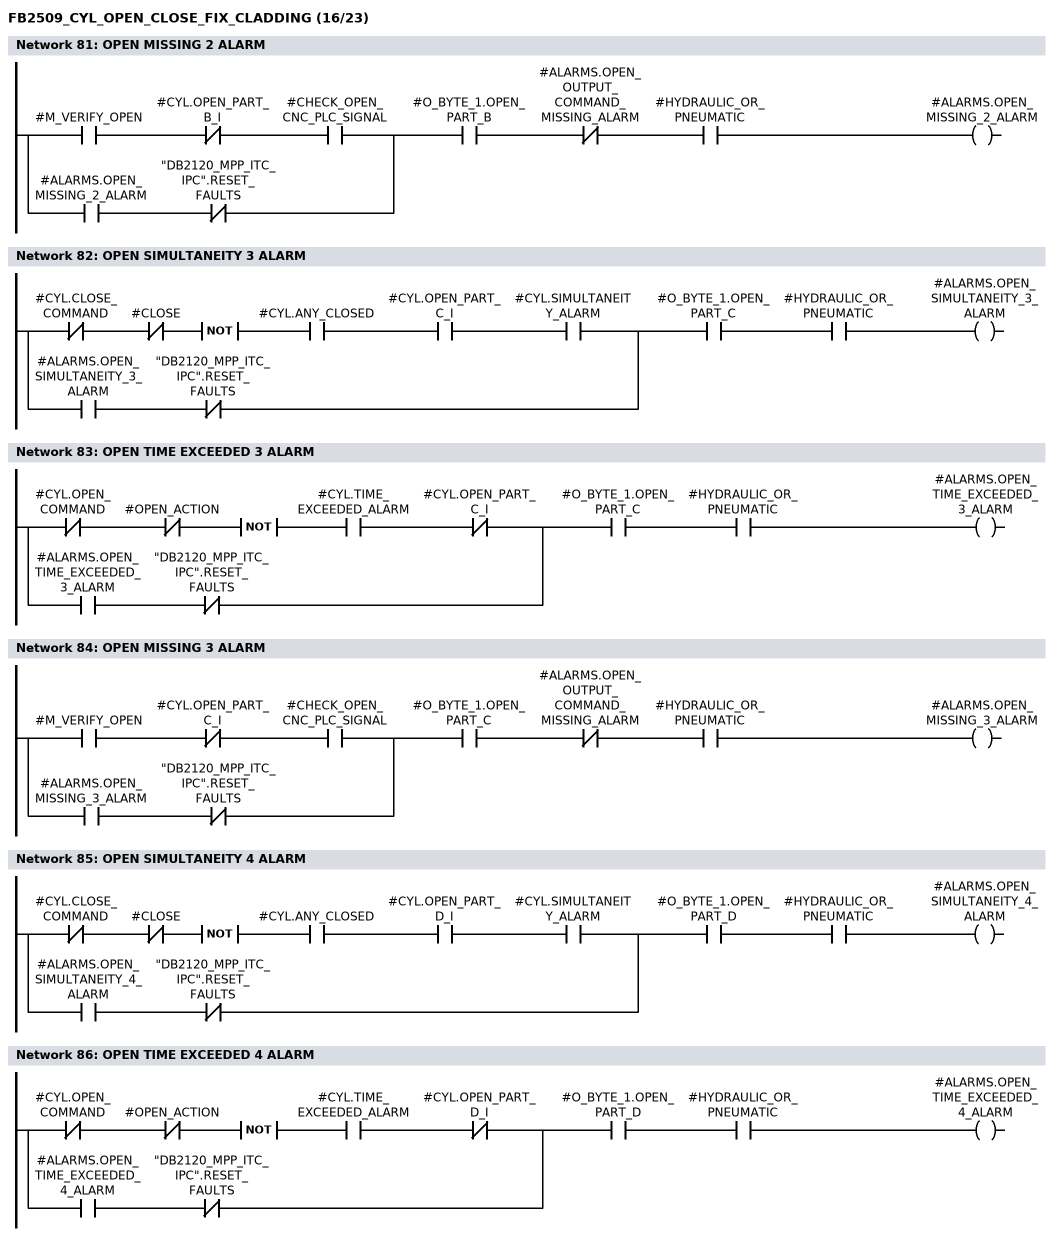
   RUNG wire#powerrail
      Contact( #M_VERIFY_OPEN )
      I_Contact( #CYL.OPEN_PART_B_I )
      Contact( #CHECK_OPEN_CNC_PLC_SIGNAL )
      wire#w1
      Contact( #O_BYTE_1.OPEN_PART_B )
      I_Contact( #ALARMS.OPEN_OUTPUT_COMMAND_MISSING_ALARM )
      Contact( #HYDRAULIC_OR_PNEUMATIC )
      Coil( #ALARMS.OPEN_MISSING_2_ALARM )
   END_RUNG
   RUNG wire#powerrail
      Contact( #ALARMS.OPEN_MISSING_2_ALARM )
      I_Contact( "DB2120_MPP_ITC_IPC".RESET_FAULTS )
   END_RUNG wire#w1
   // the same network as SCL:
   #ALARMS.OPEN_MISSING_2_ALARM := ((#M_VERIFY_OPEN AND NOT #CYL.OPEN_PART_B_I AND #CHECK_OPEN_CNC_PLC_SIGNAL) OR (#ALARMS.OPEN_MISSING_2_ALARM AND NOT "DB2120_MPP_ITC_IPC".RESET_FAULTS)) AND #O_BYTE_1.OPEN_PART_B AND NOT #ALARMS.OPEN_OUTPUT_COMMAND_MISSING_ALARM AND #HYDRAULIC_OR_PNEUMATIC;
END_REGION

REGION Network 82: OPEN SIMULTANEITY 3 ALARM
   RUNG wire#powerrail
      I_Contact( #CYL.CLOSE_COMMAND )
      I_Contact( #CLOSE )
      Not()
      Contact( #CYL.ANY_CLOSED )
      Contact( #CYL.OPEN_PART_C_I )
      Contact( #CYL.SIMULTANEITY_ALARM )
      wire#w1
      Contact( #O_BYTE_1.OPEN_PART_C )
      Contact( #HYDRAULIC_OR_PNEUMATIC )
      Coil( #ALARMS.OPEN_SIMULTANEITY_3_ALARM )
   END_RUNG
   RUNG wire#powerrail
      Contact( #ALARMS.OPEN_SIMULTANEITY_3_ALARM )
      I_Contact( "DB2120_MPP_ITC_IPC".RESET_FAULTS )
   END_RUNG wire#w1
   // the same network as SCL:
   #ALARMS.OPEN_SIMULTANEITY_3_ALARM := ((NOT (NOT #CYL.CLOSE_COMMAND AND NOT #CLOSE) AND #CYL.ANY_CLOSED AND #CYL.OPEN_PART_C_I AND #CYL.SIMULTANEITY_ALARM) OR (#ALARMS.OPEN_SIMULTANEITY_3_ALARM AND NOT "DB2120_MPP_ITC_IPC".RESET_FAULTS)) AND #O_BYTE_1.OPEN_PART_C AND #HYDRAULIC_OR_PNEUMATIC;
END_REGION

REGION Network 83: OPEN TIME EXCEEDED 3 ALARM
   RUNG wire#powerrail
      I_Contact( #CYL.OPEN_COMMAND )
      I_Contact( #OPEN_ACTION )
      Not()
      Contact( #CYL.TIME_EXCEEDED_ALARM )
      I_Contact( #CYL.OPEN_PART_C_I )
      wire#w1
      Contact( #O_BYTE_1.OPEN_PART_C )
      Contact( #HYDRAULIC_OR_PNEUMATIC )
      Coil( #ALARMS.OPEN_TIME_EXCEEDED_3_ALARM )
   END_RUNG
   RUNG wire#powerrail
      Contact( #ALARMS.OPEN_TIME_EXCEEDED_3_ALARM )
      I_Contact( "DB2120_MPP_ITC_IPC".RESET_FAULTS )
   END_RUNG wire#w1
   // the same network as SCL:
   #ALARMS.OPEN_TIME_EXCEEDED_3_ALARM := ((NOT (NOT #CYL.OPEN_COMMAND AND NOT #OPEN_ACTION) AND #CYL.TIME_EXCEEDED_ALARM AND NOT #CYL.OPEN_PART_C_I) OR (#ALARMS.OPEN_TIME_EXCEEDED_3_ALARM AND NOT "DB2120_MPP_ITC_IPC".RESET_FAULTS)) AND #O_BYTE_1.OPEN_PART_C AND #HYDRAULIC_OR_PNEUMATIC;
END_REGION

REGION Network 84: OPEN MISSING 3 ALARM
   RUNG wire#powerrail
      Contact( #M_VERIFY_OPEN )
      I_Contact( #CYL.OPEN_PART_C_I )
      Contact( #CHECK_OPEN_CNC_PLC_SIGNAL )
      wire#w1
      Contact( #O_BYTE_1.OPEN_PART_C )
      I_Contact( #ALARMS.OPEN_OUTPUT_COMMAND_MISSING_ALARM )
      Contact( #HYDRAULIC_OR_PNEUMATIC )
      Coil( #ALARMS.OPEN_MISSING_3_ALARM )
   END_RUNG
   RUNG wire#powerrail
      Contact( #ALARMS.OPEN_MISSING_3_ALARM )
      I_Contact( "DB2120_MPP_ITC_IPC".RESET_FAULTS )
   END_RUNG wire#w1
   // the same network as SCL:
   #ALARMS.OPEN_MISSING_3_ALARM := ((#M_VERIFY_OPEN AND NOT #CYL.OPEN_PART_C_I AND #CHECK_OPEN_CNC_PLC_SIGNAL) OR (#ALARMS.OPEN_MISSING_3_ALARM AND NOT "DB2120_MPP_ITC_IPC".RESET_FAULTS)) AND #O_BYTE_1.OPEN_PART_C AND NOT #ALARMS.OPEN_OUTPUT_COMMAND_MISSING_ALARM AND #HYDRAULIC_OR_PNEUMATIC;
END_REGION

REGION Network 85: OPEN SIMULTANEITY 4 ALARM
   RUNG wire#powerrail
      I_Contact( #CYL.CLOSE_COMMAND )
      I_Contact( #CLOSE )
      Not()
      Contact( #CYL.ANY_CLOSED )
      Contact( #CYL.OPEN_PART_D_I )
      Contact( #CYL.SIMULTANEITY_ALARM )
      wire#w1
      Contact( #O_BYTE_1.OPEN_PART_D )
      Contact( #HYDRAULIC_OR_PNEUMATIC )
      Coil( #ALARMS.OPEN_SIMULTANEITY_4_ALARM )
   END_RUNG
   RUNG wire#powerrail
      Contact( #ALARMS.OPEN_SIMULTANEITY_4_ALARM )
      I_Contact( "DB2120_MPP_ITC_IPC".RESET_FAULTS )
   END_RUNG wire#w1
   // the same network as SCL:
   #ALARMS.OPEN_SIMULTANEITY_4_ALARM := ((NOT (NOT #CYL.CLOSE_COMMAND AND NOT #CLOSE) AND #CYL.ANY_CLOSED AND #CYL.OPEN_PART_D_I AND #CYL.SIMULTANEITY_ALARM) OR (#ALARMS.OPEN_SIMULTANEITY_4_ALARM AND NOT "DB2120_MPP_ITC_IPC".RESET_FAULTS)) AND #O_BYTE_1.OPEN_PART_D AND #HYDRAULIC_OR_PNEUMATIC;
END_REGION

REGION Network 86: OPEN TIME EXCEEDED 4 ALARM
   RUNG wire#powerrail
      I_Contact( #CYL.OPEN_COMMAND )
      I_Contact( #OPEN_ACTION )
      Not()
      Contact( #CYL.TIME_EXCEEDED_ALARM )
      I_Contact( #CYL.OPEN_PART_D_I )
      wire#w1
      Contact( #O_BYTE_1.OPEN_PART_D )
      Contact( #HYDRAULIC_OR_PNEUMATIC )
      Coil( #ALARMS.OPEN_TIME_EXCEEDED_4_ALARM )
   END_RUNG
   RUNG wire#powerrail
      Contact( #ALARMS.OPEN_TIME_EXCEEDED_4_ALARM )
      I_Contact( "DB2120_MPP_ITC_IPC".RESET_FAULTS )
   END_RUNG wire#w1
   // the same network as SCL:
   #ALARMS.OPEN_TIME_EXCEEDED_4_ALARM := ((NOT (NOT #CYL.OPEN_COMMAND AND NOT #OPEN_ACTION) AND #CYL.TIME_EXCEEDED_ALARM AND NOT #CYL.OPEN_PART_D_I) OR (#ALARMS.OPEN_TIME_EXCEEDED_4_ALARM AND NOT "DB2120_MPP_ITC_IPC".RESET_FAULTS)) AND #O_BYTE_1.OPEN_PART_D AND #HYDRAULIC_OR_PNEUMATIC;
END_REGION

REGION Network 87: OPEN MISSING 4 ALARM
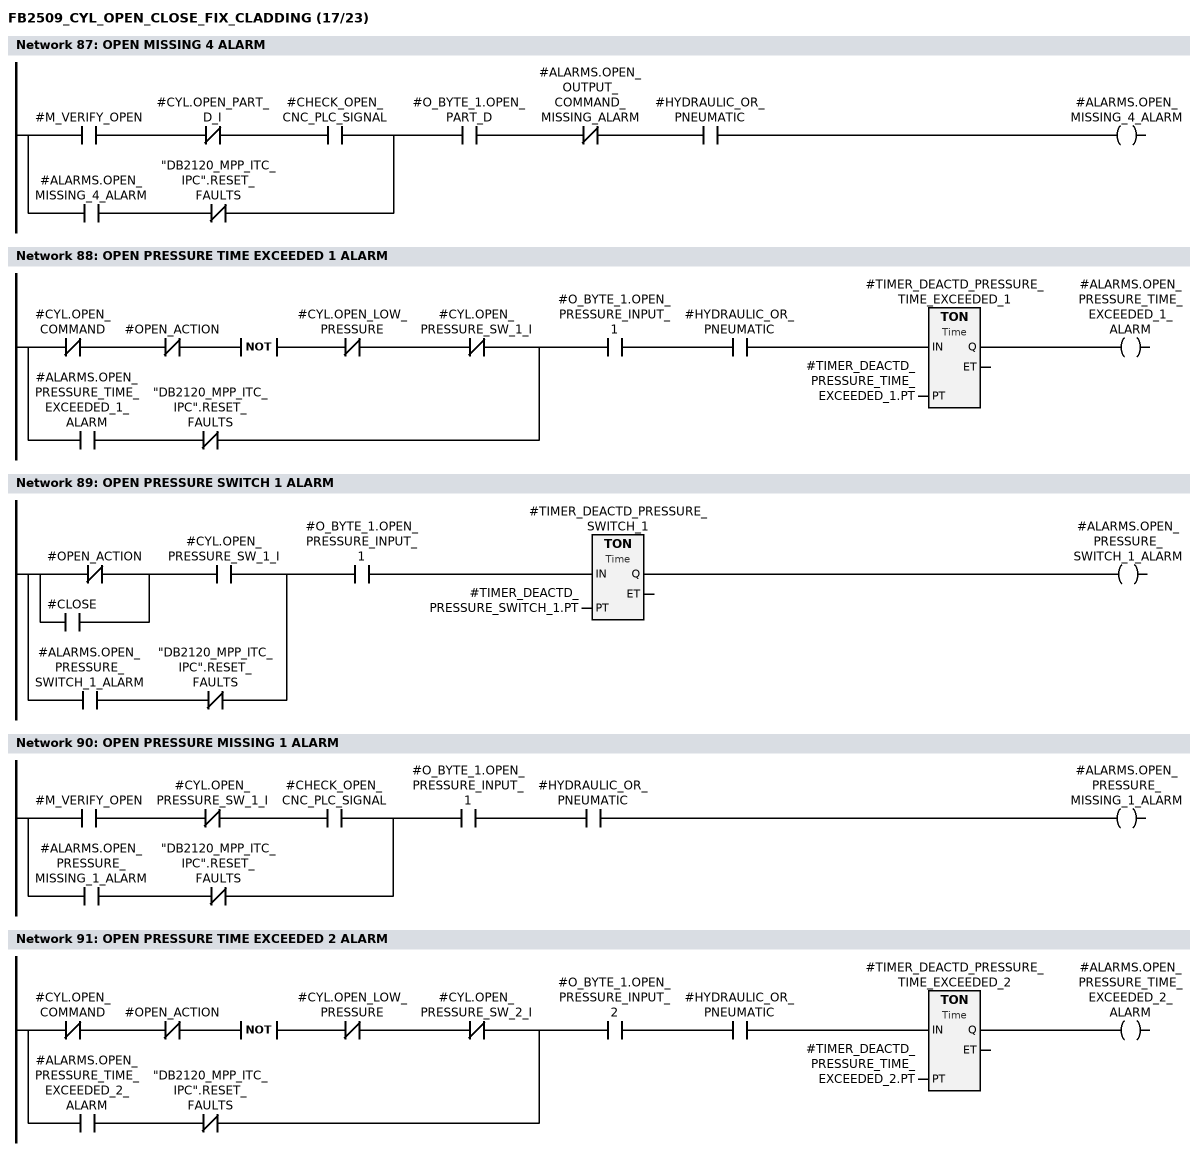
   RUNG wire#powerrail
      Contact( #M_VERIFY_OPEN )
      I_Contact( #CYL.OPEN_PART_D_I )
      Contact( #CHECK_OPEN_CNC_PLC_SIGNAL )
      wire#w1
      Contact( #O_BYTE_1.OPEN_PART_D )
      I_Contact( #ALARMS.OPEN_OUTPUT_COMMAND_MISSING_ALARM )
      Contact( #HYDRAULIC_OR_PNEUMATIC )
      Coil( #ALARMS.OPEN_MISSING_4_ALARM )
   END_RUNG
   RUNG wire#powerrail
      Contact( #ALARMS.OPEN_MISSING_4_ALARM )
      I_Contact( "DB2120_MPP_ITC_IPC".RESET_FAULTS )
   END_RUNG wire#w1
   // the same network as SCL:
   #ALARMS.OPEN_MISSING_4_ALARM := ((#M_VERIFY_OPEN AND NOT #CYL.OPEN_PART_D_I AND #CHECK_OPEN_CNC_PLC_SIGNAL) OR (#ALARMS.OPEN_MISSING_4_ALARM AND NOT "DB2120_MPP_ITC_IPC".RESET_FAULTS)) AND #O_BYTE_1.OPEN_PART_D AND NOT #ALARMS.OPEN_OUTPUT_COMMAND_MISSING_ALARM AND #HYDRAULIC_OR_PNEUMATIC;
END_REGION

REGION Network 88: OPEN PRESSURE TIME EXCEEDED 1 ALARM
   RUNG wire#powerrail
      I_Contact( #CYL.OPEN_COMMAND )
      I_Contact( #OPEN_ACTION )
      Not()
      I_Contact( #CYL.OPEN_LOW_PRESSURE )
      I_Contact( #CYL.OPEN_PRESSURE_SW_1_I )
      wire#w1
      Contact( #O_BYTE_1.OPEN_PRESSURE_INPUT_1 )
      Contact( #HYDRAULIC_OR_PNEUMATIC )
      { S7_Templates := "time_type := Time" } #TIMER_DEACTD_PRESSURE_TIME_EXCEEDED_1.TON(pt := #TIMER_DEACTD_PRESSURE_TIME_EXCEEDED_1.PT, et =>)
      Coil( #ALARMS.OPEN_PRESSURE_TIME_EXCEEDED_1_ALARM )
   END_RUNG
   RUNG wire#powerrail
      Contact( #ALARMS.OPEN_PRESSURE_TIME_EXCEEDED_1_ALARM )
      I_Contact( "DB2120_MPP_ITC_IPC".RESET_FAULTS )
   END_RUNG wire#w1
   // the same network as SCL:
   #TIMER_DEACTD_PRESSURE_TIME_EXCEEDED_1(IN := ((NOT (NOT #CYL.OPEN_COMMAND AND NOT #OPEN_ACTION) AND NOT #CYL.OPEN_LOW_PRESSURE AND NOT #CYL.OPEN_PRESSURE_SW_1_I) OR (#ALARMS.OPEN_PRESSURE_TIME_EXCEEDED_1_ALARM AND NOT "DB2120_MPP_ITC_IPC".RESET_FAULTS)) AND #O_BYTE_1.OPEN_PRESSURE_INPUT_1 AND #HYDRAULIC_OR_PNEUMATIC,   // TON
                           PT := #TIMER_DEACTD_PRESSURE_TIME_EXCEEDED_1.PT);
   #ALARMS.OPEN_PRESSURE_TIME_EXCEEDED_1_ALARM := #TIMER_DEACTD_PRESSURE_TIME_EXCEEDED_1.Q;
END_REGION

REGION Network 89: OPEN PRESSURE SWITCH 1 ALARM
   RUNG wire#powerrail
      I_Contact( #OPEN_ACTION )
      wire#w1
      Contact( #CYL.OPEN_PRESSURE_SW_1_I )
      wire#w2
      Contact( #O_BYTE_1.OPEN_PRESSURE_INPUT_1 )
      { S7_Templates := "time_type := Time" } #TIMER_DEACTD_PRESSURE_SWITCH_1.TON(pt := #TIMER_DEACTD_PRESSURE_SWITCH_1.PT, et =>)
      Coil( #ALARMS.OPEN_PRESSURE_SWITCH_1_ALARM )
   END_RUNG
   RUNG wire#powerrail
      Contact( #CLOSE )
   END_RUNG wire#w1
   RUNG wire#powerrail
      Contact( #ALARMS.OPEN_PRESSURE_SWITCH_1_ALARM )
      I_Contact( "DB2120_MPP_ITC_IPC".RESET_FAULTS )
   END_RUNG wire#w2
   // the same network as SCL:
   #TIMER_DEACTD_PRESSURE_SWITCH_1(IN := (((NOT #OPEN_ACTION OR #CLOSE) AND #CYL.OPEN_PRESSURE_SW_1_I) OR (#ALARMS.OPEN_PRESSURE_SWITCH_1_ALARM AND NOT "DB2120_MPP_ITC_IPC".RESET_FAULTS)) AND #O_BYTE_1.OPEN_PRESSURE_INPUT_1,   // TON
                           PT := #TIMER_DEACTD_PRESSURE_SWITCH_1.PT);
   #ALARMS.OPEN_PRESSURE_SWITCH_1_ALARM := #TIMER_DEACTD_PRESSURE_SWITCH_1.Q;
END_REGION

REGION Network 90: OPEN PRESSURE MISSING 1 ALARM
   RUNG wire#powerrail
      Contact( #M_VERIFY_OPEN )
      I_Contact( #CYL.OPEN_PRESSURE_SW_1_I )
      Contact( #CHECK_OPEN_CNC_PLC_SIGNAL )
      wire#w1
      Contact( #O_BYTE_1.OPEN_PRESSURE_INPUT_1 )
      Contact( #HYDRAULIC_OR_PNEUMATIC )
      Coil( #ALARMS.OPEN_PRESSURE_MISSING_1_ALARM )
   END_RUNG
   RUNG wire#powerrail
      Contact( #ALARMS.OPEN_PRESSURE_MISSING_1_ALARM )
      I_Contact( "DB2120_MPP_ITC_IPC".RESET_FAULTS )
   END_RUNG wire#w1
   // the same network as SCL:
   #ALARMS.OPEN_PRESSURE_MISSING_1_ALARM := ((#M_VERIFY_OPEN AND NOT #CYL.OPEN_PRESSURE_SW_1_I AND #CHECK_OPEN_CNC_PLC_SIGNAL) OR (#ALARMS.OPEN_PRESSURE_MISSING_1_ALARM AND NOT "DB2120_MPP_ITC_IPC".RESET_FAULTS)) AND #O_BYTE_1.OPEN_PRESSURE_INPUT_1 AND #HYDRAULIC_OR_PNEUMATIC;
END_REGION

REGION Network 91: OPEN PRESSURE TIME EXCEEDED 2 ALARM
   RUNG wire#powerrail
      I_Contact( #CYL.OPEN_COMMAND )
      I_Contact( #OPEN_ACTION )
      Not()
      I_Contact( #CYL.OPEN_LOW_PRESSURE )
      I_Contact( #CYL.OPEN_PRESSURE_SW_2_I )
      wire#w1
      Contact( #O_BYTE_1.OPEN_PRESSURE_INPUT_2 )
      Contact( #HYDRAULIC_OR_PNEUMATIC )
      { S7_Templates := "time_type := Time" } #TIMER_DEACTD_PRESSURE_TIME_EXCEEDED_2.TON(pt := #TIMER_DEACTD_PRESSURE_TIME_EXCEEDED_2.PT, et =>)
      Coil( #ALARMS.OPEN_PRESSURE_TIME_EXCEEDED_2_ALARM )
   END_RUNG
   RUNG wire#powerrail
      Contact( #ALARMS.OPEN_PRESSURE_TIME_EXCEEDED_2_ALARM )
      I_Contact( "DB2120_MPP_ITC_IPC".RESET_FAULTS )
   END_RUNG wire#w1
   // the same network as SCL:
   #TIMER_DEACTD_PRESSURE_TIME_EXCEEDED_2(IN := ((NOT (NOT #CYL.OPEN_COMMAND AND NOT #OPEN_ACTION) AND NOT #CYL.OPEN_LOW_PRESSURE AND NOT #CYL.OPEN_PRESSURE_SW_2_I) OR (#ALARMS.OPEN_PRESSURE_TIME_EXCEEDED_2_ALARM AND NOT "DB2120_MPP_ITC_IPC".RESET_FAULTS)) AND #O_BYTE_1.OPEN_PRESSURE_INPUT_2 AND #HYDRAULIC_OR_PNEUMATIC,   // TON
                           PT := #TIMER_DEACTD_PRESSURE_TIME_EXCEEDED_2.PT);
   #ALARMS.OPEN_PRESSURE_TIME_EXCEEDED_2_ALARM := #TIMER_DEACTD_PRESSURE_TIME_EXCEEDED_2.Q;
END_REGION

REGION Network 92: OPEN PRESSURE SWITCH 2 ALARM
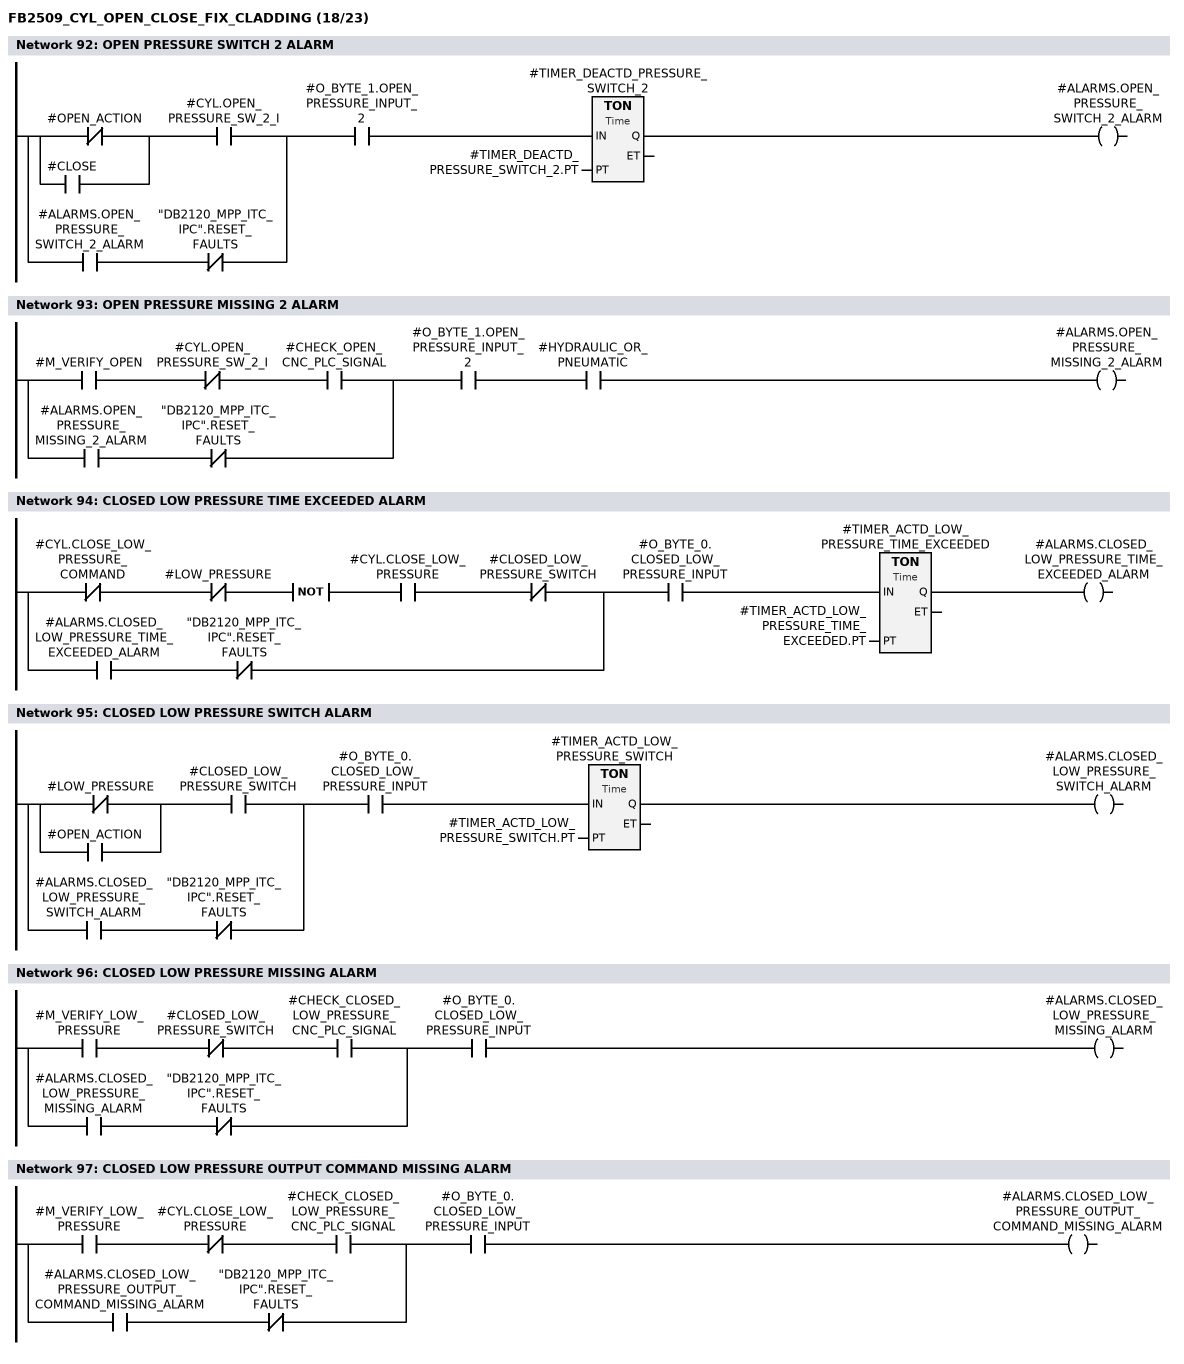
   RUNG wire#powerrail
      I_Contact( #OPEN_ACTION )
      wire#w1
      Contact( #CYL.OPEN_PRESSURE_SW_2_I )
      wire#w2
      Contact( #O_BYTE_1.OPEN_PRESSURE_INPUT_2 )
      { S7_Templates := "time_type := Time" } #TIMER_DEACTD_PRESSURE_SWITCH_2.TON(pt := #TIMER_DEACTD_PRESSURE_SWITCH_2.PT, et =>)
      Coil( #ALARMS.OPEN_PRESSURE_SWITCH_2_ALARM )
   END_RUNG
   RUNG wire#powerrail
      Contact( #CLOSE )
   END_RUNG wire#w1
   RUNG wire#powerrail
      Contact( #ALARMS.OPEN_PRESSURE_SWITCH_2_ALARM )
      I_Contact( "DB2120_MPP_ITC_IPC".RESET_FAULTS )
   END_RUNG wire#w2
   // the same network as SCL:
   #TIMER_DEACTD_PRESSURE_SWITCH_2(IN := (((NOT #OPEN_ACTION OR #CLOSE) AND #CYL.OPEN_PRESSURE_SW_2_I) OR (#ALARMS.OPEN_PRESSURE_SWITCH_2_ALARM AND NOT "DB2120_MPP_ITC_IPC".RESET_FAULTS)) AND #O_BYTE_1.OPEN_PRESSURE_INPUT_2,   // TON
                           PT := #TIMER_DEACTD_PRESSURE_SWITCH_2.PT);
   #ALARMS.OPEN_PRESSURE_SWITCH_2_ALARM := #TIMER_DEACTD_PRESSURE_SWITCH_2.Q;
END_REGION

REGION Network 93: OPEN PRESSURE MISSING 2 ALARM
   RUNG wire#powerrail
      Contact( #M_VERIFY_OPEN )
      I_Contact( #CYL.OPEN_PRESSURE_SW_2_I )
      Contact( #CHECK_OPEN_CNC_PLC_SIGNAL )
      wire#w1
      Contact( #O_BYTE_1.OPEN_PRESSURE_INPUT_2 )
      Contact( #HYDRAULIC_OR_PNEUMATIC )
      Coil( #ALARMS.OPEN_PRESSURE_MISSING_2_ALARM )
   END_RUNG
   RUNG wire#powerrail
      Contact( #ALARMS.OPEN_PRESSURE_MISSING_2_ALARM )
      I_Contact( "DB2120_MPP_ITC_IPC".RESET_FAULTS )
   END_RUNG wire#w1
   // the same network as SCL:
   #ALARMS.OPEN_PRESSURE_MISSING_2_ALARM := ((#M_VERIFY_OPEN AND NOT #CYL.OPEN_PRESSURE_SW_2_I AND #CHECK_OPEN_CNC_PLC_SIGNAL) OR (#ALARMS.OPEN_PRESSURE_MISSING_2_ALARM AND NOT "DB2120_MPP_ITC_IPC".RESET_FAULTS)) AND #O_BYTE_1.OPEN_PRESSURE_INPUT_2 AND #HYDRAULIC_OR_PNEUMATIC;
END_REGION

REGION Network 94: CLOSED LOW PRESSURE TIME EXCEEDED ALARM
   RUNG wire#powerrail
      I_Contact( #CYL.CLOSE_LOW_PRESSURE_COMMAND )
      I_Contact( #LOW_PRESSURE )
      Not()
      Contact( #CYL.CLOSE_LOW_PRESSURE )
      I_Contact( #CLOSED_LOW_PRESSURE_SWITCH )
      wire#w1
      Contact( #O_BYTE_0.CLOSED_LOW_PRESSURE_INPUT )
      { S7_Templates := "time_type := Time" } #TIMER_ACTD_LOW_PRESSURE_TIME_EXCEEDED.TON(pt := #TIMER_ACTD_LOW_PRESSURE_TIME_EXCEEDED.PT, et =>)
      Coil( #ALARMS.CLOSED_LOW_PRESSURE_TIME_EXCEEDED_ALARM )
   END_RUNG
   RUNG wire#powerrail
      Contact( #ALARMS.CLOSED_LOW_PRESSURE_TIME_EXCEEDED_ALARM )
      I_Contact( "DB2120_MPP_ITC_IPC".RESET_FAULTS )
   END_RUNG wire#w1
   // the same network as SCL:
   #TIMER_ACTD_LOW_PRESSURE_TIME_EXCEEDED(IN := ((NOT (NOT #CYL.CLOSE_LOW_PRESSURE_COMMAND AND NOT #LOW_PRESSURE) AND #CYL.CLOSE_LOW_PRESSURE AND NOT #CLOSED_LOW_PRESSURE_SWITCH) OR (#ALARMS.CLOSED_LOW_PRESSURE_TIME_EXCEEDED_ALARM AND NOT "DB2120_MPP_ITC_IPC".RESET_FAULTS)) AND #O_BYTE_0.CLOSED_LOW_PRESSURE_INPUT,   // TON
                           PT := #TIMER_ACTD_LOW_PRESSURE_TIME_EXCEEDED.PT);
   #ALARMS.CLOSED_LOW_PRESSURE_TIME_EXCEEDED_ALARM := #TIMER_ACTD_LOW_PRESSURE_TIME_EXCEEDED.Q;
END_REGION

REGION Network 95: CLOSED LOW PRESSURE SWITCH ALARM
   RUNG wire#powerrail
      I_Contact( #LOW_PRESSURE )
      wire#w1
      Contact( #CLOSED_LOW_PRESSURE_SWITCH )
      wire#w2
      Contact( #O_BYTE_0.CLOSED_LOW_PRESSURE_INPUT )
      { S7_Templates := "time_type := Time" } #TIMER_ACTD_LOW_PRESSURE_SWITCH.TON(pt := #TIMER_ACTD_LOW_PRESSURE_SWITCH.PT, et =>)
      Coil( #ALARMS.CLOSED_LOW_PRESSURE_SWITCH_ALARM )
   END_RUNG
   RUNG wire#powerrail
      Contact( #OPEN_ACTION )
   END_RUNG wire#w1
   RUNG wire#powerrail
      Contact( #ALARMS.CLOSED_LOW_PRESSURE_SWITCH_ALARM )
      I_Contact( "DB2120_MPP_ITC_IPC".RESET_FAULTS )
   END_RUNG wire#w2
   // the same network as SCL:
   #TIMER_ACTD_LOW_PRESSURE_SWITCH(IN := (((NOT #LOW_PRESSURE OR #OPEN_ACTION) AND #CLOSED_LOW_PRESSURE_SWITCH) OR (#ALARMS.CLOSED_LOW_PRESSURE_SWITCH_ALARM AND NOT "DB2120_MPP_ITC_IPC".RESET_FAULTS)) AND #O_BYTE_0.CLOSED_LOW_PRESSURE_INPUT,   // TON
                           PT := #TIMER_ACTD_LOW_PRESSURE_SWITCH.PT);
   #ALARMS.CLOSED_LOW_PRESSURE_SWITCH_ALARM := #TIMER_ACTD_LOW_PRESSURE_SWITCH.Q;
END_REGION

REGION Network 96: CLOSED LOW PRESSURE MISSING ALARM
   RUNG wire#powerrail
      Contact( #M_VERIFY_LOW_PRESSURE )
      I_Contact( #CLOSED_LOW_PRESSURE_SWITCH )
      Contact( #CHECK_CLOSED_LOW_PRESSURE_CNC_PLC_SIGNAL )
      wire#w1
      Contact( #O_BYTE_0.CLOSED_LOW_PRESSURE_INPUT )
      Coil( #ALARMS.CLOSED_LOW_PRESSURE_MISSING_ALARM )
   END_RUNG
   RUNG wire#powerrail
      Contact( #ALARMS.CLOSED_LOW_PRESSURE_MISSING_ALARM )
      I_Contact( "DB2120_MPP_ITC_IPC".RESET_FAULTS )
   END_RUNG wire#w1
   // the same network as SCL:
   #ALARMS.CLOSED_LOW_PRESSURE_MISSING_ALARM := ((#M_VERIFY_LOW_PRESSURE AND NOT #CLOSED_LOW_PRESSURE_SWITCH AND #CHECK_CLOSED_LOW_PRESSURE_CNC_PLC_SIGNAL) OR (#ALARMS.CLOSED_LOW_PRESSURE_MISSING_ALARM AND NOT "DB2120_MPP_ITC_IPC".RESET_FAULTS)) AND #O_BYTE_0.CLOSED_LOW_PRESSURE_INPUT;
END_REGION

